(* CoDeSys 2.3.9.47 project: WTP_Pro_23_6_2016.pro *)
(* Libraries: STANDARD.LIB 5.6.98 12:03:02 *)

(* Task configuration *)
TASK Standard (PRIORITY := 0, INTERVAL := T#500ms);
	MAIN
END_TASK

(* Global variable list: Global_Variables *)
VAR_GLOBAL
	dummy: BOOL;
	LSH620 : inBlock;
	GlobalON: TIME := T#5s;
	GlobalOFF: TIME := T#5s;
END_VAR

(* Global variable list: TwinCAT_Configuration *)
(* Generated automatically by TwinCAT - (read only) *)
VAR_CONFIG
	GRIT_REMOVAL_OPERATION.B101A.dutyRemoteMode AT %IX2.1 : BOOL;
	GRIT_REMOVAL_OPERATION.B101A.dutyOverload AT %IX2.2 : BOOL;
	GRIT_REMOVAL_OPERATION.B101A.dutyIncomplete AT %IX2.3 : BOOL;
	GRIT_REMOVAL_OPERATION.B101A.dutyStart AT %IX2.4 : BOOL;
	GRIT_REMOVAL_OPERATION.B101A.standbyRemoteMode AT %IX2.5 : BOOL;
	GRIT_REMOVAL_OPERATION.B101A.standbyOverload AT %IX2.6 : BOOL;
	GRIT_REMOVAL_OPERATION.B101A.standbyIncomplete AT %IX2.7 : BOOL;
	GRIT_REMOVAL_OPERATION.B101A.standbyStart AT %IX3.0 : BOOL;
	GRIT_REMOVAL_OPERATION.B101A.thirdRemoteMode AT %IX3.1 : BOOL;
	GRIT_REMOVAL_OPERATION.B101A.thirdOverload AT %IX3.2 : BOOL;
	GRIT_REMOVAL_OPERATION.B101A.thirdStart AT %IX3.3 : BOOL;
	GRIT_REMOVAL_OPERATION.B101A.thirdIncomplete AT %IX3.4 : BOOL;
	GRIT_REMOVAL_OPERATION.B101A.standbyClose AT %IX3.5 : BOOL;
	GRIT_REMOVAL_OPERATION.B101A.dutyClose AT %IX3.6 : BOOL;
	GRIT_REMOVAL_OPERATION.B101A.thirdClose AT %IX3.7 : BOOL;
	GRIT_REMOVAL_OPERATION.B101A.dutyAdditionalStat AT %IX4.0 : BOOL;
	GRIT_REMOVAL_OPERATION.B101A.remoteAdditionalStat AT %IX4.1 : BOOL;
	GRIT_REMOVAL_OPERATION.B101A.thirdAdditionalStat AT %IX4.2 : BOOL;
	GRIT_REMOVAL_OPERATION.B101A.dutyCommand AT %QX0.0 : BOOL;
	GRIT_REMOVAL_OPERATION.B101A.standbyCommand AT %QX0.1 : BOOL;
	GRIT_REMOVAL_OPERATION.B101A.thirdCommand AT %QX0.2 : BOOL;
	GRIT_REMOVAL_OPERATION.XV100A.dutyRemoteMode AT %IX4.3 : BOOL;
	GRIT_REMOVAL_OPERATION.XV100A.dutyOverload AT %IX4.4 : BOOL;
	GRIT_REMOVAL_OPERATION.XV100A.dutyIncomplete AT %IX4.5 : BOOL;
	GRIT_REMOVAL_OPERATION.XV100A.dutyStart AT %IX4.6 : BOOL;
	GRIT_REMOVAL_OPERATION.XV100A.standbyRemoteMode AT %IX4.7 : BOOL;
	GRIT_REMOVAL_OPERATION.XV100A.standbyOverload AT %IX5.0 : BOOL;
	GRIT_REMOVAL_OPERATION.XV100A.standbyIncomplete AT %IX5.1 : BOOL;
	GRIT_REMOVAL_OPERATION.XV100A.standbyStart AT %IX5.2 : BOOL;
	GRIT_REMOVAL_OPERATION.XV100A.thirdRemoteMode AT %IX5.3 : BOOL;
	GRIT_REMOVAL_OPERATION.XV100A.thirdOverload AT %IX5.4 : BOOL;
	GRIT_REMOVAL_OPERATION.XV100A.thirdStart AT %IX5.5 : BOOL;
	GRIT_REMOVAL_OPERATION.XV100A.thirdIncomplete AT %IX5.6 : BOOL;
	GRIT_REMOVAL_OPERATION.XV100A.standbyClose AT %IX5.7 : BOOL;
	GRIT_REMOVAL_OPERATION.XV100A.dutyClose AT %IX6.0 : BOOL;
	GRIT_REMOVAL_OPERATION.XV100A.thirdClose AT %IX6.1 : BOOL;
	GRIT_REMOVAL_OPERATION.XV100A.dutyAdditionalStat AT %IX6.2 : BOOL;
	GRIT_REMOVAL_OPERATION.XV100A.remoteAdditionalStat AT %IX6.3 : BOOL;
	GRIT_REMOVAL_OPERATION.XV100A.thirdAdditionalStat AT %IX6.4 : BOOL;
	GRIT_REMOVAL_OPERATION.XV100A.dutyCommand AT %QX0.3 : BOOL;
	GRIT_REMOVAL_OPERATION.XV100A.standbyCommand AT %QX0.4 : BOOL;
	GRIT_REMOVAL_OPERATION.XV100A.thirdCommand AT %QX0.5 : BOOL;
	GRIT_REMOVAL_OPERATION.XV100B.dutyRemoteMode AT %IX6.5 : BOOL;
	GRIT_REMOVAL_OPERATION.XV100B.dutyOverload AT %IX6.6 : BOOL;
	GRIT_REMOVAL_OPERATION.XV100B.dutyIncomplete AT %IX6.7 : BOOL;
	GRIT_REMOVAL_OPERATION.XV100B.dutyStart AT %IX7.0 : BOOL;
	GRIT_REMOVAL_OPERATION.XV100B.standbyRemoteMode AT %IX7.1 : BOOL;
	GRIT_REMOVAL_OPERATION.XV100B.standbyOverload AT %IX7.2 : BOOL;
	GRIT_REMOVAL_OPERATION.XV100B.standbyIncomplete AT %IX7.3 : BOOL;
	GRIT_REMOVAL_OPERATION.XV100B.standbyStart AT %IX7.4 : BOOL;
	GRIT_REMOVAL_OPERATION.XV100B.thirdRemoteMode AT %IX7.5 : BOOL;
	GRIT_REMOVAL_OPERATION.XV100B.thirdOverload AT %IX7.6 : BOOL;
	GRIT_REMOVAL_OPERATION.XV100B.thirdStart AT %IX7.7 : BOOL;
	GRIT_REMOVAL_OPERATION.XV100B.thirdIncomplete AT %IX8.0 : BOOL;
	GRIT_REMOVAL_OPERATION.XV100B.standbyClose AT %IX8.1 : BOOL;
	GRIT_REMOVAL_OPERATION.XV100B.dutyClose AT %IX8.2 : BOOL;
	GRIT_REMOVAL_OPERATION.XV100B.thirdClose AT %IX8.3 : BOOL;
	GRIT_REMOVAL_OPERATION.XV100B.dutyAdditionalStat AT %IX8.4 : BOOL;
	GRIT_REMOVAL_OPERATION.XV100B.remoteAdditionalStat AT %IX8.5 : BOOL;
	GRIT_REMOVAL_OPERATION.XV100B.thirdAdditionalStat AT %IX8.6 : BOOL;
	GRIT_REMOVAL_OPERATION.XV100B.dutyCommand AT %QX0.6 : BOOL;
	GRIT_REMOVAL_OPERATION.XV100B.standbyCommand AT %QX0.7 : BOOL;
	GRIT_REMOVAL_OPERATION.XV100B.thirdCommand AT %QX1.0 : BOOL;
	GRIT_REMOVAL_OPERATION.C103AandB.dutyRemoteMode AT %IX8.7 : BOOL;
	GRIT_REMOVAL_OPERATION.C103AandB.dutyOverload AT %IX9.0 : BOOL;
	GRIT_REMOVAL_OPERATION.C103AandB.dutyIncomplete AT %IX9.1 : BOOL;
	GRIT_REMOVAL_OPERATION.C103AandB.dutyStart AT %IX9.2 : BOOL;
	GRIT_REMOVAL_OPERATION.C103AandB.standbyRemoteMode AT %IX9.3 : BOOL;
	GRIT_REMOVAL_OPERATION.C103AandB.standbyOverload AT %IX9.4 : BOOL;
	GRIT_REMOVAL_OPERATION.C103AandB.standbyIncomplete AT %IX9.5 : BOOL;
	GRIT_REMOVAL_OPERATION.C103AandB.standbyStart AT %IX9.6 : BOOL;
	GRIT_REMOVAL_OPERATION.C103AandB.thirdRemoteMode AT %IX9.7 : BOOL;
	GRIT_REMOVAL_OPERATION.C103AandB.thirdOverload AT %IX10.0 : BOOL;
	GRIT_REMOVAL_OPERATION.C103AandB.thirdStart AT %IX10.1 : BOOL;
	GRIT_REMOVAL_OPERATION.C103AandB.thirdIncomplete AT %IX10.2 : BOOL;
	GRIT_REMOVAL_OPERATION.C103AandB.standbyClose AT %IX10.3 : BOOL;
	GRIT_REMOVAL_OPERATION.C103AandB.dutyClose AT %IX10.4 : BOOL;
	GRIT_REMOVAL_OPERATION.C103AandB.thirdClose AT %IX10.5 : BOOL;
	GRIT_REMOVAL_OPERATION.C103AandB.dutyAdditionalStat AT %IX10.6 : BOOL;
	GRIT_REMOVAL_OPERATION.C103AandB.remoteAdditionalStat AT %IX10.7 : BOOL;
	GRIT_REMOVAL_OPERATION.C103AandB.thirdAdditionalStat AT %IX11.0 : BOOL;
	GRIT_REMOVAL_OPERATION.C103AandB.dutyCommand AT %QX1.1 : BOOL;
	GRIT_REMOVAL_OPERATION.C103AandB.standbyCommand AT %QX1.2 : BOOL;
	GRIT_REMOVAL_OPERATION.C103AandB.thirdCommand AT %QX1.3 : BOOL;
	INLET_SCREENING_OPERATION_1.LSH105A.IN AT %IX38.7 : BOOL;
	INLET_SCREENING_OPERATION_1.LSHH105A.IN AT %IX39.0 : BOOL;
	INLET_SCREENING_OPERATION_1.F101A.dutyRemoteMode AT %IX39.1 : BOOL;
	INLET_SCREENING_OPERATION_1.F101A.dutyOverload AT %IX39.2 : BOOL;
	INLET_SCREENING_OPERATION_1.F101A.dutyIncomplete AT %IX39.3 : BOOL;
	INLET_SCREENING_OPERATION_1.F101A.dutyStart AT %IX39.4 : BOOL;
	INLET_SCREENING_OPERATION_1.F101A.standbyRemoteMode AT %IX39.5 : BOOL;
	INLET_SCREENING_OPERATION_1.F101A.standbyOverload AT %IX39.6 : BOOL;
	INLET_SCREENING_OPERATION_1.F101A.standbyIncomplete AT %IX39.7 : BOOL;
	INLET_SCREENING_OPERATION_1.F101A.standbyStart AT %IX40.0 : BOOL;
	INLET_SCREENING_OPERATION_1.F101A.thirdRemoteMode AT %IX40.1 : BOOL;
	INLET_SCREENING_OPERATION_1.F101A.thirdOverload AT %IX40.2 : BOOL;
	INLET_SCREENING_OPERATION_1.F101A.thirdStart AT %IX40.3 : BOOL;
	INLET_SCREENING_OPERATION_1.F101A.thirdIncomplete AT %IX40.4 : BOOL;
	INLET_SCREENING_OPERATION_1.F101A.standbyClose AT %IX40.5 : BOOL;
	INLET_SCREENING_OPERATION_1.F101A.dutyClose AT %IX40.6 : BOOL;
	INLET_SCREENING_OPERATION_1.F101A.thirdClose AT %IX40.7 : BOOL;
	INLET_SCREENING_OPERATION_1.F101A.dutyAdditionalStat AT %IX41.0 : BOOL;
	INLET_SCREENING_OPERATION_1.F101A.remoteAdditionalStat AT %IX41.1 : BOOL;
	INLET_SCREENING_OPERATION_1.F101A.thirdAdditionalStat AT %IX41.2 : BOOL;
	INLET_SCREENING_OPERATION_1.F101A.dutyCommand AT %QX5.5 : BOOL;
	INLET_SCREENING_OPERATION_1.F101A.standbyCommand AT %QX5.6 : BOOL;
	INLET_SCREENING_OPERATION_1.F101A.thirdCommand AT %QX5.7 : BOOL;
	INLET_SCREENING_OPERATION_1.XV101A1.dutyRemoteMode AT %IX41.3 : BOOL;
	INLET_SCREENING_OPERATION_1.XV101A1.dutyOverload AT %IX41.4 : BOOL;
	INLET_SCREENING_OPERATION_1.XV101A1.dutyIncomplete AT %IX41.5 : BOOL;
	INLET_SCREENING_OPERATION_1.XV101A1.dutyStart AT %IX41.6 : BOOL;
	INLET_SCREENING_OPERATION_1.XV101A1.standbyRemoteMode AT %IX41.7 : BOOL;
	INLET_SCREENING_OPERATION_1.XV101A1.standbyOverload AT %IX42.0 : BOOL;
	INLET_SCREENING_OPERATION_1.XV101A1.standbyIncomplete AT %IX42.1 : BOOL;
	INLET_SCREENING_OPERATION_1.XV101A1.standbyStart AT %IX42.2 : BOOL;
	INLET_SCREENING_OPERATION_1.XV101A1.thirdRemoteMode AT %IX42.3 : BOOL;
	INLET_SCREENING_OPERATION_1.XV101A1.thirdOverload AT %IX42.4 : BOOL;
	INLET_SCREENING_OPERATION_1.XV101A1.thirdStart AT %IX42.5 : BOOL;
	INLET_SCREENING_OPERATION_1.XV101A1.thirdIncomplete AT %IX42.6 : BOOL;
	INLET_SCREENING_OPERATION_1.XV101A1.standbyClose AT %IX42.7 : BOOL;
	INLET_SCREENING_OPERATION_1.XV101A1.dutyClose AT %IX43.0 : BOOL;
	INLET_SCREENING_OPERATION_1.XV101A1.thirdClose AT %IX43.1 : BOOL;
	INLET_SCREENING_OPERATION_1.XV101A1.dutyAdditionalStat AT %IX43.2 : BOOL;
	INLET_SCREENING_OPERATION_1.XV101A1.remoteAdditionalStat AT %IX43.3 : BOOL;
	INLET_SCREENING_OPERATION_1.XV101A1.thirdAdditionalStat AT %IX43.4 : BOOL;
	INLET_SCREENING_OPERATION_1.XV101A1.dutyCommand AT %QX6.0 : BOOL;
	INLET_SCREENING_OPERATION_1.XV101A1.standbyCommand AT %QX6.1 : BOOL;
	INLET_SCREENING_OPERATION_1.XV101A1.thirdCommand AT %QX6.2 : BOOL;
	INLET_SCREENING_OPERATION_1.XV101A2.dutyRemoteMode AT %IX43.5 : BOOL;
	INLET_SCREENING_OPERATION_1.XV101A2.dutyOverload AT %IX43.6 : BOOL;
	INLET_SCREENING_OPERATION_1.XV101A2.dutyIncomplete AT %IX43.7 : BOOL;
	INLET_SCREENING_OPERATION_1.XV101A2.dutyStart AT %IX44.0 : BOOL;
	INLET_SCREENING_OPERATION_1.XV101A2.standbyRemoteMode AT %IX44.1 : BOOL;
	INLET_SCREENING_OPERATION_1.XV101A2.standbyOverload AT %IX44.2 : BOOL;
	INLET_SCREENING_OPERATION_1.XV101A2.standbyIncomplete AT %IX44.3 : BOOL;
	INLET_SCREENING_OPERATION_1.XV101A2.standbyStart AT %IX44.4 : BOOL;
	INLET_SCREENING_OPERATION_1.XV101A2.thirdRemoteMode AT %IX44.5 : BOOL;
	INLET_SCREENING_OPERATION_1.XV101A2.thirdOverload AT %IX44.6 : BOOL;
	INLET_SCREENING_OPERATION_1.XV101A2.thirdStart AT %IX44.7 : BOOL;
	INLET_SCREENING_OPERATION_1.XV101A2.thirdIncomplete AT %IX45.0 : BOOL;
	INLET_SCREENING_OPERATION_1.XV101A2.standbyClose AT %IX45.1 : BOOL;
	INLET_SCREENING_OPERATION_1.XV101A2.dutyClose AT %IX45.2 : BOOL;
	INLET_SCREENING_OPERATION_1.XV101A2.thirdClose AT %IX45.3 : BOOL;
	INLET_SCREENING_OPERATION_1.XV101A2.dutyAdditionalStat AT %IX45.4 : BOOL;
	INLET_SCREENING_OPERATION_1.XV101A2.remoteAdditionalStat AT %IX45.5 : BOOL;
	INLET_SCREENING_OPERATION_1.XV101A2.thirdAdditionalStat AT %IX45.6 : BOOL;
	INLET_SCREENING_OPERATION_1.XV101A2.dutyCommand AT %QX6.3 : BOOL;
	INLET_SCREENING_OPERATION_1.XV101A2.standbyCommand AT %QX6.4 : BOOL;
	INLET_SCREENING_OPERATION_1.XV101A2.thirdCommand AT %QX6.5 : BOOL;
	INLET_SCREENING_OPERATION_1.PS101A.dutyRemoteMode AT %IX45.7 : BOOL;
	INLET_SCREENING_OPERATION_1.PS101A.dutyOverload AT %IX46.0 : BOOL;
	INLET_SCREENING_OPERATION_1.PS101A.dutyIncomplete AT %IX46.1 : BOOL;
	INLET_SCREENING_OPERATION_1.PS101A.dutyStart AT %IX46.2 : BOOL;
	INLET_SCREENING_OPERATION_1.PS101A.standbyRemoteMode AT %IX46.3 : BOOL;
	INLET_SCREENING_OPERATION_1.PS101A.standbyOverload AT %IX46.4 : BOOL;
	INLET_SCREENING_OPERATION_1.PS101A.standbyIncomplete AT %IX46.5 : BOOL;
	INLET_SCREENING_OPERATION_1.PS101A.standbyStart AT %IX46.6 : BOOL;
	INLET_SCREENING_OPERATION_1.PS101A.thirdRemoteMode AT %IX46.7 : BOOL;
	INLET_SCREENING_OPERATION_1.PS101A.thirdOverload AT %IX47.0 : BOOL;
	INLET_SCREENING_OPERATION_1.PS101A.thirdStart AT %IX47.1 : BOOL;
	INLET_SCREENING_OPERATION_1.PS101A.thirdIncomplete AT %IX47.2 : BOOL;
	INLET_SCREENING_OPERATION_1.PS101A.standbyClose AT %IX47.3 : BOOL;
	INLET_SCREENING_OPERATION_1.PS101A.dutyClose AT %IX47.4 : BOOL;
	INLET_SCREENING_OPERATION_1.PS101A.thirdClose AT %IX47.5 : BOOL;
	INLET_SCREENING_OPERATION_1.PS101A.dutyAdditionalStat AT %IX47.6 : BOOL;
	INLET_SCREENING_OPERATION_1.PS101A.remoteAdditionalStat AT %IX47.7 : BOOL;
	INLET_SCREENING_OPERATION_1.PS101A.thirdAdditionalStat AT %IX48.0 : BOOL;
	INLET_SCREENING_OPERATION_1.PS101A.dutyCommand AT %QX6.6 : BOOL;
	INLET_SCREENING_OPERATION_1.PS101A.standbyCommand AT %QX6.7 : BOOL;
	INLET_SCREENING_OPERATION_1.PS101A.thirdCommand AT %QX7.0 : BOOL;
	INLET_SCREENING_OPERATION_1.C102A.dutyRemoteMode AT %IX48.1 : BOOL;
	INLET_SCREENING_OPERATION_1.C102A.dutyOverload AT %IX48.2 : BOOL;
	INLET_SCREENING_OPERATION_1.C102A.dutyIncomplete AT %IX48.3 : BOOL;
	INLET_SCREENING_OPERATION_1.C102A.dutyStart AT %IX48.4 : BOOL;
	INLET_SCREENING_OPERATION_1.C102A.standbyRemoteMode AT %IX48.5 : BOOL;
	INLET_SCREENING_OPERATION_1.C102A.standbyOverload AT %IX48.6 : BOOL;
	INLET_SCREENING_OPERATION_1.C102A.standbyIncomplete AT %IX48.7 : BOOL;
	INLET_SCREENING_OPERATION_1.C102A.standbyStart AT %IX49.0 : BOOL;
	INLET_SCREENING_OPERATION_1.C102A.thirdRemoteMode AT %IX49.1 : BOOL;
	INLET_SCREENING_OPERATION_1.C102A.thirdOverload AT %IX49.2 : BOOL;
	INLET_SCREENING_OPERATION_1.C102A.thirdStart AT %IX49.3 : BOOL;
	INLET_SCREENING_OPERATION_1.C102A.thirdIncomplete AT %IX49.4 : BOOL;
	INLET_SCREENING_OPERATION_1.C102A.standbyClose AT %IX49.5 : BOOL;
	INLET_SCREENING_OPERATION_1.C102A.dutyClose AT %IX49.6 : BOOL;
	INLET_SCREENING_OPERATION_1.C102A.thirdClose AT %IX49.7 : BOOL;
	INLET_SCREENING_OPERATION_1.C102A.dutyAdditionalStat AT %IX50.0 : BOOL;
	INLET_SCREENING_OPERATION_1.C102A.remoteAdditionalStat AT %IX50.1 : BOOL;
	INLET_SCREENING_OPERATION_1.C102A.thirdAdditionalStat AT %IX50.2 : BOOL;
	INLET_SCREENING_OPERATION_1.C102A.dutyCommand AT %QX7.1 : BOOL;
	INLET_SCREENING_OPERATION_1.C102A.standbyCommand AT %QX7.2 : BOOL;
	INLET_SCREENING_OPERATION_1.C102A.thirdCommand AT %QX7.3 : BOOL;
	INLET_SCREENING_OPERATION_1.C101A.dutyRemoteMode AT %IX50.3 : BOOL;
	INLET_SCREENING_OPERATION_1.C101A.dutyOverload AT %IX50.4 : BOOL;
	INLET_SCREENING_OPERATION_1.C101A.dutyIncomplete AT %IX50.5 : BOOL;
	INLET_SCREENING_OPERATION_1.C101A.dutyStart AT %IX50.6 : BOOL;
	INLET_SCREENING_OPERATION_1.C101A.standbyRemoteMode AT %IX50.7 : BOOL;
	INLET_SCREENING_OPERATION_1.C101A.standbyOverload AT %IX51.0 : BOOL;
	INLET_SCREENING_OPERATION_1.C101A.standbyIncomplete AT %IX51.1 : BOOL;
	INLET_SCREENING_OPERATION_1.C101A.standbyStart AT %IX51.2 : BOOL;
	INLET_SCREENING_OPERATION_1.C101A.thirdRemoteMode AT %IX51.3 : BOOL;
	INLET_SCREENING_OPERATION_1.C101A.thirdOverload AT %IX51.4 : BOOL;
	INLET_SCREENING_OPERATION_1.C101A.thirdStart AT %IX51.5 : BOOL;
	INLET_SCREENING_OPERATION_1.C101A.thirdIncomplete AT %IX51.6 : BOOL;
	INLET_SCREENING_OPERATION_1.C101A.standbyClose AT %IX51.7 : BOOL;
	INLET_SCREENING_OPERATION_1.C101A.dutyClose AT %IX52.0 : BOOL;
	INLET_SCREENING_OPERATION_1.C101A.thirdClose AT %IX52.1 : BOOL;
	INLET_SCREENING_OPERATION_1.C101A.dutyAdditionalStat AT %IX52.2 : BOOL;
	INLET_SCREENING_OPERATION_1.C101A.remoteAdditionalStat AT %IX52.3 : BOOL;
	INLET_SCREENING_OPERATION_1.C101A.thirdAdditionalStat AT %IX52.4 : BOOL;
	INLET_SCREENING_OPERATION_1.C101A.dutyCommand AT %QX7.4 : BOOL;
	INLET_SCREENING_OPERATION_1.C101A.standbyCommand AT %QX7.5 : BOOL;
	INLET_SCREENING_OPERATION_1.C101A.thirdCommand AT %QX7.6 : BOOL;
	INLET_SCREENING_OPERATION_1.XV102A.dutyRemoteMode AT %IX52.5 : BOOL;
	INLET_SCREENING_OPERATION_1.XV102A.dutyOverload AT %IX52.6 : BOOL;
	INLET_SCREENING_OPERATION_1.XV102A.dutyIncomplete AT %IX52.7 : BOOL;
	INLET_SCREENING_OPERATION_1.XV102A.dutyStart AT %IX53.0 : BOOL;
	INLET_SCREENING_OPERATION_1.XV102A.standbyRemoteMode AT %IX53.1 : BOOL;
	INLET_SCREENING_OPERATION_1.XV102A.standbyOverload AT %IX53.2 : BOOL;
	INLET_SCREENING_OPERATION_1.XV102A.standbyIncomplete AT %IX53.3 : BOOL;
	INLET_SCREENING_OPERATION_1.XV102A.standbyStart AT %IX53.4 : BOOL;
	INLET_SCREENING_OPERATION_1.XV102A.thirdRemoteMode AT %IX53.5 : BOOL;
	INLET_SCREENING_OPERATION_1.XV102A.thirdOverload AT %IX53.6 : BOOL;
	INLET_SCREENING_OPERATION_1.XV102A.thirdStart AT %IX53.7 : BOOL;
	INLET_SCREENING_OPERATION_1.XV102A.thirdIncomplete AT %IX54.0 : BOOL;
	INLET_SCREENING_OPERATION_1.XV102A.standbyClose AT %IX54.1 : BOOL;
	INLET_SCREENING_OPERATION_1.XV102A.dutyClose AT %IX54.2 : BOOL;
	INLET_SCREENING_OPERATION_1.XV102A.thirdClose AT %IX54.3 : BOOL;
	INLET_SCREENING_OPERATION_1.XV102A.dutyAdditionalStat AT %IX54.4 : BOOL;
	INLET_SCREENING_OPERATION_1.XV102A.remoteAdditionalStat AT %IX54.5 : BOOL;
	INLET_SCREENING_OPERATION_1.XV102A.thirdAdditionalStat AT %IX54.6 : BOOL;
	INLET_SCREENING_OPERATION_1.XV102A.dutyCommand AT %QX7.7 : BOOL;
	INLET_SCREENING_OPERATION_1.XV102A.standbyCommand AT %QX8.0 : BOOL;
	INLET_SCREENING_OPERATION_1.XV102A.thirdCommand AT %QX8.1 : BOOL;
	INLET_SCREENING_OPERATION_2.LSH105B.IN AT %IX54.7 : BOOL;
	INLET_SCREENING_OPERATION_2.LSHH105B.IN AT %IX55.0 : BOOL;
	INLET_SCREENING_OPERATION_2.F101B.dutyRemoteMode AT %IX55.1 : BOOL;
	INLET_SCREENING_OPERATION_2.F101B.dutyOverload AT %IX55.2 : BOOL;
	INLET_SCREENING_OPERATION_2.F101B.dutyIncomplete AT %IX55.3 : BOOL;
	INLET_SCREENING_OPERATION_2.F101B.dutyStart AT %IX55.4 : BOOL;
	INLET_SCREENING_OPERATION_2.F101B.standbyRemoteMode AT %IX55.5 : BOOL;
	INLET_SCREENING_OPERATION_2.F101B.standbyOverload AT %IX55.6 : BOOL;
	INLET_SCREENING_OPERATION_2.F101B.standbyIncomplete AT %IX55.7 : BOOL;
	INLET_SCREENING_OPERATION_2.F101B.standbyStart AT %IX56.0 : BOOL;
	INLET_SCREENING_OPERATION_2.F101B.thirdRemoteMode AT %IX56.1 : BOOL;
	INLET_SCREENING_OPERATION_2.F101B.thirdOverload AT %IX56.2 : BOOL;
	INLET_SCREENING_OPERATION_2.F101B.thirdStart AT %IX56.3 : BOOL;
	INLET_SCREENING_OPERATION_2.F101B.thirdIncomplete AT %IX56.4 : BOOL;
	INLET_SCREENING_OPERATION_2.F101B.standbyClose AT %IX56.5 : BOOL;
	INLET_SCREENING_OPERATION_2.F101B.dutyClose AT %IX56.6 : BOOL;
	INLET_SCREENING_OPERATION_2.F101B.thirdClose AT %IX56.7 : BOOL;
	INLET_SCREENING_OPERATION_2.F101B.dutyAdditionalStat AT %IX57.0 : BOOL;
	INLET_SCREENING_OPERATION_2.F101B.remoteAdditionalStat AT %IX57.1 : BOOL;
	INLET_SCREENING_OPERATION_2.F101B.thirdAdditionalStat AT %IX57.2 : BOOL;
	INLET_SCREENING_OPERATION_2.F101B.dutyCommand AT %QX8.2 : BOOL;
	INLET_SCREENING_OPERATION_2.F101B.standbyCommand AT %QX8.3 : BOOL;
	INLET_SCREENING_OPERATION_2.F101B.thirdCommand AT %QX8.4 : BOOL;
	INLET_SCREENING_OPERATION_2.XV101B1.dutyRemoteMode AT %IX57.3 : BOOL;
	INLET_SCREENING_OPERATION_2.XV101B1.dutyOverload AT %IX57.4 : BOOL;
	INLET_SCREENING_OPERATION_2.XV101B1.dutyIncomplete AT %IX57.5 : BOOL;
	INLET_SCREENING_OPERATION_2.XV101B1.dutyStart AT %IX57.6 : BOOL;
	INLET_SCREENING_OPERATION_2.XV101B1.standbyRemoteMode AT %IX57.7 : BOOL;
	INLET_SCREENING_OPERATION_2.XV101B1.standbyOverload AT %IX58.0 : BOOL;
	INLET_SCREENING_OPERATION_2.XV101B1.standbyIncomplete AT %IX58.1 : BOOL;
	INLET_SCREENING_OPERATION_2.XV101B1.standbyStart AT %IX58.2 : BOOL;
	INLET_SCREENING_OPERATION_2.XV101B1.thirdRemoteMode AT %IX58.3 : BOOL;
	INLET_SCREENING_OPERATION_2.XV101B1.thirdOverload AT %IX58.4 : BOOL;
	INLET_SCREENING_OPERATION_2.XV101B1.thirdStart AT %IX58.5 : BOOL;
	INLET_SCREENING_OPERATION_2.XV101B1.thirdIncomplete AT %IX58.6 : BOOL;
	INLET_SCREENING_OPERATION_2.XV101B1.standbyClose AT %IX58.7 : BOOL;
	INLET_SCREENING_OPERATION_2.XV101B1.dutyClose AT %IX59.0 : BOOL;
	INLET_SCREENING_OPERATION_2.XV101B1.thirdClose AT %IX59.1 : BOOL;
	INLET_SCREENING_OPERATION_2.XV101B1.dutyAdditionalStat AT %IX59.2 : BOOL;
	INLET_SCREENING_OPERATION_2.XV101B1.remoteAdditionalStat AT %IX59.3 : BOOL;
	INLET_SCREENING_OPERATION_2.XV101B1.thirdAdditionalStat AT %IX59.4 : BOOL;
	INLET_SCREENING_OPERATION_2.XV101B1.dutyCommand AT %QX8.5 : BOOL;
	INLET_SCREENING_OPERATION_2.XV101B1.standbyCommand AT %QX8.6 : BOOL;
	INLET_SCREENING_OPERATION_2.XV101B1.thirdCommand AT %QX8.7 : BOOL;
	INLET_SCREENING_OPERATION_2.XV101B2.dutyRemoteMode AT %IX59.5 : BOOL;
	INLET_SCREENING_OPERATION_2.XV101B2.dutyOverload AT %IX59.6 : BOOL;
	INLET_SCREENING_OPERATION_2.XV101B2.dutyIncomplete AT %IX59.7 : BOOL;
	INLET_SCREENING_OPERATION_2.XV101B2.dutyStart AT %IX60.0 : BOOL;
	INLET_SCREENING_OPERATION_2.XV101B2.standbyRemoteMode AT %IX60.1 : BOOL;
	INLET_SCREENING_OPERATION_2.XV101B2.standbyOverload AT %IX60.2 : BOOL;
	INLET_SCREENING_OPERATION_2.XV101B2.standbyIncomplete AT %IX60.3 : BOOL;
	INLET_SCREENING_OPERATION_2.XV101B2.standbyStart AT %IX60.4 : BOOL;
	INLET_SCREENING_OPERATION_2.XV101B2.thirdRemoteMode AT %IX60.5 : BOOL;
	INLET_SCREENING_OPERATION_2.XV101B2.thirdOverload AT %IX60.6 : BOOL;
	INLET_SCREENING_OPERATION_2.XV101B2.thirdStart AT %IX60.7 : BOOL;
	INLET_SCREENING_OPERATION_2.XV101B2.thirdIncomplete AT %IX61.0 : BOOL;
	INLET_SCREENING_OPERATION_2.XV101B2.standbyClose AT %IX61.1 : BOOL;
	INLET_SCREENING_OPERATION_2.XV101B2.dutyClose AT %IX61.2 : BOOL;
	INLET_SCREENING_OPERATION_2.XV101B2.thirdClose AT %IX61.3 : BOOL;
	INLET_SCREENING_OPERATION_2.XV101B2.dutyAdditionalStat AT %IX61.4 : BOOL;
	INLET_SCREENING_OPERATION_2.XV101B2.remoteAdditionalStat AT %IX61.5 : BOOL;
	INLET_SCREENING_OPERATION_2.XV101B2.thirdAdditionalStat AT %IX61.6 : BOOL;
	INLET_SCREENING_OPERATION_2.XV101B2.dutyCommand AT %QX9.0 : BOOL;
	INLET_SCREENING_OPERATION_2.XV101B2.standbyCommand AT %QX9.1 : BOOL;
	INLET_SCREENING_OPERATION_2.XV101B2.thirdCommand AT %QX9.2 : BOOL;
	INLET_SCREENING_OPERATION_2.PS101B.dutyRemoteMode AT %IX61.7 : BOOL;
	INLET_SCREENING_OPERATION_2.PS101B.dutyOverload AT %IX62.0 : BOOL;
	INLET_SCREENING_OPERATION_2.PS101B.dutyIncomplete AT %IX62.1 : BOOL;
	INLET_SCREENING_OPERATION_2.PS101B.dutyStart AT %IX62.2 : BOOL;
	INLET_SCREENING_OPERATION_2.PS101B.standbyRemoteMode AT %IX62.3 : BOOL;
	INLET_SCREENING_OPERATION_2.PS101B.standbyOverload AT %IX62.4 : BOOL;
	INLET_SCREENING_OPERATION_2.PS101B.standbyIncomplete AT %IX62.5 : BOOL;
	INLET_SCREENING_OPERATION_2.PS101B.standbyStart AT %IX62.6 : BOOL;
	INLET_SCREENING_OPERATION_2.PS101B.thirdRemoteMode AT %IX62.7 : BOOL;
	INLET_SCREENING_OPERATION_2.PS101B.thirdOverload AT %IX63.0 : BOOL;
	INLET_SCREENING_OPERATION_2.PS101B.thirdStart AT %IX63.1 : BOOL;
	INLET_SCREENING_OPERATION_2.PS101B.thirdIncomplete AT %IX63.2 : BOOL;
	INLET_SCREENING_OPERATION_2.PS101B.standbyClose AT %IX63.3 : BOOL;
	INLET_SCREENING_OPERATION_2.PS101B.dutyClose AT %IX63.4 : BOOL;
	INLET_SCREENING_OPERATION_2.PS101B.thirdClose AT %IX63.5 : BOOL;
	INLET_SCREENING_OPERATION_2.PS101B.dutyAdditionalStat AT %IX63.6 : BOOL;
	INLET_SCREENING_OPERATION_2.PS101B.remoteAdditionalStat AT %IX63.7 : BOOL;
	INLET_SCREENING_OPERATION_2.PS101B.thirdAdditionalStat AT %IX64.0 : BOOL;
	INLET_SCREENING_OPERATION_2.PS101B.dutyCommand AT %QX9.3 : BOOL;
	INLET_SCREENING_OPERATION_2.PS101B.standbyCommand AT %QX9.4 : BOOL;
	INLET_SCREENING_OPERATION_2.PS101B.thirdCommand AT %QX9.5 : BOOL;
	INLET_SCREENING_OPERATION_2.C102B.dutyRemoteMode AT %IX64.1 : BOOL;
	INLET_SCREENING_OPERATION_2.C102B.dutyOverload AT %IX64.2 : BOOL;
	INLET_SCREENING_OPERATION_2.C102B.dutyIncomplete AT %IX64.3 : BOOL;
	INLET_SCREENING_OPERATION_2.C102B.dutyStart AT %IX64.4 : BOOL;
	INLET_SCREENING_OPERATION_2.C102B.standbyRemoteMode AT %IX64.5 : BOOL;
	INLET_SCREENING_OPERATION_2.C102B.standbyOverload AT %IX64.6 : BOOL;
	INLET_SCREENING_OPERATION_2.C102B.standbyIncomplete AT %IX64.7 : BOOL;
	INLET_SCREENING_OPERATION_2.C102B.standbyStart AT %IX65.0 : BOOL;
	INLET_SCREENING_OPERATION_2.C102B.thirdRemoteMode AT %IX65.1 : BOOL;
	INLET_SCREENING_OPERATION_2.C102B.thirdOverload AT %IX65.2 : BOOL;
	INLET_SCREENING_OPERATION_2.C102B.thirdStart AT %IX65.3 : BOOL;
	INLET_SCREENING_OPERATION_2.C102B.thirdIncomplete AT %IX65.4 : BOOL;
	INLET_SCREENING_OPERATION_2.C102B.standbyClose AT %IX65.5 : BOOL;
	INLET_SCREENING_OPERATION_2.C102B.dutyClose AT %IX65.6 : BOOL;
	INLET_SCREENING_OPERATION_2.C102B.thirdClose AT %IX65.7 : BOOL;
	INLET_SCREENING_OPERATION_2.C102B.dutyAdditionalStat AT %IX66.0 : BOOL;
	INLET_SCREENING_OPERATION_2.C102B.remoteAdditionalStat AT %IX66.1 : BOOL;
	INLET_SCREENING_OPERATION_2.C102B.thirdAdditionalStat AT %IX66.2 : BOOL;
	INLET_SCREENING_OPERATION_2.C102B.dutyCommand AT %QX9.6 : BOOL;
	INLET_SCREENING_OPERATION_2.C102B.standbyCommand AT %QX9.7 : BOOL;
	INLET_SCREENING_OPERATION_2.C102B.thirdCommand AT %QX10.0 : BOOL;
	INLET_SCREENING_OPERATION_2.C101B.dutyRemoteMode AT %IX66.3 : BOOL;
	INLET_SCREENING_OPERATION_2.C101B.dutyOverload AT %IX66.4 : BOOL;
	INLET_SCREENING_OPERATION_2.C101B.dutyIncomplete AT %IX66.5 : BOOL;
	INLET_SCREENING_OPERATION_2.C101B.dutyStart AT %IX66.6 : BOOL;
	INLET_SCREENING_OPERATION_2.C101B.standbyRemoteMode AT %IX66.7 : BOOL;
	INLET_SCREENING_OPERATION_2.C101B.standbyOverload AT %IX67.0 : BOOL;
	INLET_SCREENING_OPERATION_2.C101B.standbyIncomplete AT %IX67.1 : BOOL;
	INLET_SCREENING_OPERATION_2.C101B.standbyStart AT %IX67.2 : BOOL;
	INLET_SCREENING_OPERATION_2.C101B.thirdRemoteMode AT %IX67.3 : BOOL;
	INLET_SCREENING_OPERATION_2.C101B.thirdOverload AT %IX67.4 : BOOL;
	INLET_SCREENING_OPERATION_2.C101B.thirdStart AT %IX67.5 : BOOL;
	INLET_SCREENING_OPERATION_2.C101B.thirdIncomplete AT %IX67.6 : BOOL;
	INLET_SCREENING_OPERATION_2.C101B.standbyClose AT %IX67.7 : BOOL;
	INLET_SCREENING_OPERATION_2.C101B.dutyClose AT %IX68.0 : BOOL;
	INLET_SCREENING_OPERATION_2.C101B.thirdClose AT %IX68.1 : BOOL;
	INLET_SCREENING_OPERATION_2.C101B.dutyAdditionalStat AT %IX68.2 : BOOL;
	INLET_SCREENING_OPERATION_2.C101B.remoteAdditionalStat AT %IX68.3 : BOOL;
	INLET_SCREENING_OPERATION_2.C101B.thirdAdditionalStat AT %IX68.4 : BOOL;
	INLET_SCREENING_OPERATION_2.C101B.dutyCommand AT %QX10.1 : BOOL;
	INLET_SCREENING_OPERATION_2.C101B.standbyCommand AT %QX10.2 : BOOL;
	INLET_SCREENING_OPERATION_2.C101B.thirdCommand AT %QX10.3 : BOOL;
	INLET_SCREENING_OPERATION_2.XV102B.dutyRemoteMode AT %IX68.5 : BOOL;
	INLET_SCREENING_OPERATION_2.XV102B.dutyOverload AT %IX68.6 : BOOL;
	INLET_SCREENING_OPERATION_2.XV102B.dutyIncomplete AT %IX68.7 : BOOL;
	INLET_SCREENING_OPERATION_2.XV102B.dutyStart AT %IX69.0 : BOOL;
	INLET_SCREENING_OPERATION_2.XV102B.standbyRemoteMode AT %IX69.1 : BOOL;
	INLET_SCREENING_OPERATION_2.XV102B.standbyOverload AT %IX69.2 : BOOL;
	INLET_SCREENING_OPERATION_2.XV102B.standbyIncomplete AT %IX69.3 : BOOL;
	INLET_SCREENING_OPERATION_2.XV102B.standbyStart AT %IX69.4 : BOOL;
	INLET_SCREENING_OPERATION_2.XV102B.thirdRemoteMode AT %IX69.5 : BOOL;
	INLET_SCREENING_OPERATION_2.XV102B.thirdOverload AT %IX69.6 : BOOL;
	INLET_SCREENING_OPERATION_2.XV102B.thirdStart AT %IX69.7 : BOOL;
	INLET_SCREENING_OPERATION_2.XV102B.thirdIncomplete AT %IX70.0 : BOOL;
	INLET_SCREENING_OPERATION_2.XV102B.standbyClose AT %IX70.1 : BOOL;
	INLET_SCREENING_OPERATION_2.XV102B.dutyClose AT %IX70.2 : BOOL;
	INLET_SCREENING_OPERATION_2.XV102B.thirdClose AT %IX70.3 : BOOL;
	INLET_SCREENING_OPERATION_2.XV102B.dutyAdditionalStat AT %IX70.4 : BOOL;
	INLET_SCREENING_OPERATION_2.XV102B.remoteAdditionalStat AT %IX70.5 : BOOL;
	INLET_SCREENING_OPERATION_2.XV102B.thirdAdditionalStat AT %IX70.6 : BOOL;
	INLET_SCREENING_OPERATION_2.XV102B.dutyCommand AT %QX10.4 : BOOL;
	INLET_SCREENING_OPERATION_2.XV102B.standbyCommand AT %QX10.5 : BOOL;
	INLET_SCREENING_OPERATION_2.XV102B.thirdCommand AT %QX10.6 : BOOL;
	REUSE_WATER_SYSTEM.LSH405.IN AT %IX11.1 : BOOL;
	REUSE_WATER_SYSTEM.LSL308A.IN AT %IX11.2 : BOOL;
	REUSE_WATER_SYSTEM.LSH308A.IN AT %IX11.3 : BOOL;
	REUSE_WATER_SYSTEM.FSL101.IN AT %IX11.4 : BOOL;
	REUSE_WATER_SYSTEM.PSL411 AT %IB0 : INT;
	REUSE_WATER_SYSTEM.PSL412 AT %IX2.0 : BOOL;
	REUSE_WATER_SYSTEM.P403.dutyRemoteMode AT %IX11.5 : BOOL;
	REUSE_WATER_SYSTEM.P403.dutyOverload AT %IX11.6 : BOOL;
	REUSE_WATER_SYSTEM.P403.dutyIncomplete AT %IX11.7 : BOOL;
	REUSE_WATER_SYSTEM.P403.dutyStart AT %IX12.0 : BOOL;
	REUSE_WATER_SYSTEM.P403.standbyRemoteMode AT %IX12.1 : BOOL;
	REUSE_WATER_SYSTEM.P403.standbyOverload AT %IX12.2 : BOOL;
	REUSE_WATER_SYSTEM.P403.standbyIncomplete AT %IX12.3 : BOOL;
	REUSE_WATER_SYSTEM.P403.standbyStart AT %IX12.4 : BOOL;
	REUSE_WATER_SYSTEM.P403.thirdRemoteMode AT %IX12.5 : BOOL;
	REUSE_WATER_SYSTEM.P403.thirdOverload AT %IX12.6 : BOOL;
	REUSE_WATER_SYSTEM.P403.thirdStart AT %IX12.7 : BOOL;
	REUSE_WATER_SYSTEM.P403.thirdIncomplete AT %IX13.0 : BOOL;
	REUSE_WATER_SYSTEM.P403.standbyClose AT %IX13.1 : BOOL;
	REUSE_WATER_SYSTEM.P403.dutyClose AT %IX13.2 : BOOL;
	REUSE_WATER_SYSTEM.P403.thirdClose AT %IX13.3 : BOOL;
	REUSE_WATER_SYSTEM.P403.dutyAdditionalStat AT %IX13.4 : BOOL;
	REUSE_WATER_SYSTEM.P403.remoteAdditionalStat AT %IX13.5 : BOOL;
	REUSE_WATER_SYSTEM.P403.thirdAdditionalStat AT %IX13.6 : BOOL;
	REUSE_WATER_SYSTEM.P403.dutyCommand AT %QX1.4 : BOOL;
	REUSE_WATER_SYSTEM.P403.standbyCommand AT %QX1.5 : BOOL;
	REUSE_WATER_SYSTEM.P403.thirdCommand AT %QX1.6 : BOOL;
	REUSE_WATER_SYSTEM.P402.dutyRemoteMode AT %IX13.7 : BOOL;
	REUSE_WATER_SYSTEM.P402.dutyOverload AT %IX14.0 : BOOL;
	REUSE_WATER_SYSTEM.P402.dutyIncomplete AT %IX14.1 : BOOL;
	REUSE_WATER_SYSTEM.P402.dutyStart AT %IX14.2 : BOOL;
	REUSE_WATER_SYSTEM.P402.standbyRemoteMode AT %IX14.3 : BOOL;
	REUSE_WATER_SYSTEM.P402.standbyOverload AT %IX14.4 : BOOL;
	REUSE_WATER_SYSTEM.P402.standbyIncomplete AT %IX14.5 : BOOL;
	REUSE_WATER_SYSTEM.P402.standbyStart AT %IX14.6 : BOOL;
	REUSE_WATER_SYSTEM.P402.thirdRemoteMode AT %IX14.7 : BOOL;
	REUSE_WATER_SYSTEM.P402.thirdOverload AT %IX15.0 : BOOL;
	REUSE_WATER_SYSTEM.P402.thirdStart AT %IX15.1 : BOOL;
	REUSE_WATER_SYSTEM.P402.thirdIncomplete AT %IX15.2 : BOOL;
	REUSE_WATER_SYSTEM.P402.standbyClose AT %IX15.3 : BOOL;
	REUSE_WATER_SYSTEM.P402.dutyClose AT %IX15.4 : BOOL;
	REUSE_WATER_SYSTEM.P402.thirdClose AT %IX15.5 : BOOL;
	REUSE_WATER_SYSTEM.P402.dutyAdditionalStat AT %IX15.6 : BOOL;
	REUSE_WATER_SYSTEM.P402.remoteAdditionalStat AT %IX15.7 : BOOL;
	REUSE_WATER_SYSTEM.P402.thirdAdditionalStat AT %IX16.0 : BOOL;
	REUSE_WATER_SYSTEM.P402.dutyCommand AT %QX1.7 : BOOL;
	REUSE_WATER_SYSTEM.P402.standbyCommand AT %QX2.0 : BOOL;
	REUSE_WATER_SYSTEM.P402.thirdCommand AT %QX2.1 : BOOL;
	REUSE_WATER_SYSTEM.P401AB.dutyRemoteMode AT %IX16.1 : BOOL;
	REUSE_WATER_SYSTEM.P401AB.dutyOverload AT %IX16.2 : BOOL;
	REUSE_WATER_SYSTEM.P401AB.dutyIncomplete AT %IX16.3 : BOOL;
	REUSE_WATER_SYSTEM.P401AB.dutyStart AT %IX16.4 : BOOL;
	REUSE_WATER_SYSTEM.P401AB.standbyRemoteMode AT %IX16.5 : BOOL;
	REUSE_WATER_SYSTEM.P401AB.standbyOverload AT %IX16.6 : BOOL;
	REUSE_WATER_SYSTEM.P401AB.standbyIncomplete AT %IX16.7 : BOOL;
	REUSE_WATER_SYSTEM.P401AB.standbyStart AT %IX17.0 : BOOL;
	REUSE_WATER_SYSTEM.P401AB.thirdRemoteMode AT %IX17.1 : BOOL;
	REUSE_WATER_SYSTEM.P401AB.thirdOverload AT %IX17.2 : BOOL;
	REUSE_WATER_SYSTEM.P401AB.thirdStart AT %IX17.3 : BOOL;
	REUSE_WATER_SYSTEM.P401AB.thirdIncomplete AT %IX17.4 : BOOL;
	REUSE_WATER_SYSTEM.P401AB.standbyClose AT %IX17.5 : BOOL;
	REUSE_WATER_SYSTEM.P401AB.dutyClose AT %IX17.6 : BOOL;
	REUSE_WATER_SYSTEM.P401AB.thirdClose AT %IX17.7 : BOOL;
	REUSE_WATER_SYSTEM.P401AB.dutyAdditionalStat AT %IX18.0 : BOOL;
	REUSE_WATER_SYSTEM.P401AB.remoteAdditionalStat AT %IX18.1 : BOOL;
	REUSE_WATER_SYSTEM.P401AB.thirdAdditionalStat AT %IX18.2 : BOOL;
	REUSE_WATER_SYSTEM.P401AB.dutyCommand AT %QX2.2 : BOOL;
	REUSE_WATER_SYSTEM.P401AB.standbyCommand AT %QX2.3 : BOOL;
	REUSE_WATER_SYSTEM.P401AB.thirdCommand AT %QX2.4 : BOOL;
	REUSE_WATER_SYSTEM.P401CD.dutyRemoteMode AT %IX18.3 : BOOL;
	REUSE_WATER_SYSTEM.P401CD.dutyOverload AT %IX18.4 : BOOL;
	REUSE_WATER_SYSTEM.P401CD.dutyIncomplete AT %IX18.5 : BOOL;
	REUSE_WATER_SYSTEM.P401CD.dutyStart AT %IX18.6 : BOOL;
	REUSE_WATER_SYSTEM.P401CD.standbyRemoteMode AT %IX18.7 : BOOL;
	REUSE_WATER_SYSTEM.P401CD.standbyOverload AT %IX19.0 : BOOL;
	REUSE_WATER_SYSTEM.P401CD.standbyIncomplete AT %IX19.1 : BOOL;
	REUSE_WATER_SYSTEM.P401CD.standbyStart AT %IX19.2 : BOOL;
	REUSE_WATER_SYSTEM.P401CD.thirdRemoteMode AT %IX19.3 : BOOL;
	REUSE_WATER_SYSTEM.P401CD.thirdOverload AT %IX19.4 : BOOL;
	REUSE_WATER_SYSTEM.P401CD.thirdStart AT %IX19.5 : BOOL;
	REUSE_WATER_SYSTEM.P401CD.thirdIncomplete AT %IX19.6 : BOOL;
	REUSE_WATER_SYSTEM.P401CD.standbyClose AT %IX19.7 : BOOL;
	REUSE_WATER_SYSTEM.P401CD.dutyClose AT %IX20.0 : BOOL;
	REUSE_WATER_SYSTEM.P401CD.thirdClose AT %IX20.1 : BOOL;
	REUSE_WATER_SYSTEM.P401CD.dutyAdditionalStat AT %IX20.2 : BOOL;
	REUSE_WATER_SYSTEM.P401CD.remoteAdditionalStat AT %IX20.3 : BOOL;
	REUSE_WATER_SYSTEM.P401CD.thirdAdditionalStat AT %IX20.4 : BOOL;
	REUSE_WATER_SYSTEM.P401CD.dutyCommand AT %QX2.5 : BOOL;
	REUSE_WATER_SYSTEM.P401CD.standbyCommand AT %QX2.6 : BOOL;
	REUSE_WATER_SYSTEM.P401CD.thirdCommand AT %QX2.7 : BOOL;
	REUSE_WATER_SYSTEM.XV102.dutyRemoteMode AT %IX20.5 : BOOL;
	REUSE_WATER_SYSTEM.XV102.dutyOverload AT %IX20.6 : BOOL;
	REUSE_WATER_SYSTEM.XV102.dutyIncomplete AT %IX20.7 : BOOL;
	REUSE_WATER_SYSTEM.XV102.dutyStart AT %IX21.0 : BOOL;
	REUSE_WATER_SYSTEM.XV102.standbyRemoteMode AT %IX21.1 : BOOL;
	REUSE_WATER_SYSTEM.XV102.standbyOverload AT %IX21.2 : BOOL;
	REUSE_WATER_SYSTEM.XV102.standbyIncomplete AT %IX21.3 : BOOL;
	REUSE_WATER_SYSTEM.XV102.standbyStart AT %IX21.4 : BOOL;
	REUSE_WATER_SYSTEM.XV102.thirdRemoteMode AT %IX21.5 : BOOL;
	REUSE_WATER_SYSTEM.XV102.thirdOverload AT %IX21.6 : BOOL;
	REUSE_WATER_SYSTEM.XV102.thirdStart AT %IX21.7 : BOOL;
	REUSE_WATER_SYSTEM.XV102.thirdIncomplete AT %IX22.0 : BOOL;
	REUSE_WATER_SYSTEM.XV102.standbyClose AT %IX22.1 : BOOL;
	REUSE_WATER_SYSTEM.XV102.dutyClose AT %IX22.2 : BOOL;
	REUSE_WATER_SYSTEM.XV102.thirdClose AT %IX22.3 : BOOL;
	REUSE_WATER_SYSTEM.XV102.dutyAdditionalStat AT %IX22.4 : BOOL;
	REUSE_WATER_SYSTEM.XV102.remoteAdditionalStat AT %IX22.5 : BOOL;
	REUSE_WATER_SYSTEM.XV102.thirdAdditionalStat AT %IX22.6 : BOOL;
	REUSE_WATER_SYSTEM.XV102.dutyCommand AT %QX3.0 : BOOL;
	REUSE_WATER_SYSTEM.XV102.standbyCommand AT %QX3.1 : BOOL;
	REUSE_WATER_SYSTEM.XV102.thirdCommand AT %QX3.2 : BOOL;
	STREAM_INLET_MIXER_1.LSL101A.IN AT %IX22.7 : BOOL;
	STREAM_INLET_MIXER_1.LSS101A.IN AT %IX23.0 : BOOL;
	STREAM_INLET_MIXER_1.LSH101A.IN AT %IX23.1 : BOOL;
	STREAM_INLET_MIXER_1.LSD101A.IN AT %IX23.2 : BOOL;
	STREAM_INLET_MIXER_1.LSL100A.IN AT %IX23.3 : BOOL;
	STREAM_INLET_MIXER_1.LSHL100A.IN AT %IX23.4 : BOOL;
	STREAM_INLET_MIXER_1.P101A.dutyRemoteMode AT %IX23.5 : BOOL;
	STREAM_INLET_MIXER_1.P101A.dutyOverload AT %IX23.6 : BOOL;
	STREAM_INLET_MIXER_1.P101A.dutyIncomplete AT %IX23.7 : BOOL;
	STREAM_INLET_MIXER_1.P101A.dutyStart AT %IX24.0 : BOOL;
	STREAM_INLET_MIXER_1.P101A.standbyRemoteMode AT %IX24.1 : BOOL;
	STREAM_INLET_MIXER_1.P101A.standbyOverload AT %IX24.2 : BOOL;
	STREAM_INLET_MIXER_1.P101A.standbyIncomplete AT %IX24.3 : BOOL;
	STREAM_INLET_MIXER_1.P101A.standbyStart AT %IX24.4 : BOOL;
	STREAM_INLET_MIXER_1.P101A.thirdRemoteMode AT %IX24.5 : BOOL;
	STREAM_INLET_MIXER_1.P101A.thirdOverload AT %IX24.6 : BOOL;
	STREAM_INLET_MIXER_1.P101A.thirdStart AT %IX24.7 : BOOL;
	STREAM_INLET_MIXER_1.P101A.thirdIncomplete AT %IX25.0 : BOOL;
	STREAM_INLET_MIXER_1.P101A.standbyClose AT %IX25.1 : BOOL;
	STREAM_INLET_MIXER_1.P101A.dutyClose AT %IX25.2 : BOOL;
	STREAM_INLET_MIXER_1.P101A.thirdClose AT %IX25.3 : BOOL;
	STREAM_INLET_MIXER_1.P101A.dutyAdditionalStat AT %IX25.4 : BOOL;
	STREAM_INLET_MIXER_1.P101A.remoteAdditionalStat AT %IX25.5 : BOOL;
	STREAM_INLET_MIXER_1.P101A.thirdAdditionalStat AT %IX25.6 : BOOL;
	STREAM_INLET_MIXER_1.P101A.dutyCommand AT %QX3.3 : BOOL;
	STREAM_INLET_MIXER_1.P101A.standbyCommand AT %QX3.4 : BOOL;
	STREAM_INLET_MIXER_1.P101A.thirdCommand AT %QX3.5 : BOOL;
	STREAM_INLET_MIXER_1.M101A.dutyRemoteMode AT %IX25.7 : BOOL;
	STREAM_INLET_MIXER_1.M101A.dutyOverload AT %IX26.0 : BOOL;
	STREAM_INLET_MIXER_1.M101A.dutyIncomplete AT %IX26.1 : BOOL;
	STREAM_INLET_MIXER_1.M101A.dutyStart AT %IX26.2 : BOOL;
	STREAM_INLET_MIXER_1.M101A.standbyRemoteMode AT %IX26.3 : BOOL;
	STREAM_INLET_MIXER_1.M101A.standbyOverload AT %IX26.4 : BOOL;
	STREAM_INLET_MIXER_1.M101A.standbyIncomplete AT %IX26.5 : BOOL;
	STREAM_INLET_MIXER_1.M101A.standbyStart AT %IX26.6 : BOOL;
	STREAM_INLET_MIXER_1.M101A.thirdRemoteMode AT %IX26.7 : BOOL;
	STREAM_INLET_MIXER_1.M101A.thirdOverload AT %IX27.0 : BOOL;
	STREAM_INLET_MIXER_1.M101A.thirdStart AT %IX27.1 : BOOL;
	STREAM_INLET_MIXER_1.M101A.thirdIncomplete AT %IX27.2 : BOOL;
	STREAM_INLET_MIXER_1.M101A.standbyClose AT %IX27.3 : BOOL;
	STREAM_INLET_MIXER_1.M101A.dutyClose AT %IX27.4 : BOOL;
	STREAM_INLET_MIXER_1.M101A.thirdClose AT %IX27.5 : BOOL;
	STREAM_INLET_MIXER_1.M101A.dutyAdditionalStat AT %IX27.6 : BOOL;
	STREAM_INLET_MIXER_1.M101A.remoteAdditionalStat AT %IX27.7 : BOOL;
	STREAM_INLET_MIXER_1.M101A.thirdAdditionalStat AT %IX28.0 : BOOL;
	STREAM_INLET_MIXER_1.M101A.dutyCommand AT %QX3.6 : BOOL;
	STREAM_INLET_MIXER_1.M101A.standbyCommand AT %QX3.7 : BOOL;
	STREAM_INLET_MIXER_1.M101A.thirdCommand AT %QX4.0 : BOOL;
	STREAM_INLET_MIXER_2.LSL101B.IN AT %IX28.1 : BOOL;
	STREAM_INLET_MIXER_2.LSS101B.IN AT %IX28.2 : BOOL;
	STREAM_INLET_MIXER_2.LSH101B.IN AT %IX28.3 : BOOL;
	STREAM_INLET_MIXER_2.LSD101B.IN AT %IX28.4 : BOOL;
	STREAM_INLET_MIXER_2.LSL100B.IN AT %IX28.5 : BOOL;
	STREAM_INLET_MIXER_2.LSHL100B.IN AT %IX28.6 : BOOL;
	STREAM_INLET_MIXER_2.P101B.dutyRemoteMode AT %IX28.7 : BOOL;
	STREAM_INLET_MIXER_2.P101B.dutyOverload AT %IX29.0 : BOOL;
	STREAM_INLET_MIXER_2.P101B.dutyIncomplete AT %IX29.1 : BOOL;
	STREAM_INLET_MIXER_2.P101B.dutyStart AT %IX29.2 : BOOL;
	STREAM_INLET_MIXER_2.P101B.standbyRemoteMode AT %IX29.3 : BOOL;
	STREAM_INLET_MIXER_2.P101B.standbyOverload AT %IX29.4 : BOOL;
	STREAM_INLET_MIXER_2.P101B.standbyIncomplete AT %IX29.5 : BOOL;
	STREAM_INLET_MIXER_2.P101B.standbyStart AT %IX29.6 : BOOL;
	STREAM_INLET_MIXER_2.P101B.thirdRemoteMode AT %IX29.7 : BOOL;
	STREAM_INLET_MIXER_2.P101B.thirdOverload AT %IX30.0 : BOOL;
	STREAM_INLET_MIXER_2.P101B.thirdStart AT %IX30.1 : BOOL;
	STREAM_INLET_MIXER_2.P101B.thirdIncomplete AT %IX30.2 : BOOL;
	STREAM_INLET_MIXER_2.P101B.standbyClose AT %IX30.3 : BOOL;
	STREAM_INLET_MIXER_2.P101B.dutyClose AT %IX30.4 : BOOL;
	STREAM_INLET_MIXER_2.P101B.thirdClose AT %IX30.5 : BOOL;
	STREAM_INLET_MIXER_2.P101B.dutyAdditionalStat AT %IX30.6 : BOOL;
	STREAM_INLET_MIXER_2.P101B.remoteAdditionalStat AT %IX30.7 : BOOL;
	STREAM_INLET_MIXER_2.P101B.thirdAdditionalStat AT %IX31.0 : BOOL;
	STREAM_INLET_MIXER_2.P101B.dutyCommand AT %QX4.1 : BOOL;
	STREAM_INLET_MIXER_2.P101B.standbyCommand AT %QX4.2 : BOOL;
	STREAM_INLET_MIXER_2.P101B.thirdCommand AT %QX4.3 : BOOL;
	STREAM_INLET_MIXER_2.M101B.dutyRemoteMode AT %IX31.1 : BOOL;
	STREAM_INLET_MIXER_2.M101B.dutyOverload AT %IX31.2 : BOOL;
	STREAM_INLET_MIXER_2.M101B.dutyIncomplete AT %IX31.3 : BOOL;
	STREAM_INLET_MIXER_2.M101B.dutyStart AT %IX31.4 : BOOL;
	STREAM_INLET_MIXER_2.M101B.standbyRemoteMode AT %IX31.5 : BOOL;
	STREAM_INLET_MIXER_2.M101B.standbyOverload AT %IX31.6 : BOOL;
	STREAM_INLET_MIXER_2.M101B.standbyIncomplete AT %IX31.7 : BOOL;
	STREAM_INLET_MIXER_2.M101B.standbyStart AT %IX32.0 : BOOL;
	STREAM_INLET_MIXER_2.M101B.thirdRemoteMode AT %IX32.1 : BOOL;
	STREAM_INLET_MIXER_2.M101B.thirdOverload AT %IX32.2 : BOOL;
	STREAM_INLET_MIXER_2.M101B.thirdStart AT %IX32.3 : BOOL;
	STREAM_INLET_MIXER_2.M101B.thirdIncomplete AT %IX32.4 : BOOL;
	STREAM_INLET_MIXER_2.M101B.standbyClose AT %IX32.5 : BOOL;
	STREAM_INLET_MIXER_2.M101B.dutyClose AT %IX32.6 : BOOL;
	STREAM_INLET_MIXER_2.M101B.thirdClose AT %IX32.7 : BOOL;
	STREAM_INLET_MIXER_2.M101B.dutyAdditionalStat AT %IX33.0 : BOOL;
	STREAM_INLET_MIXER_2.M101B.remoteAdditionalStat AT %IX33.1 : BOOL;
	STREAM_INLET_MIXER_2.M101B.thirdAdditionalStat AT %IX33.2 : BOOL;
	STREAM_INLET_MIXER_2.M101B.dutyCommand AT %QX4.4 : BOOL;
	STREAM_INLET_MIXER_2.M101B.standbyCommand AT %QX4.5 : BOOL;
	STREAM_INLET_MIXER_2.M101B.thirdCommand AT %QX4.6 : BOOL;
	.LSH620.IN AT %IX70.7 : BOOL;
END_VAR

(* Data type *)
TYPE TEST :
STRUCT
	x : POINTER TO BOOL;
END_STRUCT
END_TYPE

(* Data type *)
TYPE TEST2 :
STRUCT
	X : BOOL;
END_STRUCT
END_TYPE

(* POU MAIN, ST *)
PROGRAM MAIN
VAR
END_VAR
STREAM_INLET_MIXER_1;
STREAM_INLET_MIXER_2;
INLET_SCREENING_OPERATION_2;
GRIT_REMOVAL_OPERATION;
SBR_TRANSFER_1;
SBR_TRANSFER_2;
REUSE_WATER_SYSTEM;
SBR_REACTOR_1;
SLUDGE_TANK;
END_PROGRAM

(* POU STREAM_INLET_MIXER_1, CFC *)
PROGRAM STREAM_INLET_MIXER_1
VAR
	LSL101A : inBlock;
	LSS101A : inBlock;
	LSH101A : inBlock;
	LSD101A : inBlock;

	LSL100A : inBlock;
	LSHL100A:inBlock;

	bEQPump: BOOL;
	bCriticalEQFloatHi: BOOL;
	bWarningFloatSensorLow: BOOL;
	bCriticalFloatSensorDry: BOOL;
	bEQMixer: BOOL;
	P101A: fb_equipment_with_linking;
	M101A: fb_equipment_with_linking;
END_VAR
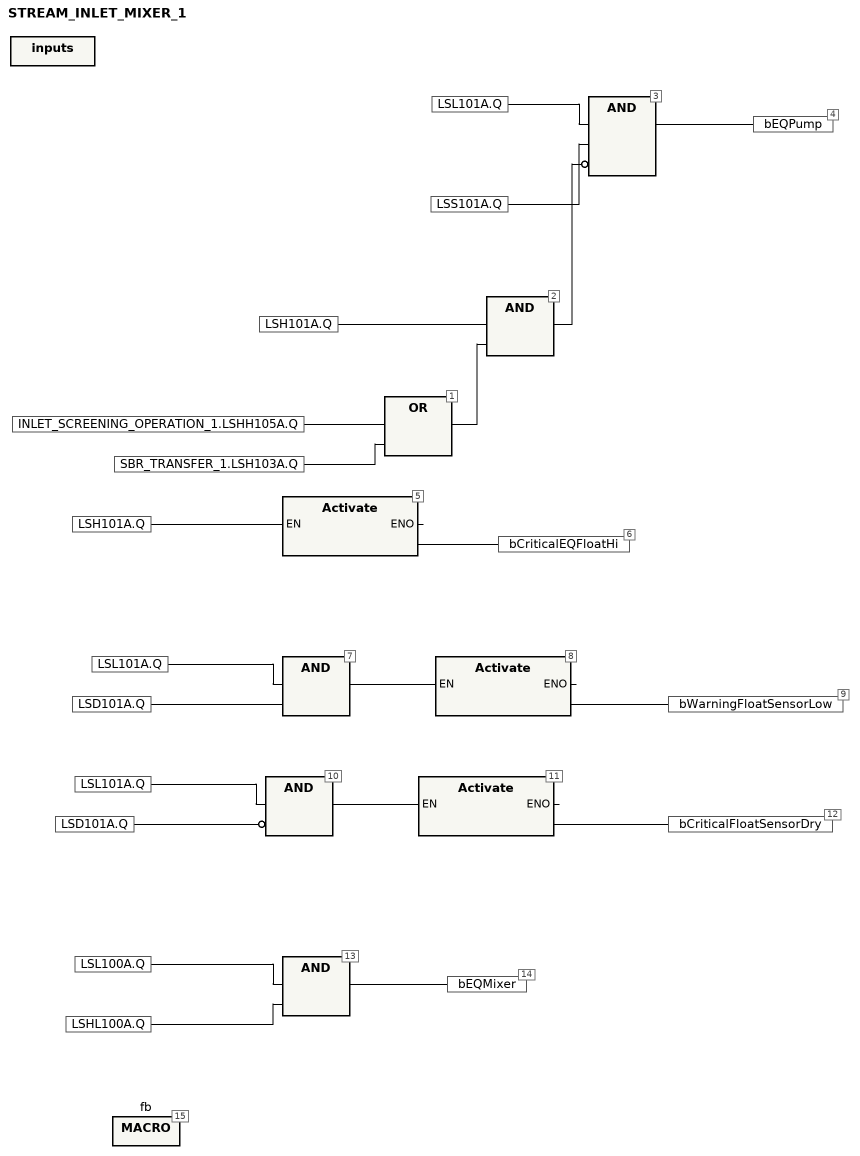
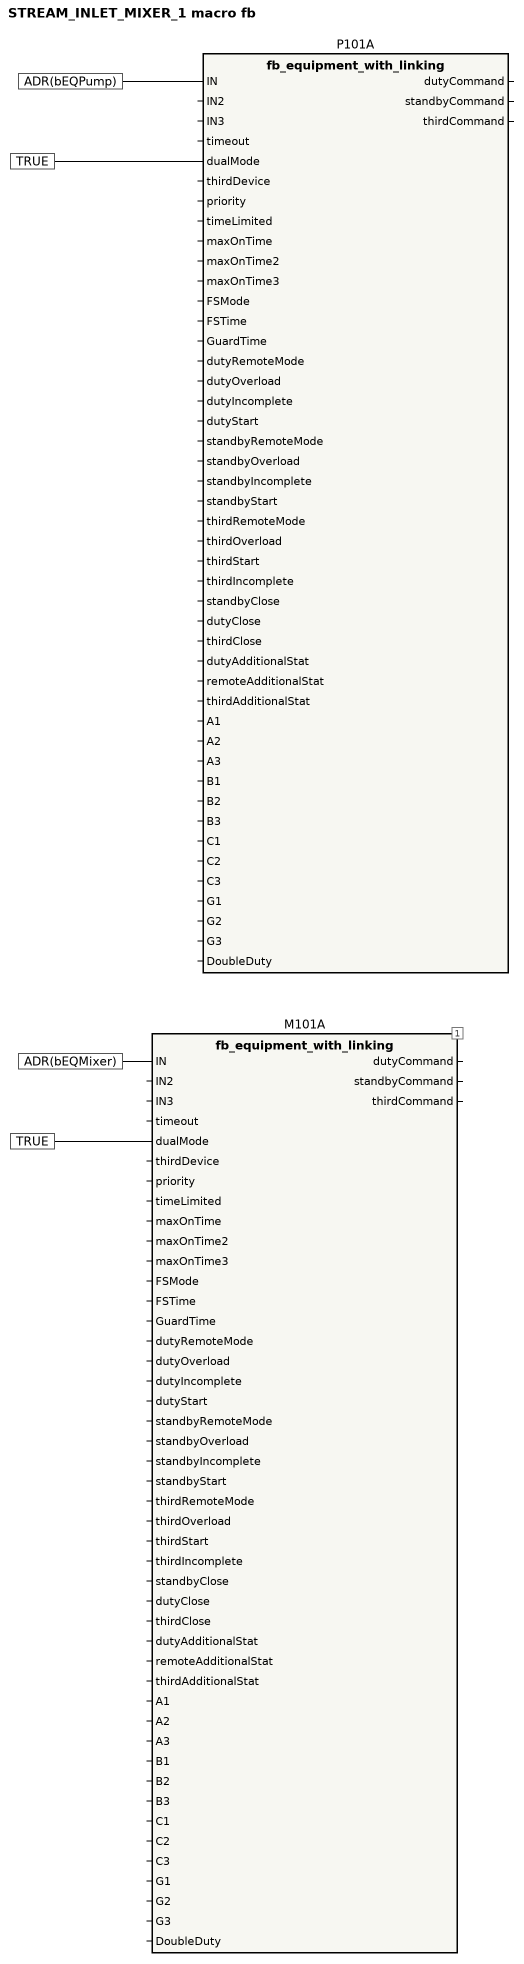
_CFC_ (* Continuous Function Chart, elements in execution order *)
#0 inputs()
#1 OR(INLET_SCREENING_OPERATION_1.LSHH105A.Q, SBR_TRANSFER_1.LSH103A.Q)
#2 AND(LSH101A.Q, #1)
#3 AND(LSL101A.Q, LSS101A.Q, NOT #2)
#4 bEQPump <= #3
#5 Activate(EN: LSH101A.Q)
#6 bCriticalEQFloatHi <= #5
#7 AND(LSL101A.Q, LSD101A.Q)
#8 Activate(EN: #7)
#9 bWarningFloatSensorLow <= #8
#10 AND(LSL101A.Q, NOT LSD101A.Q)
#11 Activate(EN: #10)
#12 bCriticalFloatSensorDry <= #11
#13 AND(LSL100A.Q, LSHL100A.Q)
#14 bEQMixer <= #13
#15 MACRO fb()
	#16 P101A:fb_equipment_with_linking(IN: ADR(bEQPump), IN2: -, IN3: -, timeout: -, dualMode: TRUE, thirdDevice: -, priority: -, timeLimited: -, maxOnTime: -, maxOnTime2: -, maxOnTime3: -, FSMode: -, FSTime: -, GuardTime: -, dutyRemoteMode: -, dutyOverload: -, dutyIncomplete: -, dutyStart: -, standbyRemoteMode: -, standbyOverload: -, standbyIncomplete: -, standbyStart: -, thirdRemoteMode: -, thirdOverload: -, thirdStart: -, thirdIncomplete: -, standbyClose: -, dutyClose: -, thirdClose: -, dutyAdditionalStat: -, remoteAdditionalStat: -, thirdAdditionalStat: -, A1: -, A2: -, A3: -, B1: -, B2: -, B3: -, C1: -, C2: -, C3: -, G1: -, G2: -, G3: -, DoubleDuty: -)
	#17 M101A:fb_equipment_with_linking(IN: ADR(bEQMixer), IN2: -, IN3: -, timeout: -, dualMode: TRUE, thirdDevice: -, priority: -, timeLimited: -, maxOnTime: -, maxOnTime2: -, maxOnTime3: -, FSMode: -, FSTime: -, GuardTime: -, dutyRemoteMode: -, dutyOverload: -, dutyIncomplete: -, dutyStart: -, standbyRemoteMode: -, standbyOverload: -, standbyIncomplete: -, standbyStart: -, thirdRemoteMode: -, thirdOverload: -, thirdStart: -, thirdIncomplete: -, standbyClose: -, dutyClose: -, thirdClose: -, dutyAdditionalStat: -, remoteAdditionalStat: -, thirdAdditionalStat: -, A1: -, A2: -, A3: -, B1: -, B2: -, B3: -, C1: -, C2: -, C3: -, G1: -, G2: -, G3: -, DoubleDuty: -)
END_MACRO
_END_CFC_
(* the same logic as Structured Text *)
inputs();
bEQPump := LSL101A.Q AND LSS101A.Q AND NOT (LSH101A.Q AND (INLET_SCREENING_OPERATION_1.LSHH105A.Q OR SBR_TRANSFER_1.LSH103A.Q));
IF LSH101A.Q THEN bCriticalEQFloatHi := Activate(); END_IF;
IF LSL101A.Q AND LSD101A.Q THEN bWarningFloatSensorLow := Activate(); END_IF;
IF LSL101A.Q AND NOT LSD101A.Q THEN bCriticalFloatSensorDry := Activate(); END_IF;
bEQMixer := LSL100A.Q AND LSHL100A.Q;
(* macro fb *)
P101A(IN := ADR(bEQPump), dualMode := TRUE);
M101A(IN := ADR(bEQMixer), dualMode := TRUE);
END_PROGRAM
ACTION inputs:
	LSL101A();
	LSS101A();
	LSH101A();
	LSD101A();

	LSL100A();
	LSHL100A();
END_ACTION

(* POU module/inBlock, ST *)
FUNCTION_BLOCK inBlock
VAR_INPUT
END_VAR
VAR_OUTPUT
	Q : BOOL;
END_VAR
VAR
	IN AT%I* : BOOL;
	ON:TON;
	OFF: TON;
END_VAR
IF NOT Q THEN
	OFF(IN:= FALSE, PT:=GlobalOFF );
	ON(IN:= IN, PT:=GlobalON );
	IF ON.Q THEN
		ON(IN:= FALSE, PT:=GlobalON );
		Q:=TRUE;
	END_IF
ELSE
	ON(IN:= FALSE, PT:=GlobalON );
	OFF(IN:= NOT IN, PT:=GlobalOFF );
	IF OFF.Q THEN
		OFF(IN:= FALSE, PT:=GlobalON );
		Q:=FALSE;
	END_IF
END_IF
END_FUNCTION_BLOCK

(* POU module/fb_equipment_with_linking, ST *)
FUNCTION_BLOCK fb_equipment_with_linking
VAR_INPUT
	IN							: POINTER TO BOOL;
	IN2							: POINTER TO BOOL;
	IN3							: POINTER TO BOOL;

	timeout						: TIME:= T#2s;
	dualMode					: BOOL:=TRUE;
	thirdDevice					: BOOL:= FALSE;
	priority						: BOOL := FALSE;
	timeLimited					: BOOL :=FALSE;
	maxOnTime					: TIME := T#10s;
	maxOnTime2					: TIME := T#10s;
	maxOnTime3					: TIME := T#10s;

	FSMode						: BOOL := FALSE;
	FSTime						: TIME := T#2m;
(*
	FSBothTime					: TIME := T#5m;
*)
	GuardTime					: TIME := T#5m;

	dutyRemoteMode				AT%I* : BOOL;
	dutyOverload					AT%I* : BOOL;
	dutyIncomplete				AT%I* : BOOL;
	dutyStart						AT%I* : BOOL;

	standbyRemoteMode			AT%I* : BOOL;
	standbyOverload				AT%I* : BOOL;
	standbyIncomplete			AT%I* : BOOL;
	standbyStart					AT%I* : BOOL;

	thirdRemoteMode				AT%I* : BOOL;
	thirdOverload					AT%I* : BOOL;
	thirdStart						AT%I* : BOOL;
	thirdIncomplete				AT%I* : BOOL;

	standbyClose					AT%I* : BOOL;
	dutyClose					AT%I* : BOOL;
	thirdClose					AT%I* : BOOL;

	dutyAdditionalStat				AT%I* : BOOL := TRUE;
	remoteAdditionalStat			AT%I* : BOOL := TRUE;
	thirdAdditionalStat				AT%I* : BOOL := TRUE;

	A1							: POINTER TO BOOL;
	A2							: POINTER TO BOOL;
	A3							: POINTER TO BOOL;
	B1							: POINTER TO BOOL;
	B2							: POINTER TO BOOL;
	B3							: POINTER TO BOOL;
	C1							: POINTER TO BOOL;
	C2							: POINTER TO BOOL;
	C3							: POINTER TO BOOL;
(*
	Q1							: POINTER TO BOOL;
	Q2							: POINTER TO BOOL;
	Q3							: POINTER TO BOOL;
*)
	G1							: POINTER TO BOOL;
	G2							: POINTER TO BOOL;
	G3							: POINTER TO BOOL;

	DoubleDuty: BOOL;
END_VAR
VAR_OUTPUT

	dutyCommand				AT%Q*: BOOL;
	standbyCommand				AT%Q*: BOOL;
	thirdCommand				AT%Q*: BOOL;
END_VAR
VAR




	warningDutyOverload			: BOOL;
	warningDutyFailed				: BOOL;
	warningDutyNotClose			: BOOL;
	warningDutyClose				: BOOL;
	warningStandbyOverload		: BOOL;
	warningStandbyFailed			: BOOL;
	warningStandbyNotClose		: BOOL;
	warningStandbyClose			: BOOL;
	warningThirdOverload			: BOOL;
	warningThirdFailed			: BOOL;
	warningThirdNotClose			: BOOL;
	warningThirdClose			: BOOL;

	criticalErrorStartingFailed		: BOOL;
	criticalDutyStopFailed			: BOOL;
	criticalStandbyStopFailed		: BOOL;
	criticalThirdStopFailed			: BOOL;

	duty							: INT;
	iStopDuty					: INT;
	state						: INT;
	third							: INT;
	iStopThird					: INT;
	iStopStandby					: INT;
	standby						: INT;
	startDuty						: BOOL;
	startStandby					: BOOL;
	stopStandby					: BOOL;
	stopDuty						: BOOL;
	dutyHalt						: BOOL;
	standbyHalt					: BOOL;
	stopThird					: BOOL;
	startThird					: BOOL;
	thirdHalt						: BOOL;

	dutyTimer					: TON;
	standbyTimer					: TON;
	stopStandbyTimer				: TON;
	stopDutyTimer				: TON;
	FSStopDuty					:TON;
	FSStopStandby				: TON;
	FSBothStop					: TON;
	OnTimer						: TON;
	StandbyOnTimer				: TON;
	thirdTimer					: TON;
	stopThirdTimer				: TON;
	GuardTONDuty				: TON;
	GuardTONStandby			: TON;
	GuardTONThird				: TON;

	ROnce5						: R_TRIG;
	ROnce10					: R_TRIG;
	ROnce20					: R_TRIG;
	SOnceDuty					: R_TRIG;
	SOnceStandby				: R_TRIG;
	SOnceFS					: R_TRIG;
	SOnceThird					: R_TRIG;
	DutyStopR					: R_TRIG;
	StandbyStopR				: R_TRIG;
	ThirdStopR					: R_TRIG;

	internalDummy: BOOL;
	dummyIN: BOOL;
	dummyIN2: BOOL;
	dummyIN3: BOOL;
END_VAR
VAR_IN_OUT
END_VAR
IF IN = 0 THEN
	IN := ADR(dummyIN);
END_IF

IF IN2 = 0 THEN
	IN2 := ADR(dummyIN2);
END_IF

IF IN3 = 0 THEN
	IN3 := ADR(dummyIN3);
END_IF

IF A1 = 0 THEN
	A1 := ADR(internalDummy);
END_IF
IF A2 = 0 THEN
	A2 := ADR(internalDummy);
END_IF
IF A3 = 0 THEN
	A3 := ADR(internalDummy);
END_IF

IF B1 = 0 THEN
	B1 := ADR(internalDummy);
END_IF
IF B2 = 0 THEN
	B2 := ADR(internalDummy);
END_IF
IF B3 = 0 THEN
	B3 := ADR(internalDummy);
END_IF

IF C1 = 0 THEN
	C1 := ADR(internalDummy);
END_IF
IF C2 = 0 THEN
	C2 := ADR(internalDummy);
END_IF
IF C3 = 0 THEN
	C3 := ADR(internalDummy);
END_IF

IF G1 = 0 THEN
	G1 := ADR(internalDummy);
END_IF
IF G2 = 0 THEN
	G2 := ADR(internalDummy);
END_IF
IF G3 = 0 THEN
	G3 := ADR(internalDummy);
END_IF


(*
IF warningDutyOverload = 0 THEN
	warningDutyOverload := ADR(internalDummy);
END_IF
IF warningDutyFailed = 0 THEN
	warningDutyFailed := ADR(internalDummy);
END_IF
IF warningDutyNotClose = 0 THEN
	warningDutyNotClose := ADR(internalDummy);
END_IF
IF warningDutyClose = 0 THEN
	warningDutyClose := ADR(internalDummy);
END_IF



IF warningStandbyOverload = 0 THEN
	warningStandbyOverload := ADR(internalDummy);
END_IF
IF warningStandbyFailed = 0 THEN
	warningStandbyFailed := ADR(internalDummy);
END_IF
IF warningStandbyNotClose = 0 THEN
	warningStandbyNotClose := ADR(internalDummy);
END_IF
IF warningStandbyClose = 0 THEN
	warningStandbyClose := ADR(internalDummy);
END_IF


IF warningThirdOverload = 0 THEN
	warningThirdOverload := ADR(internalDummy);
END_IF
IF warningThirdFailed = 0 THEN
	warningThirdFailed := ADR(internalDummy);
END_IF
IF warningThirdNotClose = 0 THEN
	warningThirdNotClose := ADR(internalDummy);
END_IF
IF warningThirdClose = 0 THEN
	warningThirdClose := ADR(internalDummy);
END_IF


IF criticalErrorStartingFailed = 0 THEN
	criticalErrorStartingFailed := ADR(internalDummy);
END_IF
IF criticalDutyStopFailed = 0 THEN
	criticalDutyStopFailed := ADR(internalDummy);
END_IF
IF criticalStandbyStopFailed = 0 THEN
	criticalStandbyStopFailed := ADR(internalDummy);
END_IF
IF criticalThirdStopFailed = 0 THEN
	criticalThirdStopFailed := ADR(internalDummy);
END_IF
*)
(*---------------------------------------------------------------------------------------------------------------------------*)

IF dualMode THEN

IF NOT IN^ THEN
	state := 0;
	stopDuty := TRUE;
	stopStandby := TRUE;

	startDuty:=FALSE;
	startStandby := FALSE;
	IF thirdDevice THEN
		stopThird :=TRUE;
		startThird := FALSE;
	END_IF
END_IF

ELSE

state := 0;
startDuty := IN^;
stopDuty := NOT IN^;

startStandby := IN2^;
stopStandby := NOT IN2^;

startThird := IN3^;
stopThird := NOT IN3^;

A1^:=  IN^;
A2^:= IN^;
A3^ := IN^;
B1^:=  IN2^;
B2^:= IN2^;
B3^ := IN2^;
C1^:=  IN3^;
C2^:= IN3^;
C3^ := IN3^;

END_IF

(*
IF NOT IN^ THEN
	state := 0;
	stopDuty := TRUE;
	stopStandby := TRUE;

	startDuty:=FALSE;
	startStandby := FALSE;
	IF thirdDevice THEN
		stopThird :=TRUE;
		startThird := FALSE;
	END_IF
ELSIF IN^ AND NOT dualMode THEN
	state := 0;
	stopDuty := FALSE;
	stopStandby := FALSE;

	startDuty:=TRUE;
	startStandby := TRUE;
	IF thirdDevice THEN
		stopThird :=FALSE;
		startThird := TRUE;
	END_IF

	A1^:= TRUE;
	A2^:=TRUE;
	A3^ :=TRUE;
	B1^:= TRUE;
	B2^:=TRUE;
	B3^ :=TRUE;
	C1^:= TRUE;
	C2^:=TRUE;
	C3^ :=TRUE;
END_IF
*)

(*-------------------------------------------------------------------------------------------------------------------------------------------*)

IF NOT DoubleDuty THEN

CASE state OF
0:
	state := 5;
5:
	IF NOT DutyHalt AND dutyStart THEN
		stopStandby := TRUE;
		stopThird:=TRUE;
	END_IF

	stopDuty := FALSE;
	startDuty := TRUE;
	IF timeLimited THEN
		OnTimer(IN:=TRUE,PT:=maxOnTime);
	ELSE
		OnTimer(IN:=FALSE,PT:=maxOnTime);
	END_IF
	IF dutyHalt  OR onTimer.Q THEN
		OnTimer(IN:=FALSE,PT:=maxOnTime);
		startDuty := FALSE;
		stopDuty := TRUE;
		state := 10;
	END_IF
10:
	IF NOT StandbyHalt AND standbyStart THEN
		stopDuty := TRUE;
		stopThird:=TRUE;
	END_IF

	stopStandby := FALSE;
	startStandby := TRUE;

	IF timeLimited THEN
		OnTimer(IN:=TRUE,PT:=maxOnTime2);
	ELSE
		OnTimer(IN:=FALSE,PT:=maxOnTime2);
	END_IF
	IF standbyHalt OR onTimer.Q THEN
		OnTimer(IN:=FALSE,PT:=maxOnTime2);
		startStandby := FALSE;
		stopStandby := TRUE;
		IF thirdDevice THEN
			IF priority THEN
				IF dutyIncomplete OR dutyOverload THEN
					state:= 20;
				ELSE
					dutyHalt := FALSE;
					standbyHalt := FALSE;
					state:=0;
				END_IF
			ELSE
				state:= 20;
			END_IF
		ELSE
			IF dutyIncomplete OR dutyOverload THEN
				CriticalErrorStartingFailed := TRUE;
			END_IF
			state:=0;
			dutyHalt := FALSE;
			standbyHalt := FALSE;
		END_IF
	END_IF
20:
	IF NOT thirdHalt AND thirdStart THEN
		stopStandby := TRUE;
		stopDuty:=TRUE;
	END_IF

	stopThird := FALSE;
	startThird := TRUE;
	IF timeLimited THEN
		OnTimer(IN:=TRUE,PT:=maxOnTime3);
	ELSE
		OnTimer(IN:=FALSE,PT:=maxOnTime3);
	END_IF
	IF thirdHalt OR OnTimer.Q THEN
		OnTimer(IN:=FALSE,PT:=maxOnTime3);
		startThird := FALSE;
		stopThird := TRUE;
		state := 0;
		IF  (dutyIncomplete OR dutyOverload)  AND (standbyIncomplete OR standbyOverload) THEN
				CriticalErrorStartingFailed := TRUE;
		END_IF
		dutyHalt := FALSE;
		standbyHalt := FALSE;
		thirdHalt := FALSE;
	END_IF
END_CASE

ELSE

thirdDevice := TRUE; (*third device must be enable when double duty*)
dualMode := TRUE; (*dual mode also must be true*)

CASE state OF
0:
	state := 5;
5:
	thirdHalt := FALSE;
	stopStandby := TRUE;
	startStandby := FALSE;

	stopDuty := FALSE;
	startDuty := TRUE;

	stopThird := FALSE;
	startThird := TRUE;

	IF dutyHalt  THEN
		state := 10;
	END_IF


	IF thirdHalt  THEN
		state := 20;
	END_IF
10:
	dutyHalt := FALSE;

	stopStandby := FALSE;
	startStandby := TRUE;

	stopDuty := TRUE;
	startDuty := FALSE;

	stopThird := FALSE;
	startThird := TRUE;

	IF standbyHalt THEN
		state:= 0;
	END_IF
20:
	thirdHalt := FALSE;

	stopStandby := FALSE;
	startStandby := TRUE;

	stopDuty := FALSE;
	startDuty := TRUE;

	stopThird := TRUE;
	startThird := FALSE;

	IF standbyHalt THEN
		state:= 0;
	END_IF
END_CASE


IF NOT(state = 0) AND  (dutyIncomplete OR dutyOverload)  AND (standbyIncomplete OR standbyOverload) AND (thirdIncomplete OR thirdOverload)  THEN
	CriticalErrorStartingFailed := TRUE;
END_IF
END_IF

(*-------------------------------------------------------------------------------------------------------------------------------------------*)

CASE duty OF
0:
	IF startDuty THEN
		duty := 5;
	END_IF
5:
	IF dutyRemoteMode AND dutyAdditionalStat THEN
		duty := 10;
	ELSE
		duty := 900;
	END_IF
10:
	IF dutyOverload THEN
		warningDutyOverload := TRUE;
		dutyHalt := TRUE;
		duty := 40;
	ELSE
		duty := 15;
	END_IF

15:
	duty := 20;
	dutyCommand := TRUE;
20:
	dutyTimer(IN:= TRUE, PT := timeout);
	IF dutyTimer.Q THEN
		dutyTimer(IN:=FALSE);
		duty := 30;
	END_IF
30:

		IF dutyIncomplete OR NOT dutyStart THEN
			warningDutyFailed := TRUE;
			dutyHalt := TRUE;
			IF  dutyClose THEN
				warningDutyClose := TRUE;
			END_IF
		END_IF
		duty := 40;
40:

	duty := 900;
900:
	duty := 0;
END_CASE

(*----------------------------------------------------------------------------------------------------------------------*)

CASE standby OF
0:
	IF startStandby THEN
		standby := 5;
	END_IF
5:
	IF standbyRemoteMode AND remoteAdditionalStat THEN
		standby := 10;
	ELSE
		standby := 900;
	END_IF
10:
	IF standbyOverload THEN
		warningStandbyOverload := TRUE;
		standbyHalt := TRUE;
		standby := 40;
	ELSE
		standby := 15;
	END_IF
15:
		standbyCommand := TRUE;
		standby := 20;
20:
	standbyTimer(IN:= TRUE, PT := timeout);
	IF standbyTimer.Q THEN
		standbyTimer(IN:=FALSE);
		standby := 30;
	END_IF
30:

		IF standbyIncomplete OR NOT standbyStart THEN
			warningStandbyFailed := TRUE;
			standbyHalt := TRUE;
			IF  standbyClose THEN
				warningStandbyClose := TRUE;
			END_IF
		END_IF
		standby := 40;
40:

	standby := 900;

900:
	standby := 0;
END_CASE

(*-------------------------------------------------------------------------------------------------------------------------------------------*)

CASE third OF
0:
	IF startThird THEN
		third := 5;
	END_IF
5:
	IF thirdRemoteMode AND thirdAdditionalStat THEN
		third := 10;
	ELSE
		third := 900;
	END_IF
10:
	IF thirdOverload THEN
		warningThirdOverload := TRUE;
		thirdHalt := TRUE;
		third := 40;
	ELSE
		third := 15;
	END_IF
15:
		thirdCommand := TRUE;
		third := 20;
20:
	thirdTimer(IN:= TRUE, PT := timeout);
	IF thirdTimer.Q THEN
		thirdTimer(IN:=FALSE);
		third := 30;
	END_IF
30:

		IF thirdIncomplete OR NOT thirdStart THEN
			warningThirdFailed := TRUE;
			thirdHalt := TRUE;
			IF thirdClose THEN
				warningThirdClose := TRUE;
			END_IF
		END_IF
		third := 40;
40:

	third := 900;

900:
	third := 0;
END_CASE

(*-------------------------------------------------------------------------------------------------------------------------------------------*)

ROnce5(CLK:=(state=5));
IF ROnce5.Q THEN
		A1^:= TRUE;
		A2^:=TRUE;
		A3^ :=TRUE;
END_IF

ROnce10(CLK:=(state=10));
IF ROnce10.Q THEN
		B1^:= TRUE;
		B2^:= TRUE;
		B3^:= TRUE;
END_IF

IF thirdDevice THEN
ROnce20(CLK:=(state=20));
IF ROnce20.Q THEN
		C1^:= TRUE;
		C2^:= TRUE;
		C3^:= TRUE;
END_IF
END_IF

(*-------------------------------------------------------------------------------------------------------------------------------------------*)
GuardTONDuty(IN:=dutyIncomplete OR dutyOverload OR NOT dutyStart, PT:= GuardTime);
IF GuardTONDuty.Q THEN
	G1^ := TRUE;
END_IF
GuardTONStandby(IN:=standbyIncomplete OR standbyOverload OR NOT standbyStart, PT:= GuardTime);
IF GuardTONStandby.Q THEN
	G2^ := TRUE;
END_IF

IF thirdDevice THEN
GuardTONThird(IN:=thirdIncomplete OR thirdOverload OR NOT thirdStart, PT:= GuardTime);
IF GuardTONThird.q THEN
	G3^ := TRUE;
END_IF
END_IF
(*-------------------------------------------------------------------------------------------------------------------------------------------*)
stopAction;
test();
END_FUNCTION_BLOCK
ACTION stopAction:
CASE iStopDuty OF
0:
	DutyStopR(CLK:=stopDuty);
	IF DutyStopR.Q THEN
		iStopDuty := 5;
	END_IF
5:
	IF FSMode THEN
		FSStopDuty(IN:=TRUE,PT:=FSTime);
		IF FSStopDuty.Q THEN
			iStopDuty := 10;
			FSStopDuty(IN:=FALSE,PT:=FSTime);
		END_IF
	ELSE
		iStopDuty:=10;
	END_IF
10:
	dutyCommand := FALSE;
	stopDutyTimer(IN:=TRUE, PT:=timeout);
		IF stopDutyTimer.Q THEN
			stopDutyTimer(IN:=FALSE);
			IF NOT dutyClose THEN
				IF dutyStart THEN
					criticalDutyStopFailed := TRUE;
				END_IF
				warningDutyNotClose := TRUE;
			END_IF
			iStopDuty := 0;
		END_IF
END_CASE

(*-------------------------------------------------------------------------------------------------------------------------------------------*)

CASE iStopStandby OF
0:
	StandbyStopR(CLK:=stopStandby);
	IF StandbyStopR.Q THEN
		iStopStandby := 5;
	END_IF
5:
	IF FSMode THEN
		FSStopStandby(IN:=TRUE,PT:=FSTime);
		IF FSStopStandby.Q THEN
			iStopStandby := 10;
			FSStopStandby(IN:=FALSE,PT:=FSTime);
		END_IF
	ELSE
		iStopStandby:=10;
	END_IF
10:
	standbyCommand := FALSE;
	stopStandbyTimer(IN:=TRUE, PT:=timeout);
		IF stopStandbyTimer.Q THEN
			stopStandbyTimer(IN:=FALSE);
			IF NOT standbyClose THEN
				IF standbyStart THEN
					criticalStandbyStopFailed := TRUE;
				END_IF
					warningStandbyNotClose := TRUE;
			END_IF
			iStopStandby := 0;
		END_IF
END_CASE


(*-------------------------------------------------------------------------------------------------------------------------------------------*)

CASE iStopThird OF
0:
	ThirdStopR(CLK:=stopThird);
	IF ThirdStopR.Q THEN
		iStopThird := 10;
	END_IF
10:
	thirdCommand := FALSE;
	stopThirdTimer(IN:=TRUE, PT:=timeout);
		IF stopThirdTimer.Q THEN
			stopThirdTimer(IN:=FALSE);
			IF NOT thirdClose THEN
				IF thirdStart THEN
					criticalThirdStopFailed := TRUE;
				END_IF
				warningThirdNotClose := TRUE;
			END_IF
			iStopThird := 0;
		END_IF
END_CASE


(*-------------------------------------------------------------------------------------------------------------------------------------------*)

SOnceDuty(CLK:=(iStopDuty = 10));
IF SOnceDuty.Q THEN
		A1^:=FALSE;
		A2^:=FALSE;
		A3^:=FALSE;
END_IF


SOnceStandby(CLK:=(iStopStandby = 10));
IF SOnceStandby.Q THEN
		B1^:=FALSE;
		B2^:=FALSE;
		B3^:=FALSE;
END_IF

IF thirdDevice THEN
SOnceThird(CLK:=(iStopThird = 10));
IF SOnceThird.Q THEN
		C1^:=FALSE;
		C2^:=FALSE;
		C3^:=FALSE;
END_IF
END_IF


(*-------------------------------------------------------------------------------------------------------------------------------------------*)

(*
IF FSMode THEN

FSBothStop(IN:=NOT dutyCommand AND NOT standbyCommand,PT:=FSBothTime);
SOnceFS(CLK:=FSBothStop.Q);
IF SOnceFS.Q THEN
	FSBothStop(IN:=FALSE,PT:=FSBothTime);
	Q1^ := TRUE;
	Q2^ := TRUE;
	Q3^:=TRUE;
END_IF

END_IF
*)
END_ACTION
ACTION test:
dutyStart := dutyCommand;
standbyStart := standbyCommand;
thirdStart:=thirdCommand;
END_ACTION

(* POU INLET_SCREENING_OPERATION_1, CFC *)
PROGRAM INLET_SCREENING_OPERATION_1
VAR
	bTest: BOOL;
	bTestReault: BOOL;

	LSH105A : inBlock;
	LSHH105A: inBlock;
	bPenstockDual: BOOL;
	Timer1: TON;
	bWarningStreamLineOverflow: BOOL;
	bFineScreen: BOOL;
	F101A: fb_equipment_with_linking;
	XV101A1 : fb_equipment_with_linking;
	StopTimer: TON;
	bScrewConveyor: BOOL;
	bScreenCompactor: BOOL;
	bWaterSprayScreenDuty: BOOL;
	bWaterSprayScreenStandby: BOOL;
	bPenstockDuty: BOOL;
	bPenstockStandby: BOOL;
	XV101A2: fb_equipment_with_linking;
	timerCompactor: TON;
	bFineScreenDual: BOOL;
	PS101A: fb_equipment_with_linking;
	bContinuousWaterSpray: BOOL;
	C102A: fb_equipment_with_linking;
	C101A: fb_equipment_with_linking;
	XV102A: fb_equipment_with_linking;
END_VAR
VAR (* helpers for the ST form of the networks *)
	_en57 : BOOL;
	_t57 : BOOL;
	_en85 : BOOL;
	_t85 : BOOL;
END_VAR
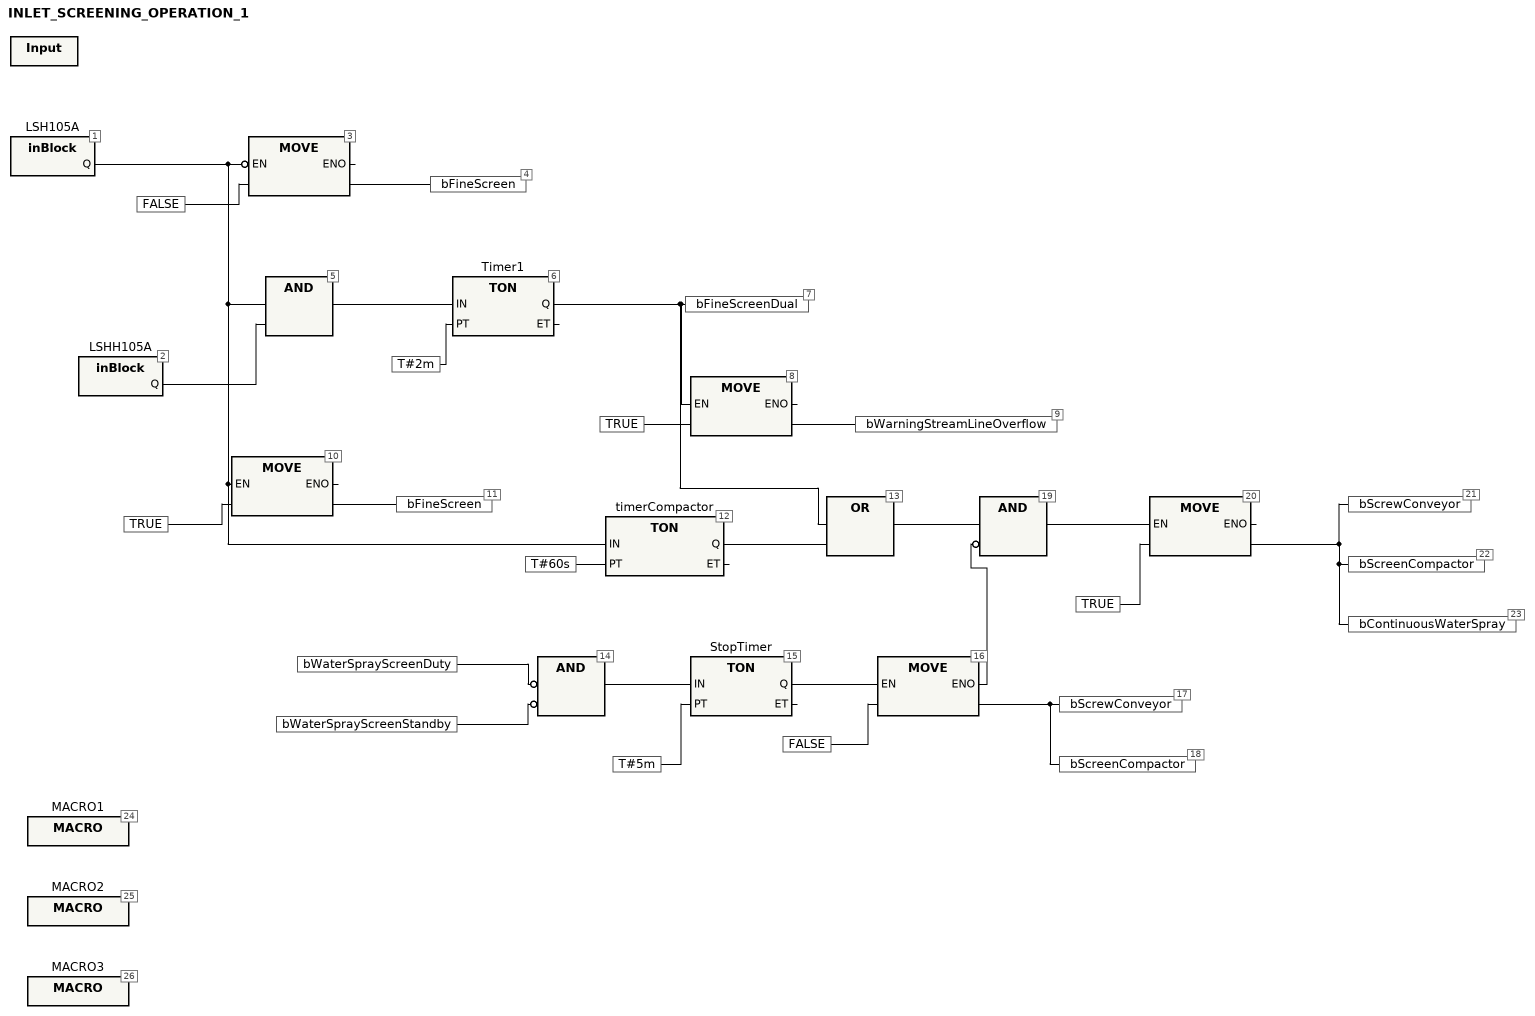
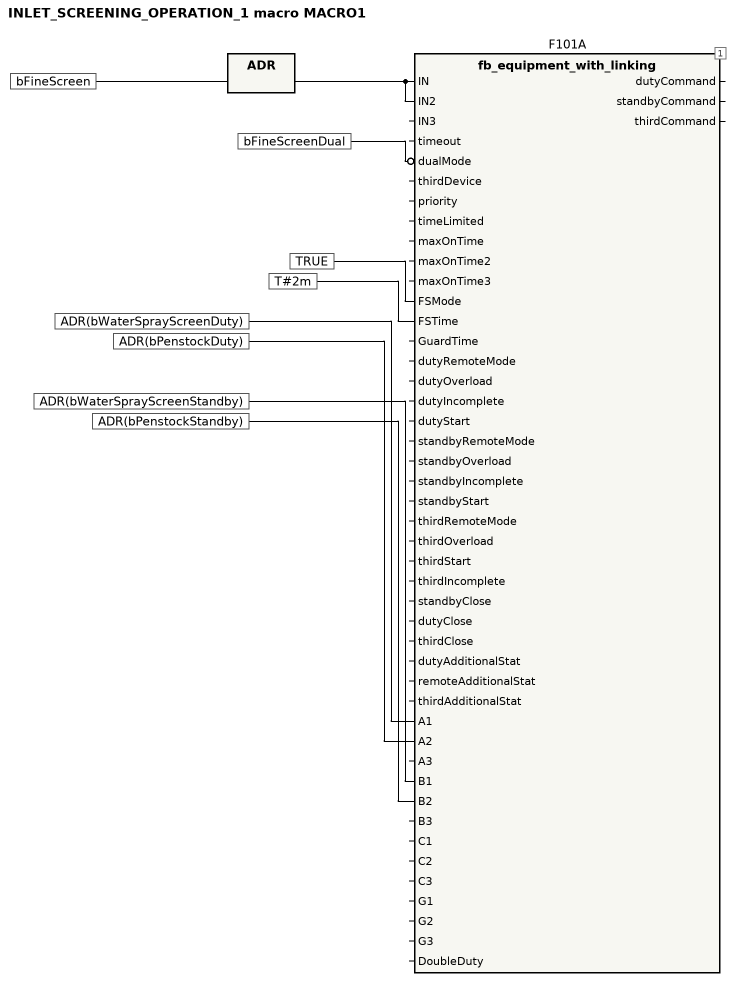
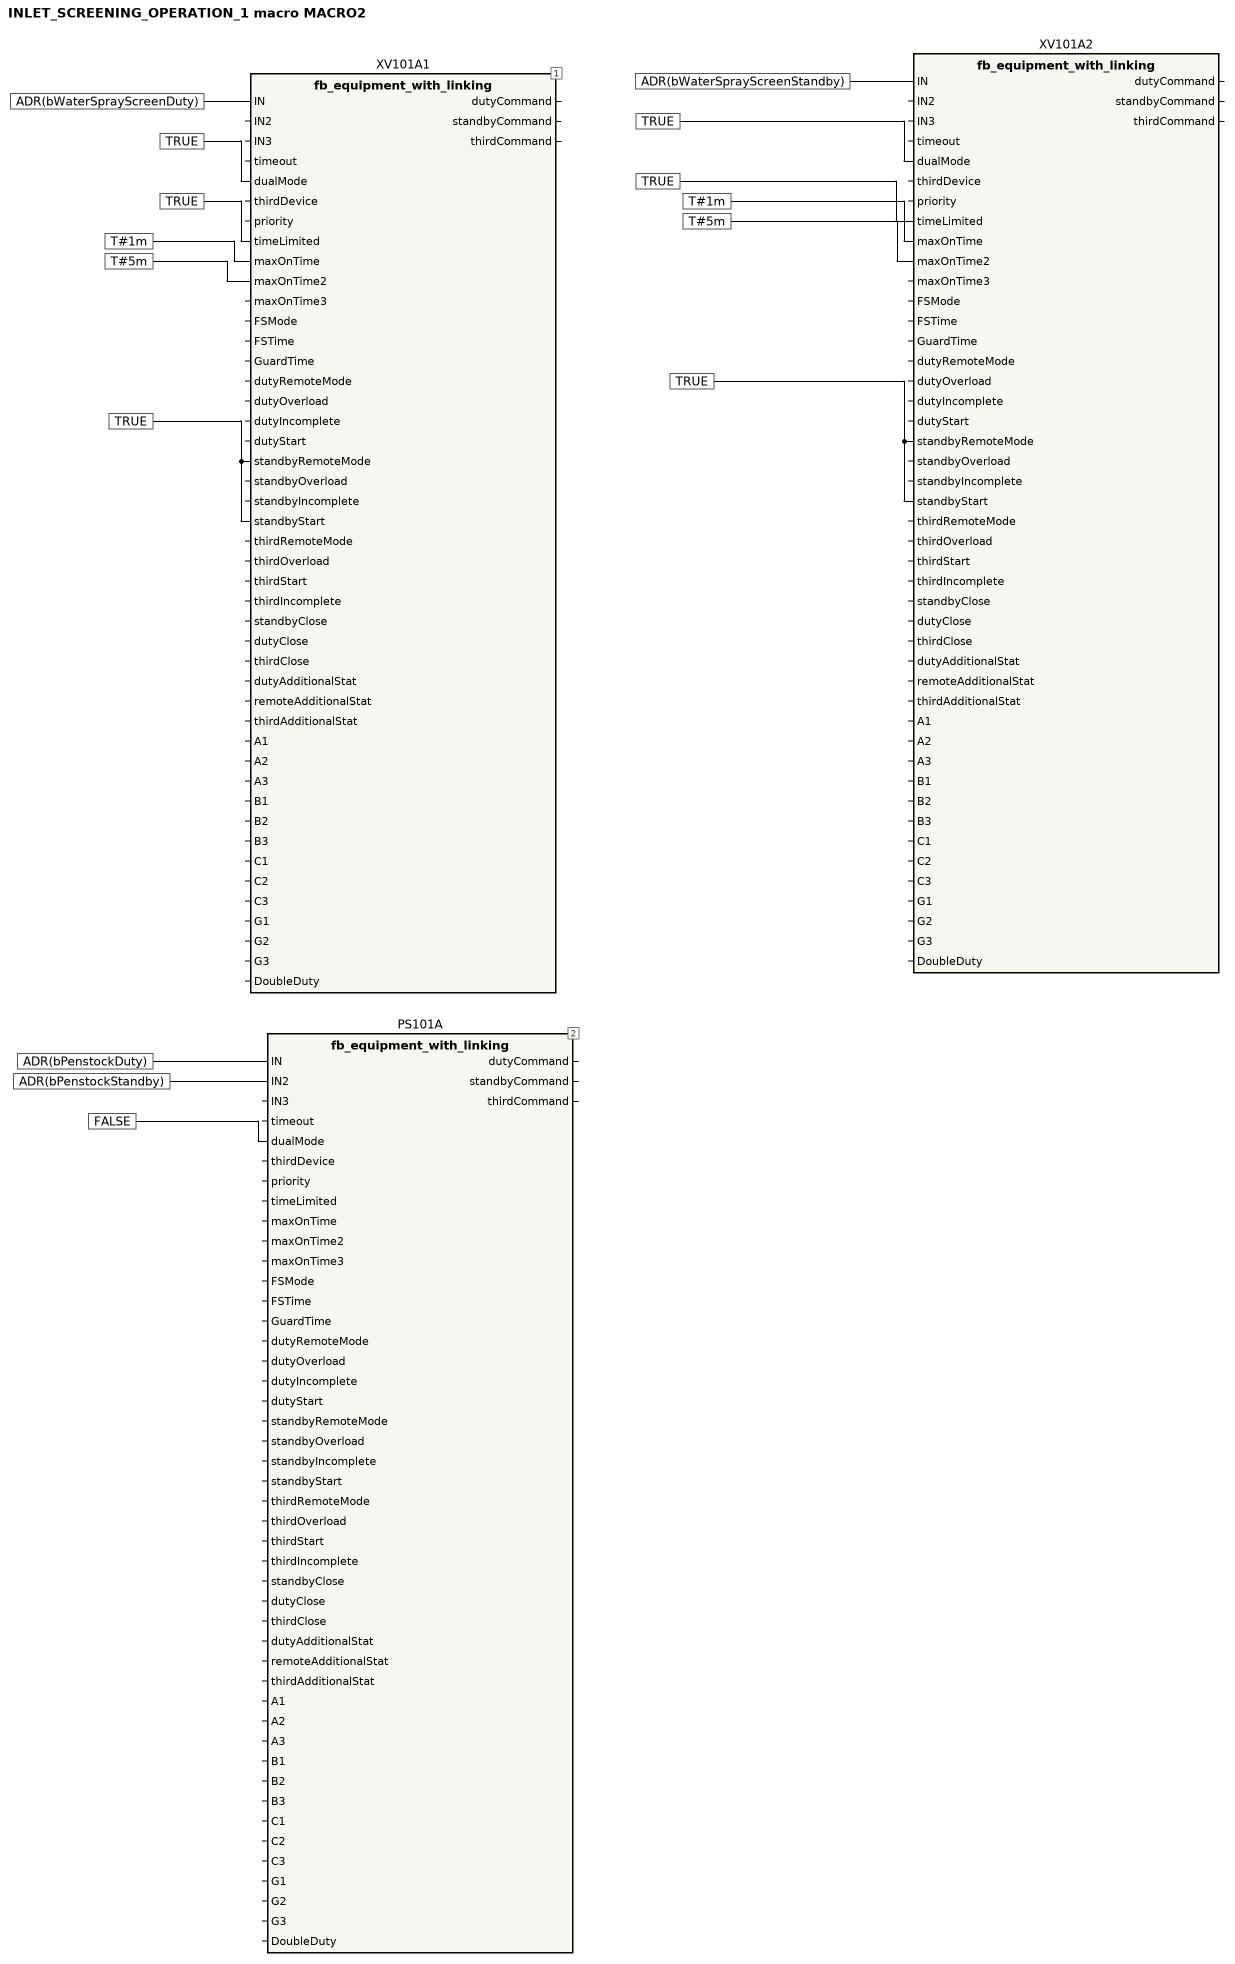
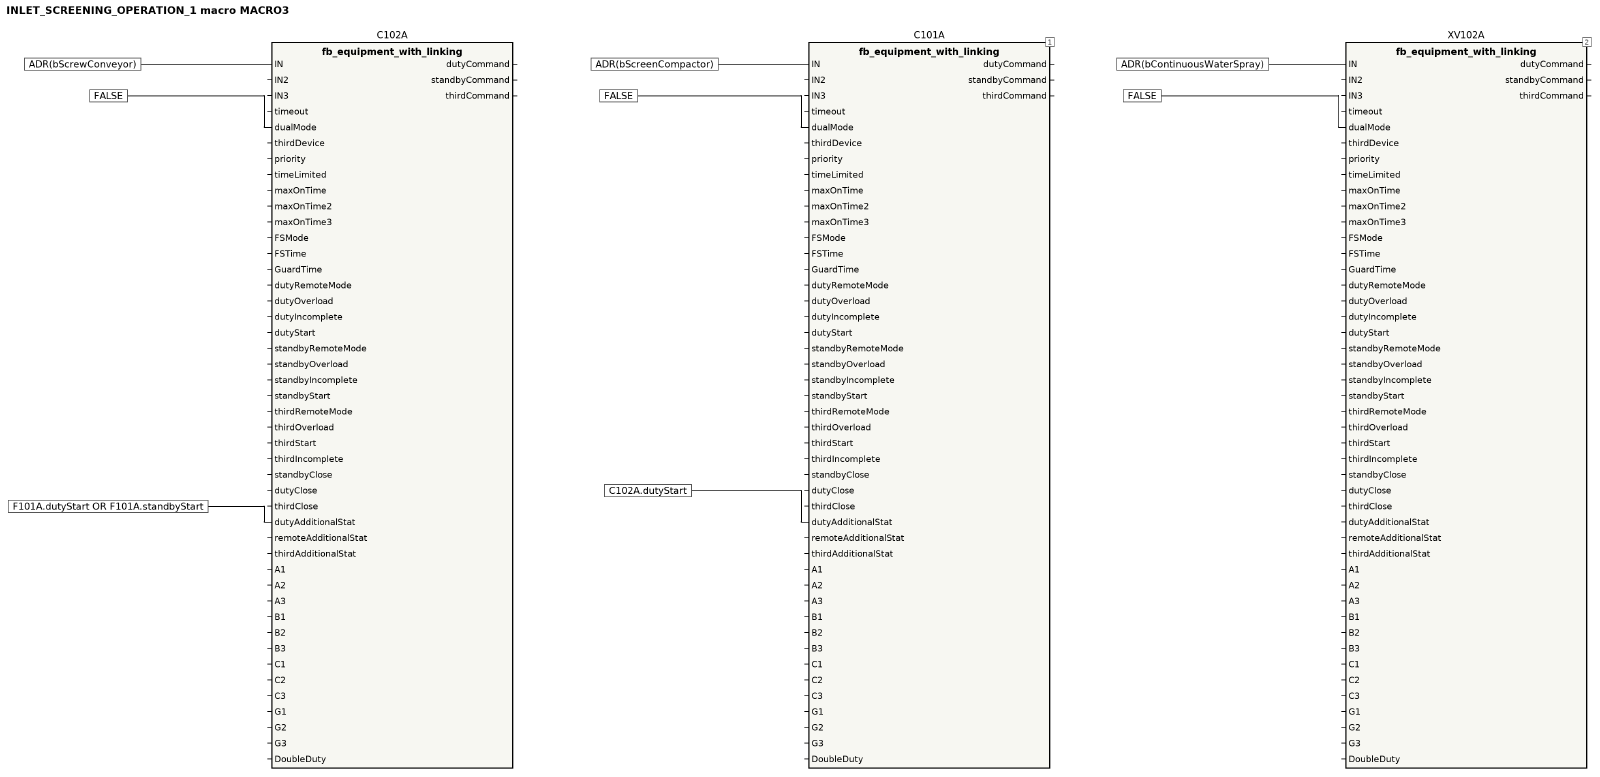
_CFC_ (* Continuous Function Chart, elements in execution order *)
#0 Input()
#1 LSH105A:inBlock()
#2 LSHH105A:inBlock()
#3 MOVE(EN: NOT #1.Q, FALSE)
#4 bFineScreen <= #3
#5 AND(#1.Q, #2.Q)
#6 Timer1:TON(IN: #5, PT: T#2m)
#7 bFineScreenDual <= #6.Q
#8 MOVE(EN: #6.Q, TRUE)
#9 bWarningStreamLineOverflow <= #8
#10 MOVE(EN: #1.Q, TRUE)
#11 bFineScreen <= #10
#12 timerCompactor:TON(IN: #1.Q, PT: T#60s)
#13 OR(#6.Q, #12.Q)
#14 AND(NOT bWaterSprayScreenDuty, NOT bWaterSprayScreenStandby)
#15 StopTimer:TON(IN: #14, PT: T#5m)
#16 MOVE(EN: #15.Q, FALSE)
#17 bScrewConveyor <= #16
#18 bScreenCompactor <= #16
#19 AND(#13, NOT #16.ENO)
#20 MOVE(EN: #19, TRUE)
#21 bScrewConveyor <= #20
#22 bScreenCompactor <= #20
#23 bContinuousWaterSpray <= #20
#24 MACRO MACRO1()
	#25 ADR(bFineScreen)
	#26 F101A:fb_equipment_with_linking(IN: #25, IN2: #25, IN3: -, timeout: -, dualMode: NOT bFineScreenDual, thirdDevice: -, priority: -, timeLimited: -, maxOnTime: -, maxOnTime2: -, maxOnTime3: -, FSMode: TRUE, FSTime: T#2m, GuardTime: -, dutyRemoteMode: -, dutyOverload: -, dutyIncomplete: -, dutyStart: -, standbyRemoteMode: -, standbyOverload: -, standbyIncomplete: -, standbyStart: -, thirdRemoteMode: -, thirdOverload: -, thirdStart: -, thirdIncomplete: -, standbyClose: -, dutyClose: -, thirdClose: -, dutyAdditionalStat: -, remoteAdditionalStat: -, thirdAdditionalStat: -, A1: ADR(bWaterSprayScreenDuty), A2: ADR(bPenstockDuty), A3: -, B1: ADR(bWaterSprayScreenStandby), B2: ADR(bPenstockStandby), B3: -, C1: -, C2: -, C3: -, G1: -, G2: -, G3: -, DoubleDuty: -)
END_MACRO
#27 MACRO MACRO2()
	#28 XV101A2:fb_equipment_with_linking(IN: ADR(bWaterSprayScreenStandby), IN2: -, IN3: -, timeout: -, dualMode: TRUE, thirdDevice: -, priority: -, timeLimited: TRUE, maxOnTime: T#1m, maxOnTime2: T#5m, maxOnTime3: -, FSMode: -, FSTime: -, GuardTime: -, dutyRemoteMode: -, dutyOverload: -, dutyIncomplete: -, dutyStart: -, standbyRemoteMode: TRUE, standbyOverload: -, standbyIncomplete: -, standbyStart: TRUE, thirdRemoteMode: -, thirdOverload: -, thirdStart: -, thirdIncomplete: -, standbyClose: -, dutyClose: -, thirdClose: -, dutyAdditionalStat: -, remoteAdditionalStat: -, thirdAdditionalStat: -, A1: -, A2: -, A3: -, B1: -, B2: -, B3: -, C1: -, C2: -, C3: -, G1: -, G2: -, G3: -, DoubleDuty: -)
	#29 XV101A1:fb_equipment_with_linking(IN: ADR(bWaterSprayScreenDuty), IN2: -, IN3: -, timeout: -, dualMode: TRUE, thirdDevice: -, priority: -, timeLimited: TRUE, maxOnTime: T#1m, maxOnTime2: T#5m, maxOnTime3: -, FSMode: -, FSTime: -, GuardTime: -, dutyRemoteMode: -, dutyOverload: -, dutyIncomplete: -, dutyStart: -, standbyRemoteMode: TRUE, standbyOverload: -, standbyIncomplete: -, standbyStart: TRUE, thirdRemoteMode: -, thirdOverload: -, thirdStart: -, thirdIncomplete: -, standbyClose: -, dutyClose: -, thirdClose: -, dutyAdditionalStat: -, remoteAdditionalStat: -, thirdAdditionalStat: -, A1: -, A2: -, A3: -, B1: -, B2: -, B3: -, C1: -, C2: -, C3: -, G1: -, G2: -, G3: -, DoubleDuty: -)
	#30 PS101A:fb_equipment_with_linking(IN: ADR(bPenstockDuty), IN2: ADR(bPenstockStandby), IN3: -, timeout: -, dualMode: FALSE, thirdDevice: -, priority: -, timeLimited: -, maxOnTime: -, maxOnTime2: -, maxOnTime3: -, FSMode: -, FSTime: -, GuardTime: -, dutyRemoteMode: -, dutyOverload: -, dutyIncomplete: -, dutyStart: -, standbyRemoteMode: -, standbyOverload: -, standbyIncomplete: -, standbyStart: -, thirdRemoteMode: -, thirdOverload: -, thirdStart: -, thirdIncomplete: -, standbyClose: -, dutyClose: -, thirdClose: -, dutyAdditionalStat: -, remoteAdditionalStat: -, thirdAdditionalStat: -, A1: -, A2: -, A3: -, B1: -, B2: -, B3: -, C1: -, C2: -, C3: -, G1: -, G2: -, G3: -, DoubleDuty: -)
END_MACRO
#31 MACRO MACRO3()
	#32 C102A:fb_equipment_with_linking(IN: ADR(bScrewConveyor), IN2: -, IN3: -, timeout: -, dualMode: FALSE, thirdDevice: -, priority: -, timeLimited: -, maxOnTime: -, maxOnTime2: -, maxOnTime3: -, FSMode: -, FSTime: -, GuardTime: -, dutyRemoteMode: -, dutyOverload: -, dutyIncomplete: -, dutyStart: -, standbyRemoteMode: -, standbyOverload: -, standbyIncomplete: -, standbyStart: -, thirdRemoteMode: -, thirdOverload: -, thirdStart: -, thirdIncomplete: -, standbyClose: -, dutyClose: -, thirdClose: -, dutyAdditionalStat: F101A.dutyStart OR F101A.standbyStart, remoteAdditionalStat: -, thirdAdditionalStat: -, A1: -, A2: -, A3: -, B1: -, B2: -, B3: -, C1: -, C2: -, C3: -, G1: -, G2: -, G3: -, DoubleDuty: -)
	#33 C101A:fb_equipment_with_linking(IN: ADR(bScreenCompactor), IN2: -, IN3: -, timeout: -, dualMode: FALSE, thirdDevice: -, priority: -, timeLimited: -, maxOnTime: -, maxOnTime2: -, maxOnTime3: -, FSMode: -, FSTime: -, GuardTime: -, dutyRemoteMode: -, dutyOverload: -, dutyIncomplete: -, dutyStart: -, standbyRemoteMode: -, standbyOverload: -, standbyIncomplete: -, standbyStart: -, thirdRemoteMode: -, thirdOverload: -, thirdStart: -, thirdIncomplete: -, standbyClose: -, dutyClose: -, thirdClose: -, dutyAdditionalStat: C102A.dutyStart, remoteAdditionalStat: -, thirdAdditionalStat: -, A1: -, A2: -, A3: -, B1: -, B2: -, B3: -, C1: -, C2: -, C3: -, G1: -, G2: -, G3: -, DoubleDuty: -)
	#34 XV102A:fb_equipment_with_linking(IN: ADR(bContinuousWaterSpray), IN2: -, IN3: -, timeout: -, dualMode: FALSE, thirdDevice: -, priority: -, timeLimited: -, maxOnTime: -, maxOnTime2: -, maxOnTime3: -, FSMode: -, FSTime: -, GuardTime: -, dutyRemoteMode: -, dutyOverload: -, dutyIncomplete: -, dutyStart: -, standbyRemoteMode: -, standbyOverload: -, standbyIncomplete: -, standbyStart: -, thirdRemoteMode: -, thirdOverload: -, thirdStart: -, thirdIncomplete: -, standbyClose: -, dutyClose: -, thirdClose: -, dutyAdditionalStat: -, remoteAdditionalStat: -, thirdAdditionalStat: -, A1: -, A2: -, A3: -, B1: -, B2: -, B3: -, C1: -, C2: -, C3: -, G1: -, G2: -, G3: -, DoubleDuty: -)
END_MACRO
_END_CFC_
(* the same logic as Structured Text *)
Input();
LSH105A();
LSHH105A();
IF NOT LSH105A.Q THEN bFineScreen := FALSE; END_IF;
Timer1(IN := LSH105A.Q AND LSHH105A.Q, PT := T#2m);
bFineScreenDual := Timer1.Q;
IF Timer1.Q THEN bWarningStreamLineOverflow := TRUE; END_IF;
IF LSH105A.Q THEN bFineScreen := TRUE; END_IF;
timerCompactor(IN := LSH105A.Q, PT := T#60s);
StopTimer(IN := NOT bWaterSprayScreenDuty AND NOT bWaterSprayScreenStandby, PT := T#5m);
_en57 := StopTimer.Q;
IF _en57 THEN _t57 := FALSE; END_IF;
IF _en57 THEN bScrewConveyor := _t57; END_IF;
IF _en57 THEN bScreenCompactor := _t57; END_IF;
_en85 := (Timer1.Q OR timerCompactor.Q) AND NOT _en57;
IF _en85 THEN _t85 := TRUE; END_IF;
IF _en85 THEN bScrewConveyor := _t85; END_IF;
IF _en85 THEN bScreenCompactor := _t85; END_IF;
IF _en85 THEN bContinuousWaterSpray := _t85; END_IF;
(* macro MACRO1 *)
F101A(IN := ADR(bFineScreen), IN2 := ADR(bFineScreen), dualMode := NOT bFineScreenDual, FSMode := TRUE, FSTime := T#2m, A1 := ADR(bWaterSprayScreenDuty), A2 := ADR(bPenstockDuty), B1 := ADR(bWaterSprayScreenStandby), B2 := ADR(bPenstockStandby));
(* macro MACRO2 *)
XV101A2(IN := ADR(bWaterSprayScreenStandby), dualMode := TRUE, timeLimited := TRUE, maxOnTime := T#1m, maxOnTime2 := T#5m, standbyRemoteMode := TRUE, standbyStart := TRUE);
XV101A1(IN := ADR(bWaterSprayScreenDuty), dualMode := TRUE, timeLimited := TRUE, maxOnTime := T#1m, maxOnTime2 := T#5m, standbyRemoteMode := TRUE, standbyStart := TRUE);
PS101A(IN := ADR(bPenstockDuty), IN2 := ADR(bPenstockStandby), dualMode := FALSE);
(* macro MACRO3 *)
C102A(IN := ADR(bScrewConveyor), dualMode := FALSE, dutyAdditionalStat := F101A.dutyStart OR F101A.standbyStart);
C101A(IN := ADR(bScreenCompactor), dualMode := FALSE, dutyAdditionalStat := C102A.dutyStart);
XV102A(IN := ADR(bContinuousWaterSpray), dualMode := FALSE);
END_PROGRAM
ACTION Input:
LSH105A( );
LSHH105A( );
END_ACTION

(* POU SBR_TRANSFER_1, CFC *)
PROGRAM SBR_TRANSFER_1
VAR
	LSL103A : inBlock;
	LSS103A : inBlock;
	LSH103A : inBlock;
	LSD103A : inBlock;

	bSBRTransfer:BOOL;


	bWarningSBRDry: BOOL;
	bCriticalSBRDry: BOOL;
	bCriticalSBRHi: BOOL;
	P102A: fb_equipment_with_linking;
END_VAR
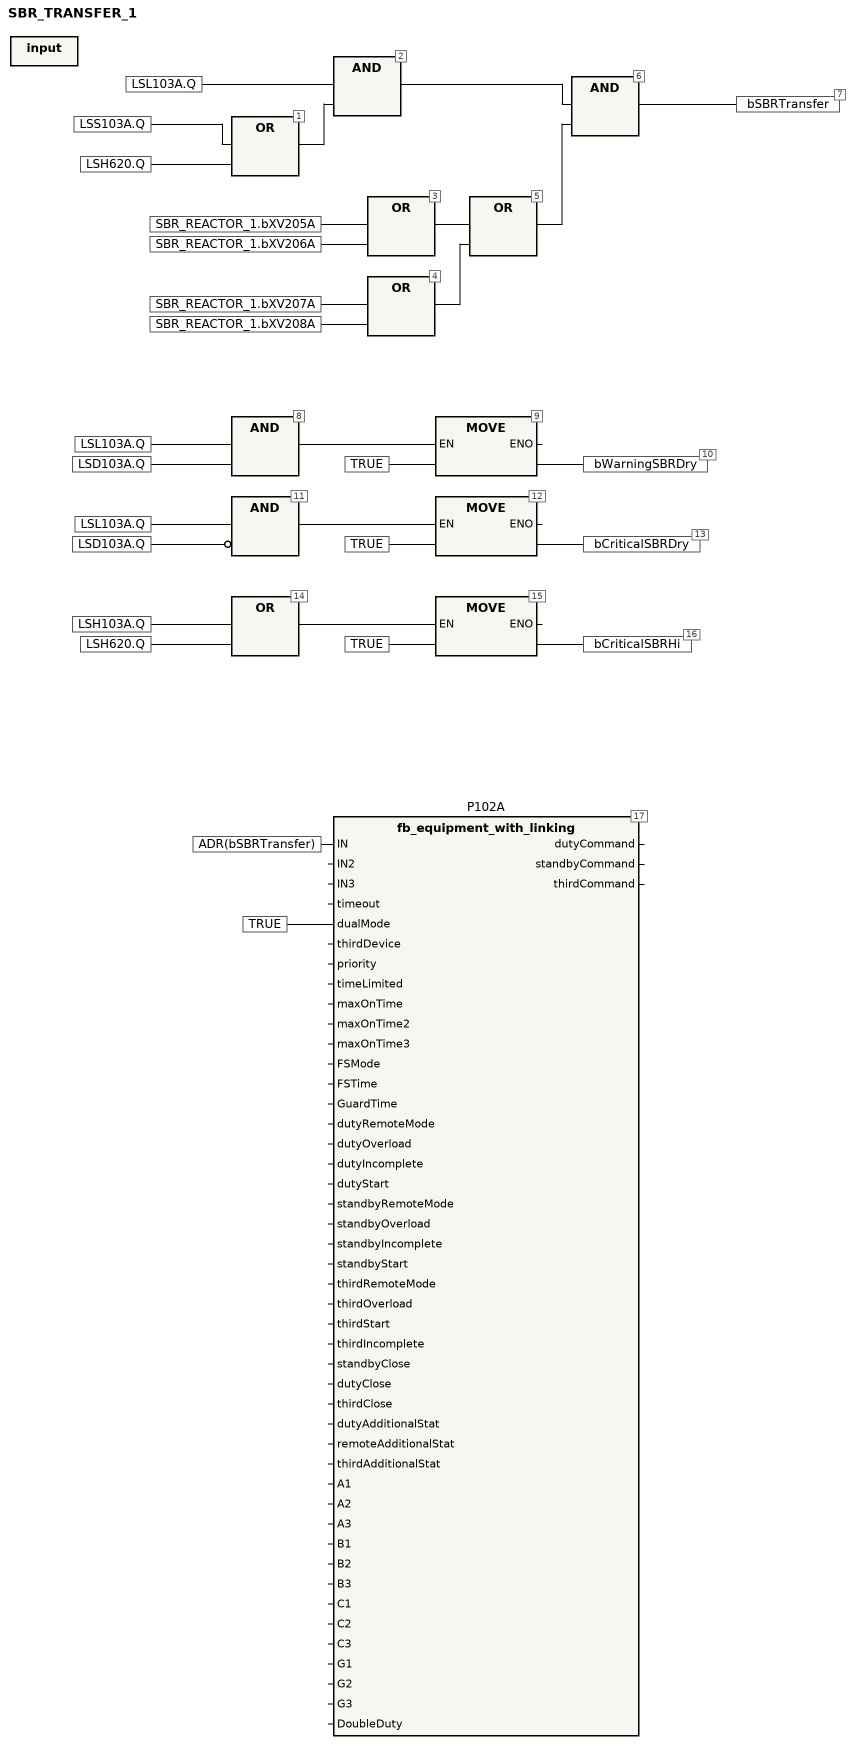
_CFC_ (* Continuous Function Chart, elements in execution order *)
#0 input()
#1 OR(LSS103A.Q, LSH620.Q)
#2 AND(LSL103A.Q, #1)
#3 OR(SBR_REACTOR_1.bXV205A, SBR_REACTOR_1.bXV206A)
#4 OR(SBR_REACTOR_1.bXV207A, SBR_REACTOR_1.bXV208A)
#5 OR(#3, #4)
#6 AND(#2, #5)
#7 bSBRTransfer <= #6
#8 AND(LSL103A.Q, LSD103A.Q)
#9 MOVE(EN: #8, TRUE)
#10 bWarningSBRDry <= #9
#11 AND(LSL103A.Q, NOT LSD103A.Q)
#12 MOVE(EN: #11, TRUE)
#13 bCriticalSBRDry <= #12
#14 OR(LSH103A.Q, LSH620.Q)
#15 MOVE(EN: #14, TRUE)
#16 bCriticalSBRHi <= #15
#17 P102A:fb_equipment_with_linking(IN: ADR(bSBRTransfer), IN2: -, IN3: -, timeout: -, dualMode: TRUE, thirdDevice: -, priority: -, timeLimited: -, maxOnTime: -, maxOnTime2: -, maxOnTime3: -, FSMode: -, FSTime: -, GuardTime: -, dutyRemoteMode: -, dutyOverload: -, dutyIncomplete: -, dutyStart: -, standbyRemoteMode: -, standbyOverload: -, standbyIncomplete: -, standbyStart: -, thirdRemoteMode: -, thirdOverload: -, thirdStart: -, thirdIncomplete: -, standbyClose: -, dutyClose: -, thirdClose: -, dutyAdditionalStat: -, remoteAdditionalStat: -, thirdAdditionalStat: -, A1: -, A2: -, A3: -, B1: -, B2: -, B3: -, C1: -, C2: -, C3: -, G1: -, G2: -, G3: -, DoubleDuty: -)
_END_CFC_
(* the same logic as Structured Text *)
input();
bSBRTransfer := (LSL103A.Q AND (LSS103A.Q OR LSH620.Q)) AND ((SBR_REACTOR_1.bXV205A OR SBR_REACTOR_1.bXV206A) OR (SBR_REACTOR_1.bXV207A OR SBR_REACTOR_1.bXV208A));
IF LSL103A.Q AND LSD103A.Q THEN bWarningSBRDry := TRUE; END_IF;
IF LSL103A.Q AND NOT LSD103A.Q THEN bCriticalSBRDry := TRUE; END_IF;
IF LSH103A.Q OR LSH620.Q THEN bCriticalSBRHi := TRUE; END_IF;
P102A(IN := ADR(bSBRTransfer), dualMode := TRUE);
END_PROGRAM
ACTION Input:
LSD103A( );
LSH103A();
LSH620( );
LSL103A( );
LSS103A( );
END_ACTION

(* POU SBR_REACTOR_1, CFC *)
PROGRAM SBR_REACTOR_1
VAR
	REACTOR1 :SBRReactor;
	REACTOR2 :SBRReactor;
	REACTOR3 :SBRReactor;
	REACTOR4 :SBRReactor;
	OP_SW_R1 AT %I*: BOOL;
	LSL510A: inBlock;
	bDeSlug: BOOL;
	P201A: fb_equipment_with_linking;
	bBlower: BOOL;
	TimerStartBlower1: TON;
	TimerStartBlower2: TON;
	TimerStartBlower3: TON;
	tBlower1: fb_timer_on_off;
	tBlower2: fb_timer_on_off;
	tBlower3: fb_timer_on_off;
	B201A: fb_equipment_with_linking;
	bXV205A: BOOL;
	bXV206A: BOOL;
	bXV207A: BOOL;
	bXV208A: BOOL;
END_VAR

VAR PERSISTENT
	FILLING_TOKEN : INT;
	AERATION_TOKEN: INT;
	DECANTING_TOKEN: INT;
END_VAR
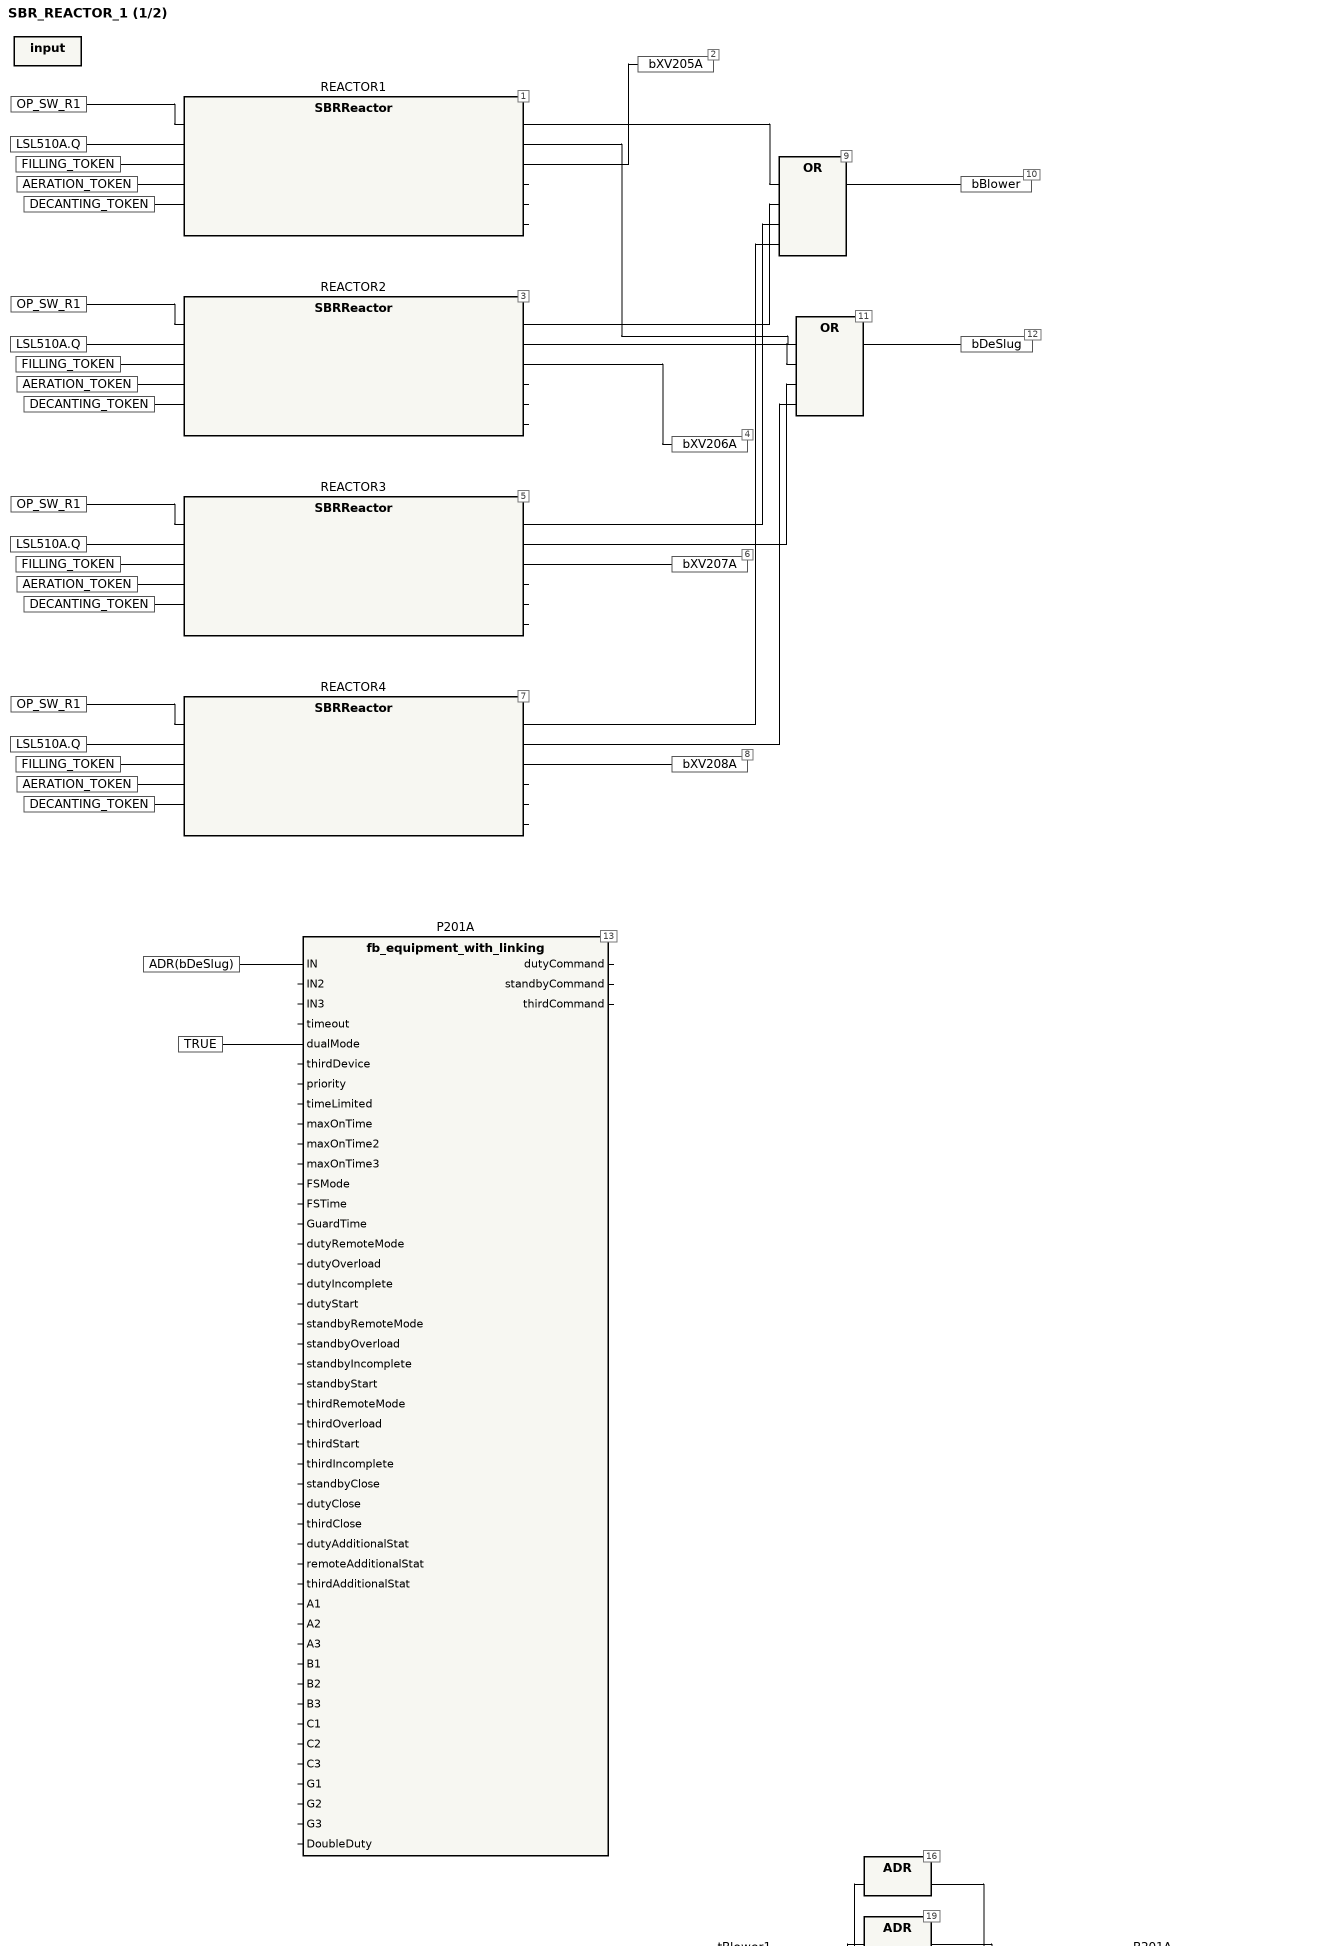
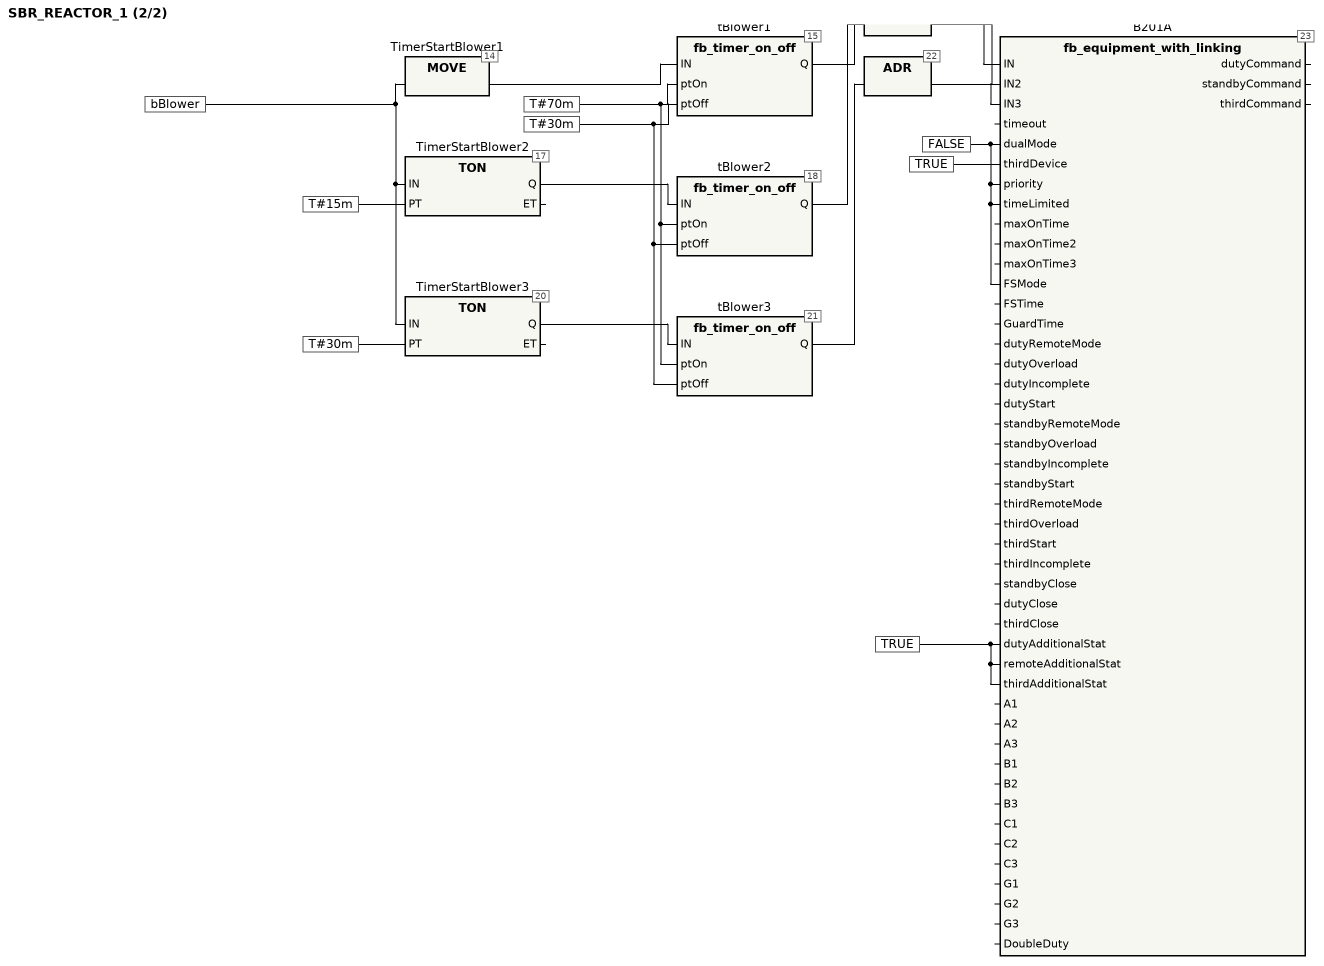
_CFC_ (* Continuous Function Chart, elements in execution order *)
#0 input()
#1 REACTOR1:SBRReactor(OP_SW_R1, LSL510A.Q, FILLING_TOKEN, AERATION_TOKEN, DECANTING_TOKEN)
#2 bXV205A <= #1.out 3
#3 REACTOR2:SBRReactor(OP_SW_R1, LSL510A.Q, FILLING_TOKEN, AERATION_TOKEN, DECANTING_TOKEN)
#4 bXV206A <= #3.out 3
#5 REACTOR3:SBRReactor(OP_SW_R1, LSL510A.Q, FILLING_TOKEN, AERATION_TOKEN, DECANTING_TOKEN)
#6 bXV207A <= #5.out 3
#7 REACTOR4:SBRReactor(OP_SW_R1, LSL510A.Q, FILLING_TOKEN, AERATION_TOKEN, DECANTING_TOKEN)
#8 bXV208A <= #7.out 3
#9 OR(#1.out 1, #3.out 1, #5.out 1, #7.out 1)
#10 bBlower <= #9
#11 OR(#1.out 2, #3.out 2, #5.out 2, #7.out 2)
#12 bDeSlug <= #11
#13 P201A:fb_equipment_with_linking(IN: ADR(bDeSlug), IN2: -, IN3: -, timeout: -, dualMode: TRUE, thirdDevice: -, priority: -, timeLimited: -, maxOnTime: -, maxOnTime2: -, maxOnTime3: -, FSMode: -, FSTime: -, GuardTime: -, dutyRemoteMode: -, dutyOverload: -, dutyIncomplete: -, dutyStart: -, standbyRemoteMode: -, standbyOverload: -, standbyIncomplete: -, standbyStart: -, thirdRemoteMode: -, thirdOverload: -, thirdStart: -, thirdIncomplete: -, standbyClose: -, dutyClose: -, thirdClose: -, dutyAdditionalStat: -, remoteAdditionalStat: -, thirdAdditionalStat: -, A1: -, A2: -, A3: -, B1: -, B2: -, B3: -, C1: -, C2: -, C3: -, G1: -, G2: -, G3: -, DoubleDuty: -)
#14 TimerStartBlower1:MOVE(bBlower)
#15 tBlower1:fb_timer_on_off(IN: #14, ptOn: T#70m, ptOff: T#30m)
#16 ADR(#15.Q)
#17 TimerStartBlower2:TON(IN: bBlower, PT: T#15m)
#18 tBlower2:fb_timer_on_off(IN: #17.Q, ptOn: T#70m, ptOff: T#30m)
#19 ADR(#18.Q)
#20 TimerStartBlower3:TON(IN: bBlower, PT: T#30m)
#21 tBlower3:fb_timer_on_off(IN: #20.Q, ptOn: T#70m, ptOff: T#30m)
#22 ADR(#21.Q)
#23 B201A:fb_equipment_with_linking(IN: #16, IN2: #19, IN3: #22, timeout: -, dualMode: FALSE, thirdDevice: TRUE, priority: FALSE, timeLimited: FALSE, maxOnTime: -, maxOnTime2: -, maxOnTime3: -, FSMode: FALSE, FSTime: -, GuardTime: -, dutyRemoteMode: -, dutyOverload: -, dutyIncomplete: -, dutyStart: -, standbyRemoteMode: -, standbyOverload: -, standbyIncomplete: -, standbyStart: -, thirdRemoteMode: -, thirdOverload: -, thirdStart: -, thirdIncomplete: -, standbyClose: -, dutyClose: -, thirdClose: -, dutyAdditionalStat: TRUE, remoteAdditionalStat: TRUE, thirdAdditionalStat: TRUE, A1: -, A2: -, A3: -, B1: -, B2: -, B3: -, C1: -, C2: -, C3: -, G1: -, G2: -, G3: -, DoubleDuty: -)
_END_CFC_
END_PROGRAM
ACTION input:
LSL510A();
END_ACTION

(* POU module/SBRReactor, ST *)
FUNCTION_BLOCK SBRReactor
VAR_INPUT
	bEnable : BOOL;
	SludgeTankLevelHi: BOOL;

END_VAR
VAR_OUTPUT

	bBlowerOn: BOOL;
	bDeSludgePump: BOOL;
	bSBRValve : BOOL;

END_VAR
VAR PERSISTENT
	step: INT;
END_VAR
VAR

	bFilling: BOOL;
	bAeration: BOOL;
	bSettling: BOOL;
	bDecanting: BOOL;


	bFillingDone: BOOL;
	bAerationDone: BOOL;
	bSettingDone: BOOL;
	bDecantingDone: BOOL;



	MixerOff: TON;
	bSBRMixer: BOOL;
	timerBlower: TON;
	DOtimer: TON;
	rDO201: REAL;
	bWarning_DoNotInRange: BOOL;
	TimerSettling: TON;

	decant: INT;
	bReverseDecant: BOOL;
	timerDecant: TON;


	SBRLevelSensor_LSH200A1: inBlock;

	DecanterLevelSensorHi AT%I*: BOOL;
	DecanterLevelSensorLow AT%I*: BOOL;

	bFowardDacant AT%Q*: BOOL;
	bForwardDecant AT%Q*: BOOL;
	bBlowerValve_XV201A AT%Q* : BOOL;
	bDeslugValve_XV241A AT %Q*: BOOL;
	bSBRValve_XV205A AT %Q*: BOOL;

	DecantTimeLapse: TON;
	bDesluging: BOOL;


	M200_MixerABC: fb_equipment_with_linking;
END_VAR

VAR_IN_OUT
	FILLING_TOKEN : INT;
	AERATION_TOKEN: INT;
	DECANTING_TOKEN: INT;
END_VAR
bFilling:= FALSE;
bAeration:= FALSE;
bSettling:= FALSE;
bDecanting:= FALSE;

IF NOT bEnable THEN
	step := 0;
END_IF

CASE step OF
0:
	(*Idle*)
	step := 10;
10:

	IF FILLING_TOKEN > 0 THEN
		FILLING_TOKEN :=0;
		step := 15;
	END_IF
15:
	bFilling :=TRUE;
	IF bFillingDone THEN
		step := 20;
		FILLING_TOKEN := 1;
	END_IF
20:

	IF AERATION_TOKEN > 0 THEN
		step := 25;
		AERATION_TOKEN := 0;
	END_IF
25:
	IF bAerationDone THEN
		step:= 30;
		AERATION_TOKEN := 1;
	END_IF
30:
	bSettling := TRUE;
	IF bSettingDone THEN
		step := 40;
	END_IF
40:
	IF DECANTING_TOKEN > 0 THEN
		DECANTING_TOKEN := 0;
		step := 45;
	END_IF
45:
		bDecanting := TRUE;
		IF bDecantingDone THEN
			step := 0;
			DECANTING_TOKEN := 1;
		END_IF
END_CASE



filling;
Aeration;
Settle;
Decanting;
FBs;
END_FUNCTION_BLOCK
ACTION Aeration:
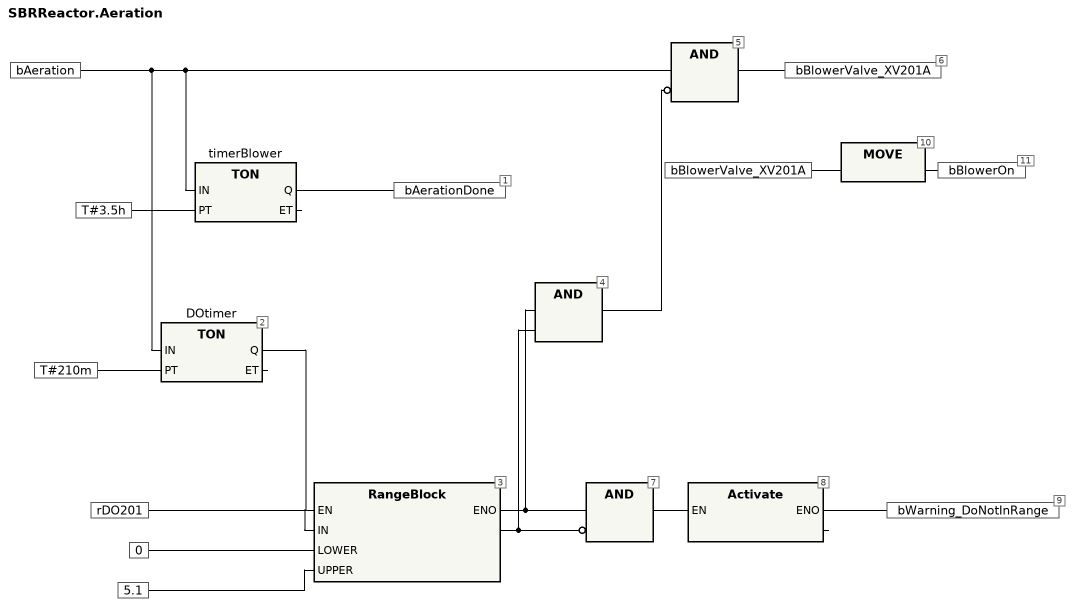
_CFC_ (* Continuous Function Chart, elements in execution order *)
#0 timerBlower:TON(IN: bAeration, PT: T#3.5h)
#1 bAerationDone <= #0.Q
#2 DOtimer:TON(IN: bAeration, PT: T#210m)
#3 RangeBlock(EN: #2.Q, IN: rDO201, LOWER: 0, UPPER: 5.1)
#4 AND(#3.ENO, #3)
#5 AND(bAeration, NOT #4)
#6 bBlowerValve_XV201A <= #5
#7 AND(#3.ENO, NOT #3)
#8 Activate(EN: #7)
#9 bWarning_DoNotInRange <= #8.ENO
#10 MOVE(bBlowerValve_XV201A)
#11 bBlowerOn <= #10
_END_CFC_
END_ACTION
ACTION Decanting:
IF NOT bDecanting THEN
decant := 0;
END_IF

bDecantingDone := (decant >= 60);


CASE decant OF
0:
	decant := 10;
10:

	IF DecanterLevelSensorHi THEN
		(*start Reverse Sequence*)
		bForwardDecant :=FALSE;
		decant := 20;
	ELSE
		bForwardDecant :=TRUE;
	END_IF


20:
	bReverseDecant := TRUE;
	timerDecant(IN:= TRUE, PT:= T#2s);
		IF timerDecant.Q THEN
			timerDecant(IN:= FALSE);
			bReverseDecant := FALSE;
			decant := 30;
		END_IF
30:
	timerDecant(IN:= TRUE, PT:= T#10s);
		IF timerDecant.Q THEN
			timerDecant(IN:= FALSE);
			IF DecanterLevelSensorLow THEN
				decant := 40;
			ELSE
				decant := 20;
			END_IF
		END_IF
40:
	timerDecant(IN:=TRUE,PT:=T#300s);
	IF timerDecant.Q THEN
		timerDecant(IN:=FALSE);
		decant := 50;
	END_IF
50:

	IF DecanterLevelSensorHi THEN
		(*start Reverse Sequence*)
		bForwardDecant :=FALSE;
		decant := 60;
	ELSE
		bForwardDecant :=TRUE;
	END_IF
60:
;
END_CASE

DecantTimeLapse(IN:=bDecanting, PT:= T#4000s);
bDesluging := (DecantTimeLapse.ET <= T#15m) OR (DecantTimeLapse.ET >= T#15m);

bDeslugValve_XV241A := bDesluging AND NOT SludgeTankLevelHi;
bDeSludgePump := bDeslugValve_XV241A;
END_ACTION
ACTION FBs:
M200_MixerABC(
	IN:=ADR(bSBRMixer) ,
	IN2:=ADR(bSBRMixer) ,
	IN3:= ADR(bSBRMixer),
	timeout:= T#2s,
	dualMode:=FALSE ,
	thirdDevice:= TRUE,
	priority:= FALSE,
	timeLimited:= FALSE,
	FSMode:=FALSE ,
	dutyRemoteMode:= ,
	dutyOverload:= , 
	dutyIncomplete:= ,
	dutyStart:= , 
	standbyRemoteMode:= ,
	standbyOverload:= , 
	standbyIncomplete:= , 
	standbyStart:= , 
	thirdRemoteMode:= , 
	thirdOverload:= , 
	thirdStart:= , 
	thirdIncomplete:= , 
	dutyCommand=> ,
	standbyCommand=> , 
	thirdCommand=> );
END_ACTION
ACTION filling:
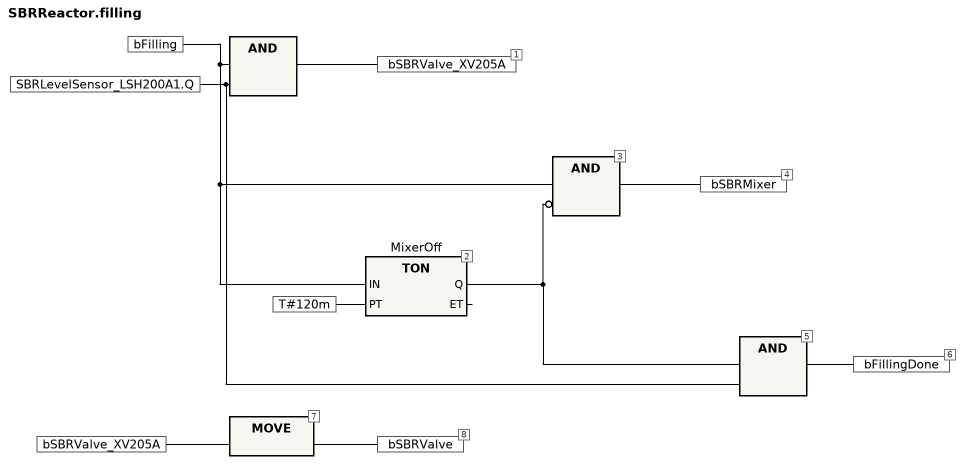
_CFC_ (* Continuous Function Chart, elements in execution order *)
#0 AND(bFilling, SBRLevelSensor_LSH200A1.Q)
#1 bSBRValve_XV205A <= #0
#2 MixerOff:TON(IN: bFilling, PT: T#120m)
#3 AND(bFilling, NOT #2.Q)
#4 bSBRMixer <= #3
#5 AND(#2.Q, SBRLevelSensor_LSH200A1.Q)
#6 bFillingDone <= #5
#7 MOVE(bSBRValve_XV205A)
#8 bSBRValve <= #7
_END_CFC_
(* the same logic as Structured Text *)
bSBRValve_XV205A := bFilling AND SBRLevelSensor_LSH200A1.Q;
MixerOff(IN := bFilling, PT := T#120m);
bSBRMixer := bFilling AND NOT MixerOff.Q;
bFillingDone := MixerOff.Q AND SBRLevelSensor_LSH200A1.Q;
bSBRValve := bSBRValve_XV205A;
END_ACTION
ACTION Settle:
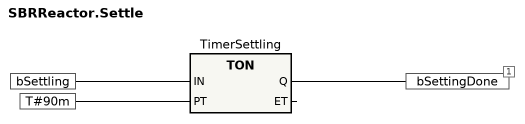
_CFC_ (* Continuous Function Chart, elements in execution order *)
#0 TimerSettling:TON(IN: bSettling, PT: T#90m)
#1 bSettingDone <= #0.Q
_END_CFC_
(* the same logic as Structured Text *)
TimerSettling(IN := bSettling, PT := T#90m);
bSettingDone := TimerSettling.Q;
END_ACTION

(* POU module/RangeBlock, ST *)
FUNCTION RangeBlock : BOOL
VAR_INPUT
	IN:REAL;
	LOWER : REAL;
	UPPER : REAL;
END_VAR
VAR
END_VAR
IF IN >= LOWER AND IN < UPPER THEN
	RangeBlock :=TRUE;
ELSE
	RangeBlock := FALSE;
END_IF
END_FUNCTION

(* POU module/Activate, ST *)
FUNCTION Activate : BOOL
VAR_INPUT
END_VAR
VAR
END_VAR
Activate := TRUE;
END_FUNCTION

(* POU module/fb_timer_on_off, CFC *)
FUNCTION_BLOCK fb_timer_on_off
VAR_INPUT
	IN: BOOL;
	ptOn: TIME;
	ptOff: TIME;
END_VAR
VAR_OUTPUT
	Q: BOOL;
END_VAR
VAR
	ON: TON;
	OFF: TON;
END_VAR
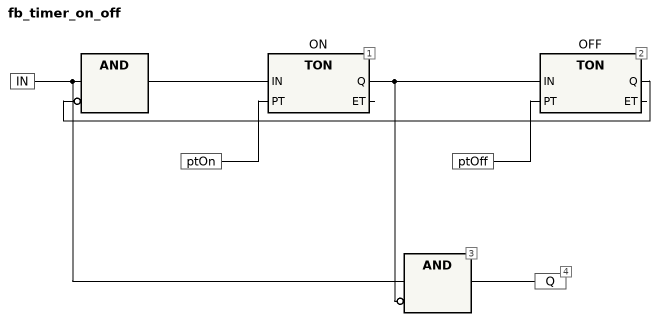
_CFC_ (* Continuous Function Chart, elements in execution order *)
#0 AND(IN, NOT #2.Q)
#1 ON:TON(IN: #0, PT: ptOn)
#2 OFF:TON(IN: #1.Q, PT: ptOff)
#3 AND(IN, NOT #1.Q)
#4 Q <= #3
_END_CFC_
(* the same logic as Structured Text *)
ON(IN := IN AND NOT OFF.Q, PT := ptOn);
OFF(IN := ON.Q, PT := ptOff);
Q := IN AND NOT ON.Q;
END_FUNCTION_BLOCK

(* POU STREAM_INLET_MIXER_2, CFC *)
PROGRAM STREAM_INLET_MIXER_2
VAR
	LSL101B : inBlock;
	LSS101B : inBlock;
	LSH101B : inBlock;
	LSD101B : inBlock;

	LSL100B : inBlock;
	LSHL100B:inBlock;

	bEQPump: BOOL;
	bCriticalEQFloatHi: BOOL;
	bWarningFloatSensorLow: BOOL;
	bCriticalFloatSensorDry: BOOL;
	bEQMixer: BOOL;
	P101B: fb_equipment_with_linking;
	M101B: fb_equipment_with_linking;
END_VAR
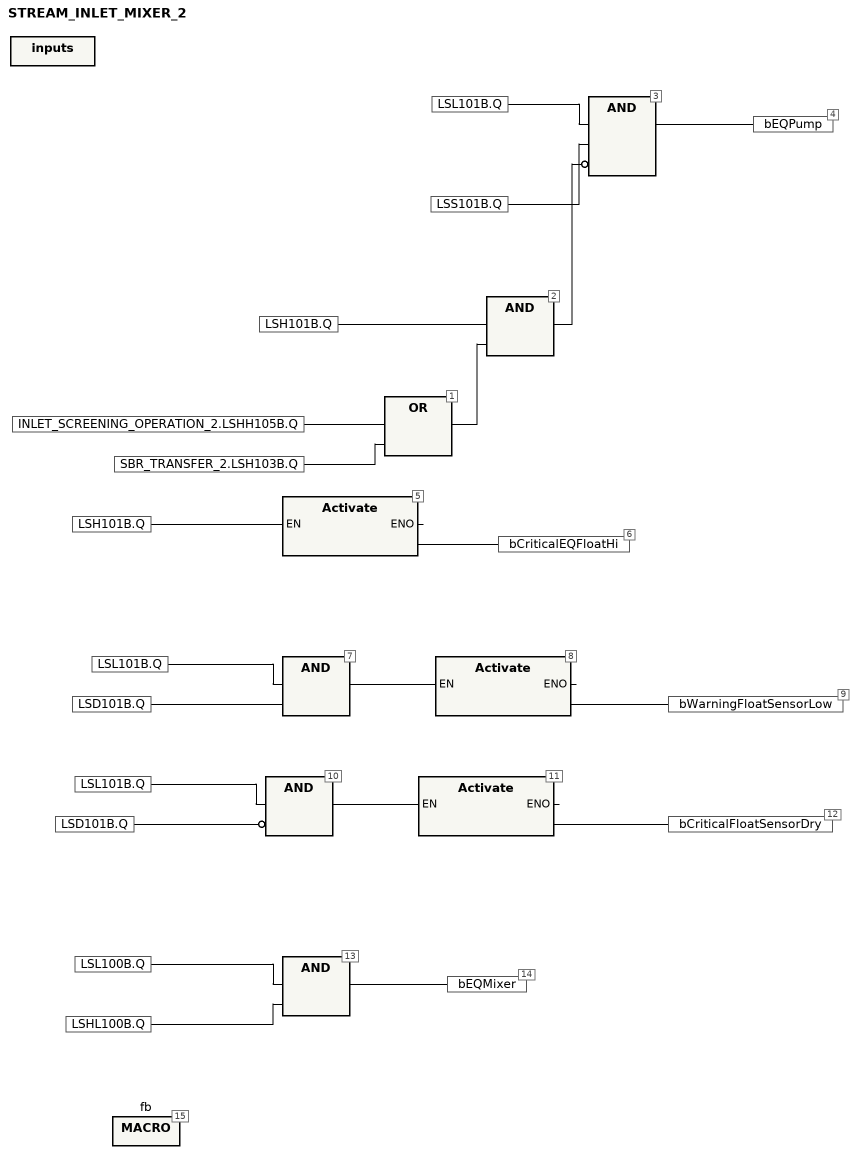
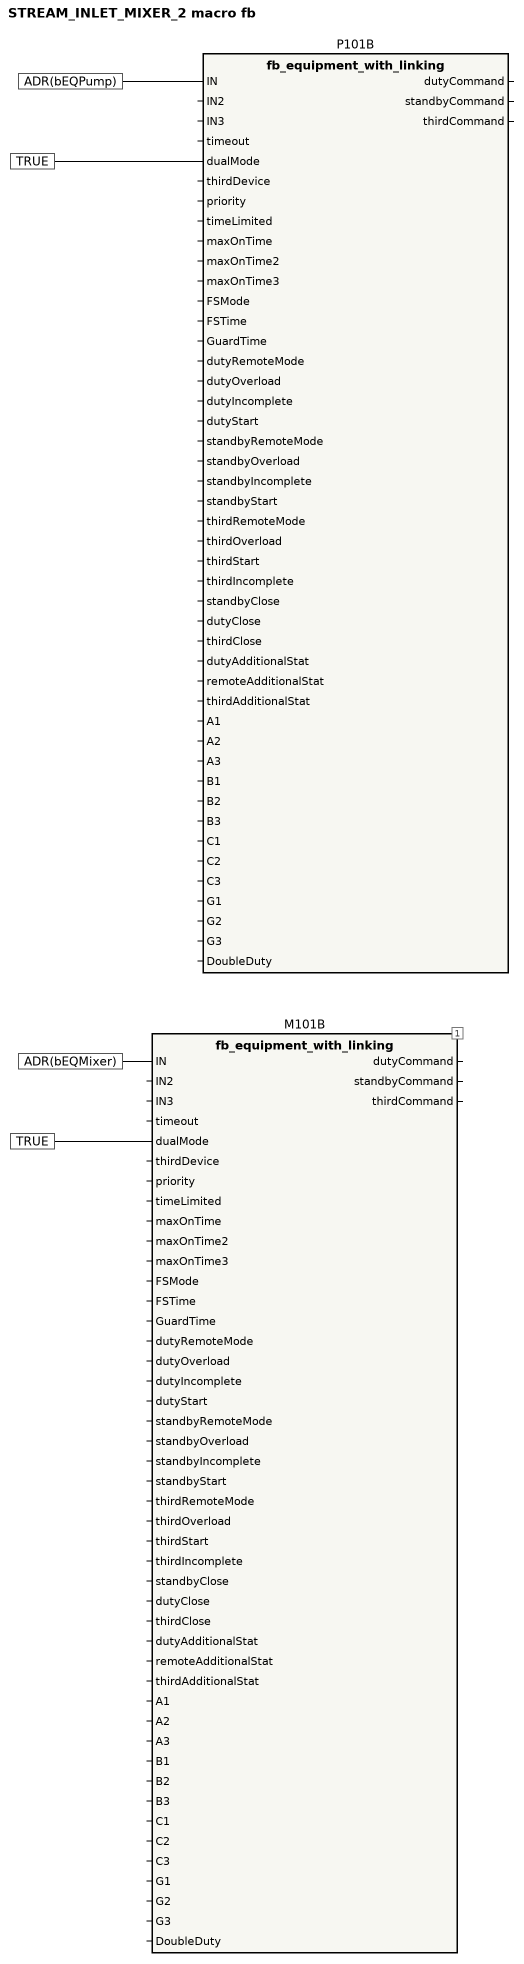
_CFC_ (* Continuous Function Chart, elements in execution order *)
#0 inputs()
#1 OR(INLET_SCREENING_OPERATION_2.LSHH105B.Q, SBR_TRANSFER_2.LSH103B.Q)
#2 AND(LSH101B.Q, #1)
#3 AND(LSL101B.Q, LSS101B.Q, NOT #2)
#4 bEQPump <= #3
#5 Activate(EN: LSH101B.Q)
#6 bCriticalEQFloatHi <= #5
#7 AND(LSL101B.Q, LSD101B.Q)
#8 Activate(EN: #7)
#9 bWarningFloatSensorLow <= #8
#10 AND(LSL101B.Q, NOT LSD101B.Q)
#11 Activate(EN: #10)
#12 bCriticalFloatSensorDry <= #11
#13 AND(LSL100B.Q, LSHL100B.Q)
#14 bEQMixer <= #13
#15 MACRO fb()
	#16 P101B:fb_equipment_with_linking(IN: ADR(bEQPump), IN2: -, IN3: -, timeout: -, dualMode: TRUE, thirdDevice: -, priority: -, timeLimited: -, maxOnTime: -, maxOnTime2: -, maxOnTime3: -, FSMode: -, FSTime: -, GuardTime: -, dutyRemoteMode: -, dutyOverload: -, dutyIncomplete: -, dutyStart: -, standbyRemoteMode: -, standbyOverload: -, standbyIncomplete: -, standbyStart: -, thirdRemoteMode: -, thirdOverload: -, thirdStart: -, thirdIncomplete: -, standbyClose: -, dutyClose: -, thirdClose: -, dutyAdditionalStat: -, remoteAdditionalStat: -, thirdAdditionalStat: -, A1: -, A2: -, A3: -, B1: -, B2: -, B3: -, C1: -, C2: -, C3: -, G1: -, G2: -, G3: -, DoubleDuty: -)
	#17 M101B:fb_equipment_with_linking(IN: ADR(bEQMixer), IN2: -, IN3: -, timeout: -, dualMode: TRUE, thirdDevice: -, priority: -, timeLimited: -, maxOnTime: -, maxOnTime2: -, maxOnTime3: -, FSMode: -, FSTime: -, GuardTime: -, dutyRemoteMode: -, dutyOverload: -, dutyIncomplete: -, dutyStart: -, standbyRemoteMode: -, standbyOverload: -, standbyIncomplete: -, standbyStart: -, thirdRemoteMode: -, thirdOverload: -, thirdStart: -, thirdIncomplete: -, standbyClose: -, dutyClose: -, thirdClose: -, dutyAdditionalStat: -, remoteAdditionalStat: -, thirdAdditionalStat: -, A1: -, A2: -, A3: -, B1: -, B2: -, B3: -, C1: -, C2: -, C3: -, G1: -, G2: -, G3: -, DoubleDuty: -)
END_MACRO
_END_CFC_
(* the same logic as Structured Text *)
inputs();
bEQPump := LSL101B.Q AND LSS101B.Q AND NOT (LSH101B.Q AND (INLET_SCREENING_OPERATION_2.LSHH105B.Q OR SBR_TRANSFER_2.LSH103B.Q));
IF LSH101B.Q THEN bCriticalEQFloatHi := Activate(); END_IF;
IF LSL101B.Q AND LSD101B.Q THEN bWarningFloatSensorLow := Activate(); END_IF;
IF LSL101B.Q AND NOT LSD101B.Q THEN bCriticalFloatSensorDry := Activate(); END_IF;
bEQMixer := LSL100B.Q AND LSHL100B.Q;
(* macro fb *)
P101B(IN := ADR(bEQPump), dualMode := TRUE);
M101B(IN := ADR(bEQMixer), dualMode := TRUE);
END_PROGRAM
ACTION inputs:
	LSL101B();
	LSS101B();
	LSH101B();
	LSD101B();

	LSL100B();
	LSHL100B();
END_ACTION

(* POU INLET_SCREENING_OPERATION_2, CFC *)
PROGRAM INLET_SCREENING_OPERATION_2
VAR
	bTest: BOOL;
	bTestReault: BOOL;

	LSH105B : inBlock;
	LSHH105B: inBlock;
	bPenstockDual: BOOL;
	Timer1: TON;
	bWarningStreamLineOverflow: BOOL;
	bFineScreen: BOOL;
	F101B: fb_equipment_with_linking;
	XV101B1 : fb_equipment_with_linking;
	StopTimer: TON;
	bScrewConveyor: BOOL;
	bScreenCompactor: BOOL;
	bWaterSprayScreenDuty: BOOL;
	bWaterSprayScreenStandby: BOOL;
	bPenstockDuty: BOOL;
	bPenstockStandby: BOOL;
	XV101B2: fb_equipment_with_linking;
	timerCompactor: TON;
	bFineScreenDual: BOOL;
	PS101B: fb_equipment_with_linking;
	bContinuousWaterSpray: BOOL;
	C102B: fb_equipment_with_linking;
	C101B: fb_equipment_with_linking;
	XV102B: fb_equipment_with_linking;
END_VAR
VAR (* helpers for the ST form of the networks *)
	_en57 : BOOL;
	_t57 : BOOL;
	_en85 : BOOL;
	_t85 : BOOL;
END_VAR
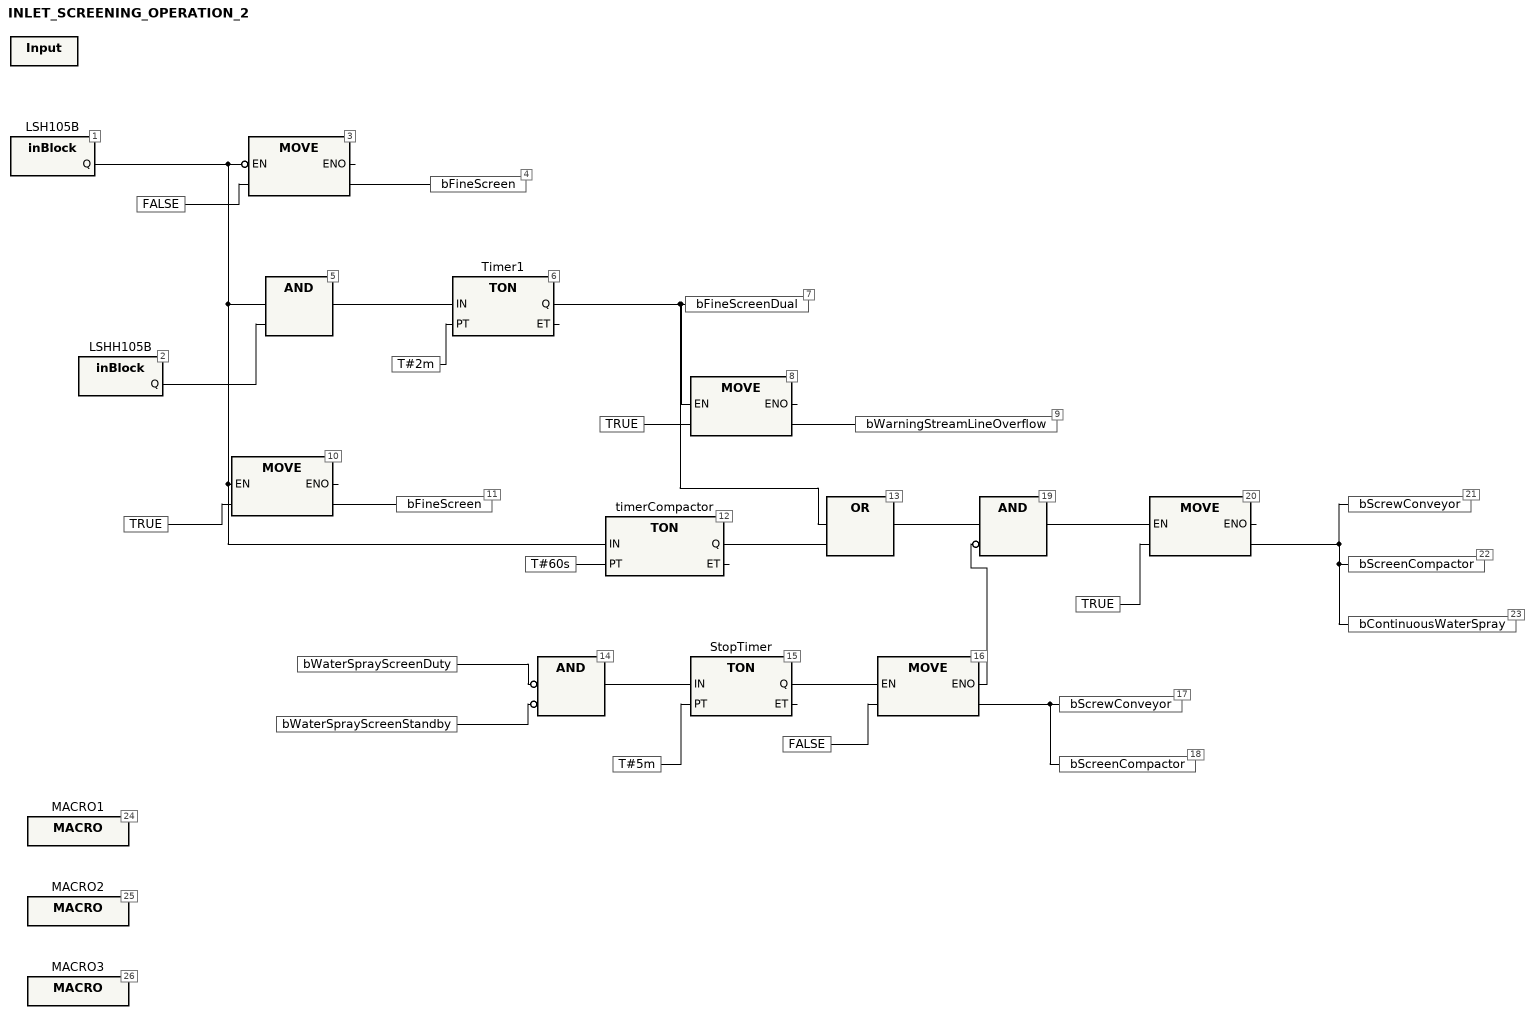
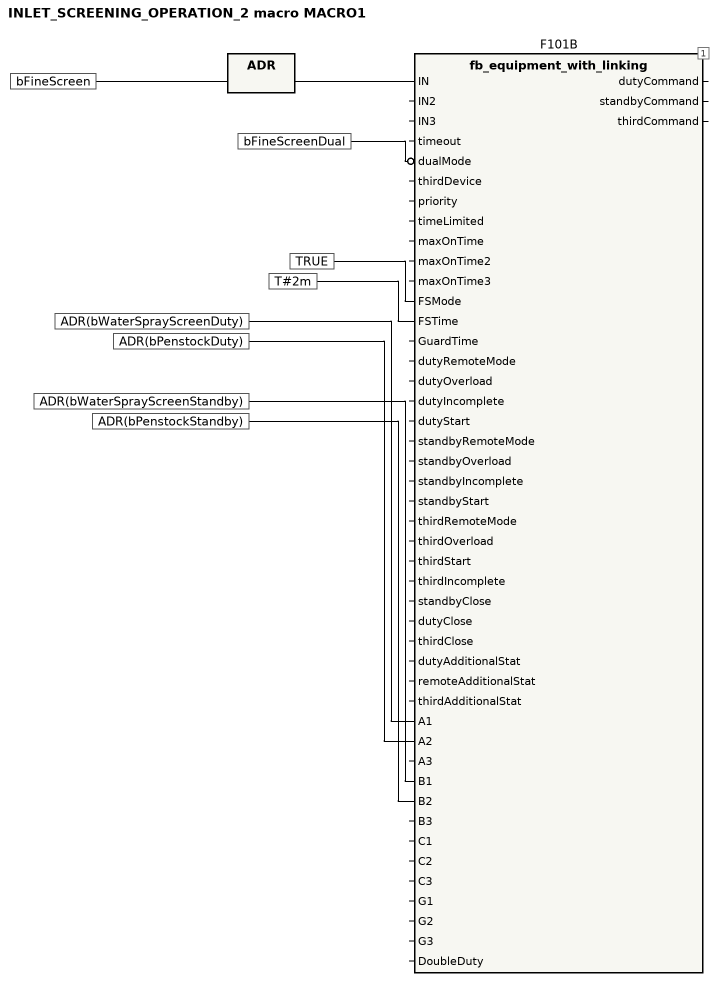
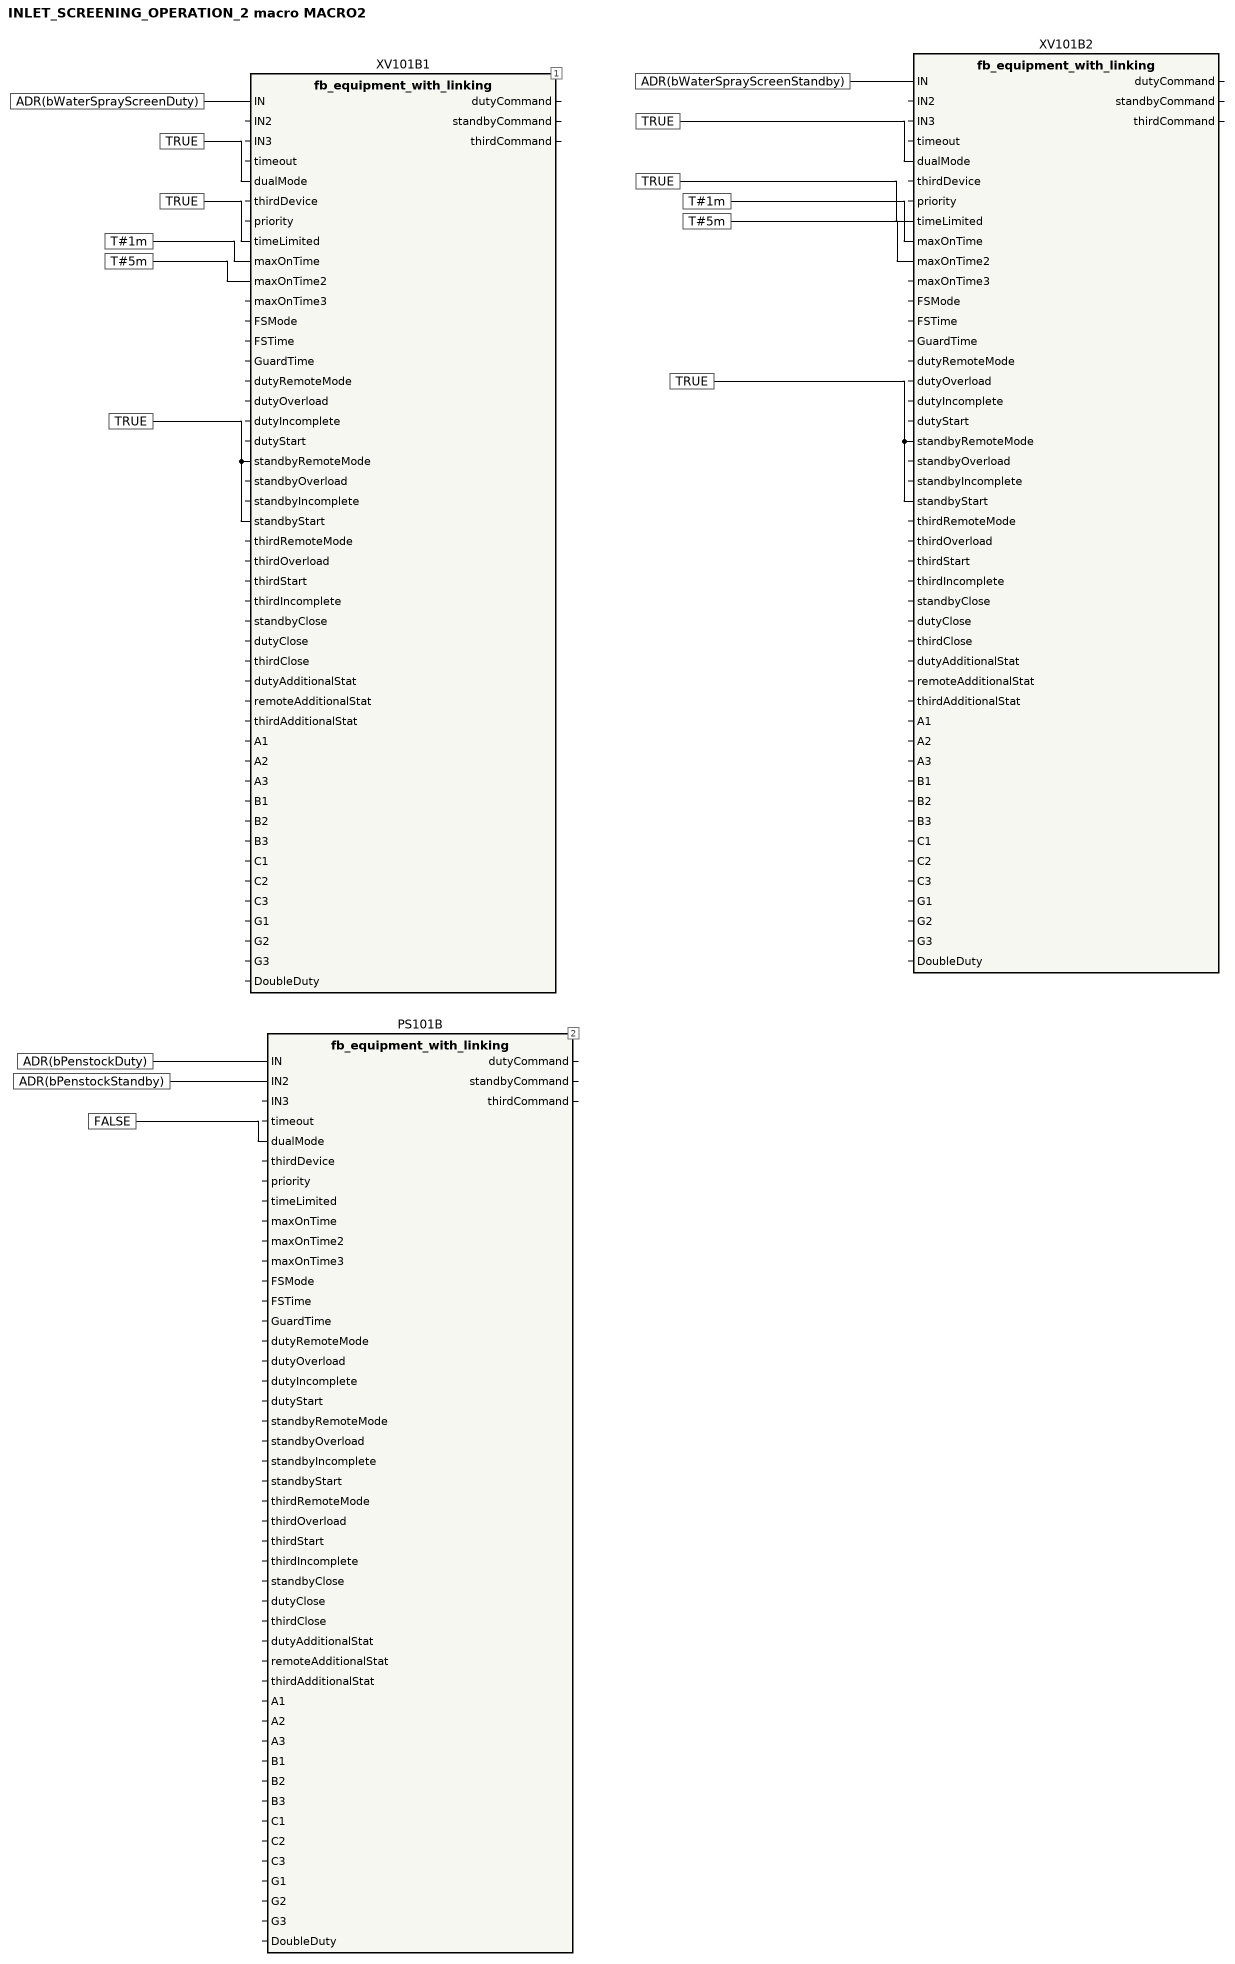
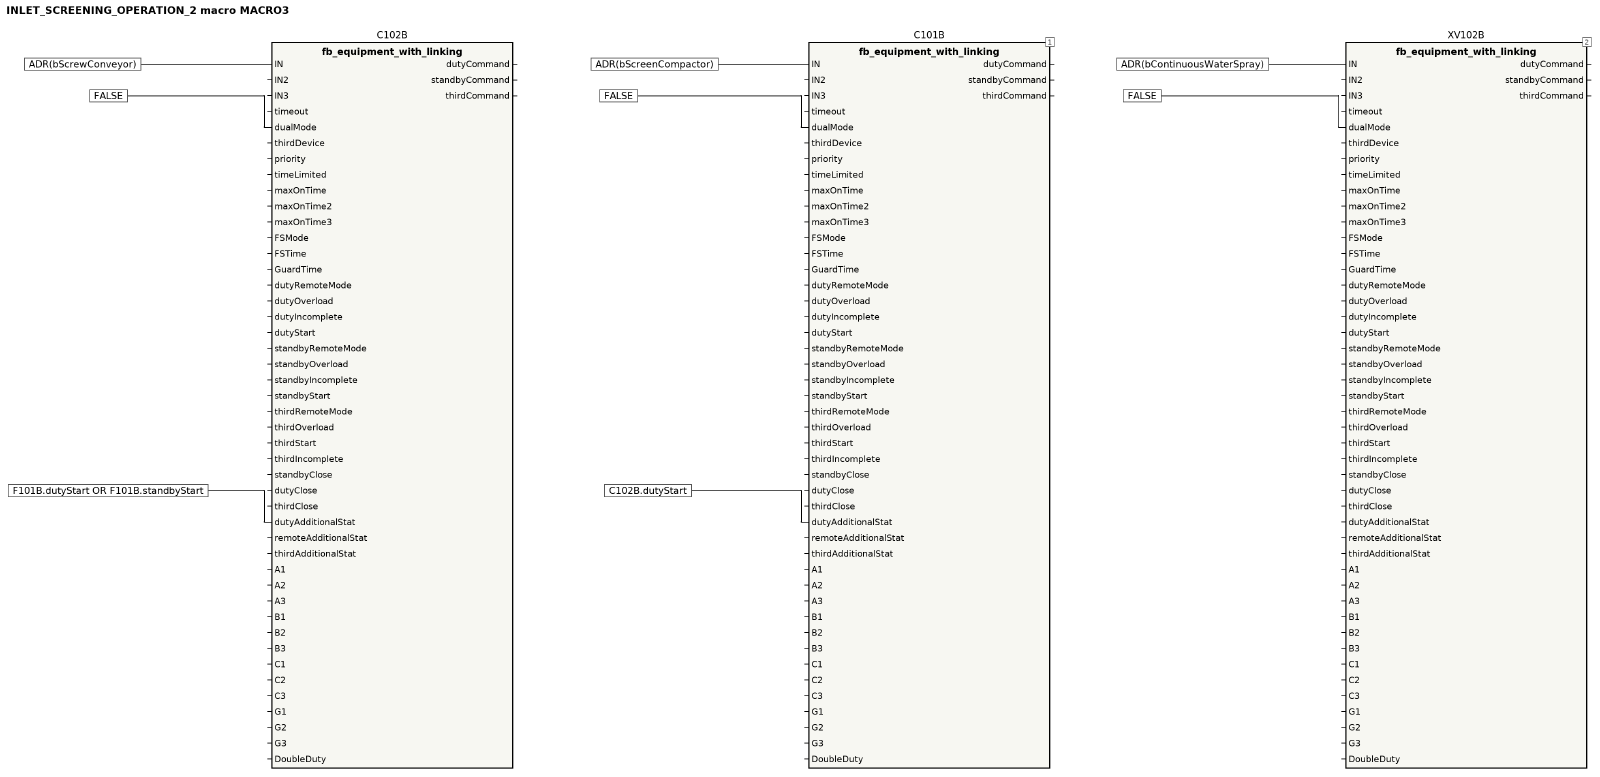
_CFC_ (* Continuous Function Chart, elements in execution order *)
#0 Input()
#1 LSH105B:inBlock()
#2 LSHH105B:inBlock()
#3 MOVE(EN: NOT #1.Q, FALSE)
#4 bFineScreen <= #3
#5 AND(#1.Q, #2.Q)
#6 Timer1:TON(IN: #5, PT: T#2m)
#7 bFineScreenDual <= #6.Q
#8 MOVE(EN: #6.Q, TRUE)
#9 bWarningStreamLineOverflow <= #8
#10 MOVE(EN: #1.Q, TRUE)
#11 bFineScreen <= #10
#12 timerCompactor:TON(IN: #1.Q, PT: T#60s)
#13 OR(#6.Q, #12.Q)
#14 AND(NOT bWaterSprayScreenDuty, NOT bWaterSprayScreenStandby)
#15 StopTimer:TON(IN: #14, PT: T#5m)
#16 MOVE(EN: #15.Q, FALSE)
#17 bScrewConveyor <= #16
#18 bScreenCompactor <= #16
#19 AND(#13, NOT #16.ENO)
#20 MOVE(EN: #19, TRUE)
#21 bScrewConveyor <= #20
#22 bScreenCompactor <= #20
#23 bContinuousWaterSpray <= #20
#24 MACRO MACRO1()
	#25 ADR(bFineScreen)
	#26 F101B:fb_equipment_with_linking(IN: #25, IN2: -, IN3: -, timeout: -, dualMode: NOT bFineScreenDual, thirdDevice: -, priority: -, timeLimited: -, maxOnTime: -, maxOnTime2: -, maxOnTime3: -, FSMode: TRUE, FSTime: T#2m, GuardTime: -, dutyRemoteMode: -, dutyOverload: -, dutyIncomplete: -, dutyStart: -, standbyRemoteMode: -, standbyOverload: -, standbyIncomplete: -, standbyStart: -, thirdRemoteMode: -, thirdOverload: -, thirdStart: -, thirdIncomplete: -, standbyClose: -, dutyClose: -, thirdClose: -, dutyAdditionalStat: -, remoteAdditionalStat: -, thirdAdditionalStat: -, A1: ADR(bWaterSprayScreenDuty), A2: ADR(bPenstockDuty), A3: -, B1: ADR(bWaterSprayScreenStandby), B2: ADR(bPenstockStandby), B3: -, C1: -, C2: -, C3: -, G1: -, G2: -, G3: -, DoubleDuty: -)
END_MACRO
#27 MACRO MACRO2()
	#28 XV101B2:fb_equipment_with_linking(IN: ADR(bWaterSprayScreenStandby), IN2: -, IN3: -, timeout: -, dualMode: TRUE, thirdDevice: -, priority: -, timeLimited: TRUE, maxOnTime: T#1m, maxOnTime2: T#5m, maxOnTime3: -, FSMode: -, FSTime: -, GuardTime: -, dutyRemoteMode: -, dutyOverload: -, dutyIncomplete: -, dutyStart: -, standbyRemoteMode: TRUE, standbyOverload: -, standbyIncomplete: -, standbyStart: TRUE, thirdRemoteMode: -, thirdOverload: -, thirdStart: -, thirdIncomplete: -, standbyClose: -, dutyClose: -, thirdClose: -, dutyAdditionalStat: -, remoteAdditionalStat: -, thirdAdditionalStat: -, A1: -, A2: -, A3: -, B1: -, B2: -, B3: -, C1: -, C2: -, C3: -, G1: -, G2: -, G3: -, DoubleDuty: -)
	#29 XV101B1:fb_equipment_with_linking(IN: ADR(bWaterSprayScreenDuty), IN2: -, IN3: -, timeout: -, dualMode: TRUE, thirdDevice: -, priority: -, timeLimited: TRUE, maxOnTime: T#1m, maxOnTime2: T#5m, maxOnTime3: -, FSMode: -, FSTime: -, GuardTime: -, dutyRemoteMode: -, dutyOverload: -, dutyIncomplete: -, dutyStart: -, standbyRemoteMode: TRUE, standbyOverload: -, standbyIncomplete: -, standbyStart: TRUE, thirdRemoteMode: -, thirdOverload: -, thirdStart: -, thirdIncomplete: -, standbyClose: -, dutyClose: -, thirdClose: -, dutyAdditionalStat: -, remoteAdditionalStat: -, thirdAdditionalStat: -, A1: -, A2: -, A3: -, B1: -, B2: -, B3: -, C1: -, C2: -, C3: -, G1: -, G2: -, G3: -, DoubleDuty: -)
	#30 PS101B:fb_equipment_with_linking(IN: ADR(bPenstockDuty), IN2: ADR(bPenstockStandby), IN3: -, timeout: -, dualMode: FALSE, thirdDevice: -, priority: -, timeLimited: -, maxOnTime: -, maxOnTime2: -, maxOnTime3: -, FSMode: -, FSTime: -, GuardTime: -, dutyRemoteMode: -, dutyOverload: -, dutyIncomplete: -, dutyStart: -, standbyRemoteMode: -, standbyOverload: -, standbyIncomplete: -, standbyStart: -, thirdRemoteMode: -, thirdOverload: -, thirdStart: -, thirdIncomplete: -, standbyClose: -, dutyClose: -, thirdClose: -, dutyAdditionalStat: -, remoteAdditionalStat: -, thirdAdditionalStat: -, A1: -, A2: -, A3: -, B1: -, B2: -, B3: -, C1: -, C2: -, C3: -, G1: -, G2: -, G3: -, DoubleDuty: -)
END_MACRO
#31 MACRO MACRO3()
	#32 C102B:fb_equipment_with_linking(IN: ADR(bScrewConveyor), IN2: -, IN3: -, timeout: -, dualMode: FALSE, thirdDevice: -, priority: -, timeLimited: -, maxOnTime: -, maxOnTime2: -, maxOnTime3: -, FSMode: -, FSTime: -, GuardTime: -, dutyRemoteMode: -, dutyOverload: -, dutyIncomplete: -, dutyStart: -, standbyRemoteMode: -, standbyOverload: -, standbyIncomplete: -, standbyStart: -, thirdRemoteMode: -, thirdOverload: -, thirdStart: -, thirdIncomplete: -, standbyClose: -, dutyClose: -, thirdClose: -, dutyAdditionalStat: F101B.dutyStart OR F101B.standbyStart, remoteAdditionalStat: -, thirdAdditionalStat: -, A1: -, A2: -, A3: -, B1: -, B2: -, B3: -, C1: -, C2: -, C3: -, G1: -, G2: -, G3: -, DoubleDuty: -)
	#33 C101B:fb_equipment_with_linking(IN: ADR(bScreenCompactor), IN2: -, IN3: -, timeout: -, dualMode: FALSE, thirdDevice: -, priority: -, timeLimited: -, maxOnTime: -, maxOnTime2: -, maxOnTime3: -, FSMode: -, FSTime: -, GuardTime: -, dutyRemoteMode: -, dutyOverload: -, dutyIncomplete: -, dutyStart: -, standbyRemoteMode: -, standbyOverload: -, standbyIncomplete: -, standbyStart: -, thirdRemoteMode: -, thirdOverload: -, thirdStart: -, thirdIncomplete: -, standbyClose: -, dutyClose: -, thirdClose: -, dutyAdditionalStat: C102B.dutyStart, remoteAdditionalStat: -, thirdAdditionalStat: -, A1: -, A2: -, A3: -, B1: -, B2: -, B3: -, C1: -, C2: -, C3: -, G1: -, G2: -, G3: -, DoubleDuty: -)
	#34 XV102B:fb_equipment_with_linking(IN: ADR(bContinuousWaterSpray), IN2: -, IN3: -, timeout: -, dualMode: FALSE, thirdDevice: -, priority: -, timeLimited: -, maxOnTime: -, maxOnTime2: -, maxOnTime3: -, FSMode: -, FSTime: -, GuardTime: -, dutyRemoteMode: -, dutyOverload: -, dutyIncomplete: -, dutyStart: -, standbyRemoteMode: -, standbyOverload: -, standbyIncomplete: -, standbyStart: -, thirdRemoteMode: -, thirdOverload: -, thirdStart: -, thirdIncomplete: -, standbyClose: -, dutyClose: -, thirdClose: -, dutyAdditionalStat: -, remoteAdditionalStat: -, thirdAdditionalStat: -, A1: -, A2: -, A3: -, B1: -, B2: -, B3: -, C1: -, C2: -, C3: -, G1: -, G2: -, G3: -, DoubleDuty: -)
END_MACRO
_END_CFC_
(* the same logic as Structured Text *)
Input();
LSH105B();
LSHH105B();
IF NOT LSH105B.Q THEN bFineScreen := FALSE; END_IF;
Timer1(IN := LSH105B.Q AND LSHH105B.Q, PT := T#2m);
bFineScreenDual := Timer1.Q;
IF Timer1.Q THEN bWarningStreamLineOverflow := TRUE; END_IF;
IF LSH105B.Q THEN bFineScreen := TRUE; END_IF;
timerCompactor(IN := LSH105B.Q, PT := T#60s);
StopTimer(IN := NOT bWaterSprayScreenDuty AND NOT bWaterSprayScreenStandby, PT := T#5m);
_en57 := StopTimer.Q;
IF _en57 THEN _t57 := FALSE; END_IF;
IF _en57 THEN bScrewConveyor := _t57; END_IF;
IF _en57 THEN bScreenCompactor := _t57; END_IF;
_en85 := (Timer1.Q OR timerCompactor.Q) AND NOT _en57;
IF _en85 THEN _t85 := TRUE; END_IF;
IF _en85 THEN bScrewConveyor := _t85; END_IF;
IF _en85 THEN bScreenCompactor := _t85; END_IF;
IF _en85 THEN bContinuousWaterSpray := _t85; END_IF;
(* macro MACRO1 *)
F101B(IN := ADR(bFineScreen), dualMode := NOT bFineScreenDual, FSMode := TRUE, FSTime := T#2m, A1 := ADR(bWaterSprayScreenDuty), A2 := ADR(bPenstockDuty), B1 := ADR(bWaterSprayScreenStandby), B2 := ADR(bPenstockStandby));
(* macro MACRO2 *)
XV101B2(IN := ADR(bWaterSprayScreenStandby), dualMode := TRUE, timeLimited := TRUE, maxOnTime := T#1m, maxOnTime2 := T#5m, standbyRemoteMode := TRUE, standbyStart := TRUE);
XV101B1(IN := ADR(bWaterSprayScreenDuty), dualMode := TRUE, timeLimited := TRUE, maxOnTime := T#1m, maxOnTime2 := T#5m, standbyRemoteMode := TRUE, standbyStart := TRUE);
PS101B(IN := ADR(bPenstockDuty), IN2 := ADR(bPenstockStandby), dualMode := FALSE);
(* macro MACRO3 *)
C102B(IN := ADR(bScrewConveyor), dualMode := FALSE, dutyAdditionalStat := F101B.dutyStart OR F101B.standbyStart);
C101B(IN := ADR(bScreenCompactor), dualMode := FALSE, dutyAdditionalStat := C102B.dutyStart);
XV102B(IN := ADR(bContinuousWaterSpray), dualMode := FALSE);
END_PROGRAM
ACTION Input:
LSH105B( );
LSHH105B( );
END_ACTION

(* POU SBR_TRANSFER_2, CFC *)
PROGRAM SBR_TRANSFER_2
VAR
	LSL103B : inBlock;
	LSS103B : inBlock;
	LSH103B : inBlock;
	LSD103B : inBlock;

	bXV205B : BOOL;
 	bXV206B : BOOL;
	bXV207B : BOOL;
	bXV208B : BOOL;
	bSBRTransfer:BOOL;


	bWarningSBRDry: BOOL;
	bCriticalSBRDry: BOOL;
	bCriticalSBRHi: BOOL;
	P102B: fb_equipment_with_linking;
END_VAR
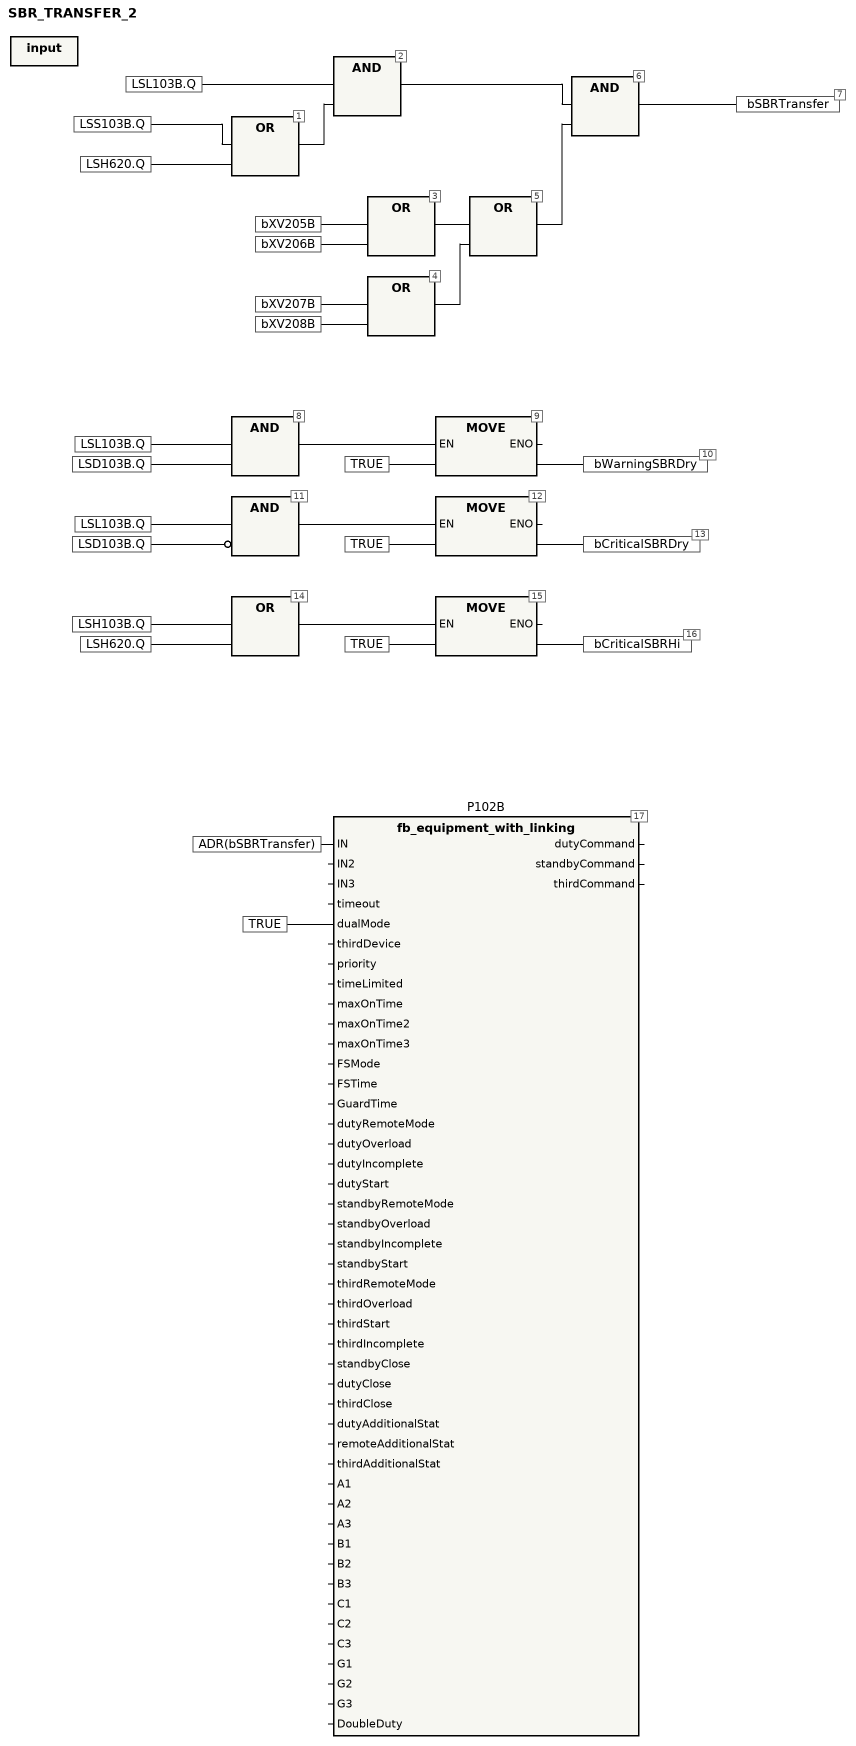
_CFC_ (* Continuous Function Chart, elements in execution order *)
#0 input()
#1 OR(LSS103B.Q, LSH620.Q)
#2 AND(LSL103B.Q, #1)
#3 OR(bXV205B, bXV206B)
#4 OR(bXV207B, bXV208B)
#5 OR(#3, #4)
#6 AND(#2, #5)
#7 bSBRTransfer <= #6
#8 AND(LSL103B.Q, LSD103B.Q)
#9 MOVE(EN: #8, TRUE)
#10 bWarningSBRDry <= #9
#11 AND(LSL103B.Q, NOT LSD103B.Q)
#12 MOVE(EN: #11, TRUE)
#13 bCriticalSBRDry <= #12
#14 OR(LSH103B.Q, LSH620.Q)
#15 MOVE(EN: #14, TRUE)
#16 bCriticalSBRHi <= #15
#17 P102B:fb_equipment_with_linking(IN: ADR(bSBRTransfer), IN2: -, IN3: -, timeout: -, dualMode: TRUE, thirdDevice: -, priority: -, timeLimited: -, maxOnTime: -, maxOnTime2: -, maxOnTime3: -, FSMode: -, FSTime: -, GuardTime: -, dutyRemoteMode: -, dutyOverload: -, dutyIncomplete: -, dutyStart: -, standbyRemoteMode: -, standbyOverload: -, standbyIncomplete: -, standbyStart: -, thirdRemoteMode: -, thirdOverload: -, thirdStart: -, thirdIncomplete: -, standbyClose: -, dutyClose: -, thirdClose: -, dutyAdditionalStat: -, remoteAdditionalStat: -, thirdAdditionalStat: -, A1: -, A2: -, A3: -, B1: -, B2: -, B3: -, C1: -, C2: -, C3: -, G1: -, G2: -, G3: -, DoubleDuty: -)
_END_CFC_
(* the same logic as Structured Text *)
input();
bSBRTransfer := (LSL103B.Q AND (LSS103B.Q OR LSH620.Q)) AND ((bXV205B OR bXV206B) OR (bXV207B OR bXV208B));
IF LSL103B.Q AND LSD103B.Q THEN bWarningSBRDry := TRUE; END_IF;
IF LSL103B.Q AND NOT LSD103B.Q THEN bCriticalSBRDry := TRUE; END_IF;
IF LSH103B.Q OR LSH620.Q THEN bCriticalSBRHi := TRUE; END_IF;
P102B(IN := ADR(bSBRTransfer), dualMode := TRUE);
END_PROGRAM
ACTION Input:
LSD103B( );
LSH103B();
LSH620( );
LSL103B( );
LSS103B( );
END_ACTION

(* POU GRIT_REMOVAL_OPERATION, CFC *)
PROGRAM GRIT_REMOVAL_OPERATION
VAR
	bGritAirBlower: BOOL;
	bGritClasifier: BOOL;
	bSuctionValveOperation: BOOL;
	offGritClassifier: TON;
	B101A: fb_equipment_with_linking;
	bSuctionValveA1: BOOL;
	bSuctionValveA2: BOOL;
	bSuctionValveB1: BOOL;
	bSuctionValveB2: BOOL;
	XV100A: fb_equipment_with_linking;
	XV100B: fb_equipment_with_linking;
	bGritClassifierA: BOOL;
	bGritClassifierB: BOOL;
	C103AandB: fb_equipment_with_linking;
END_VAR
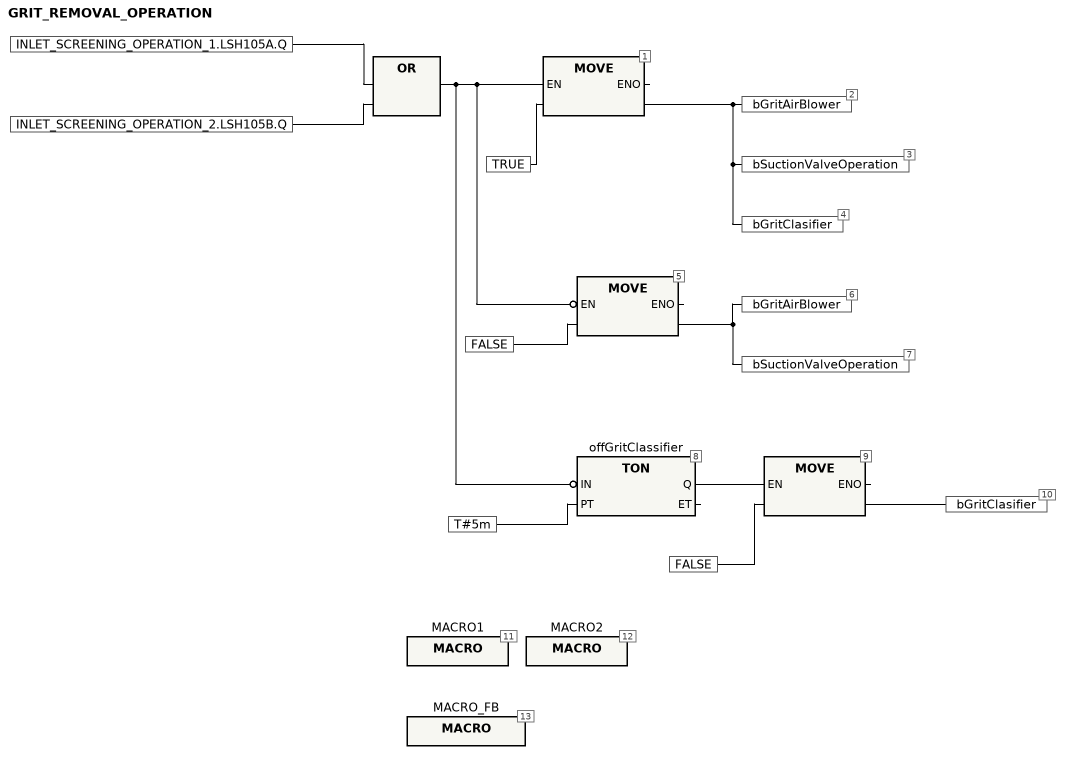
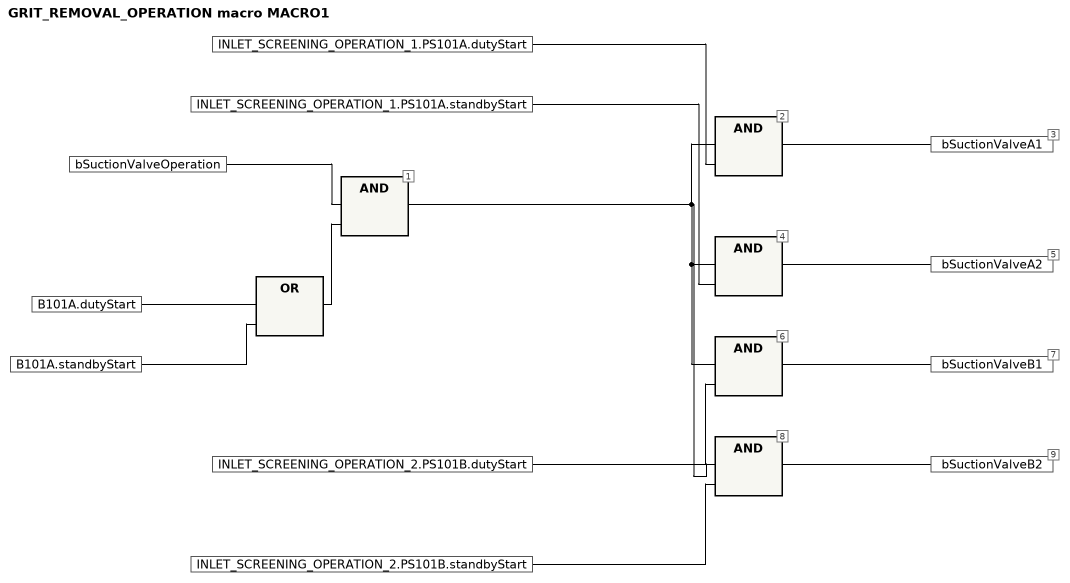
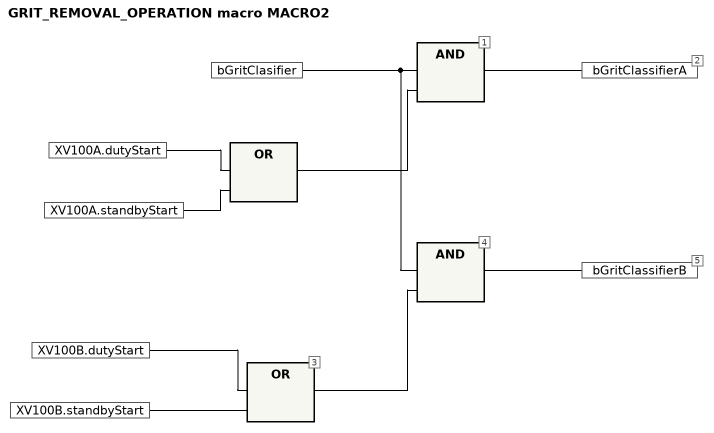
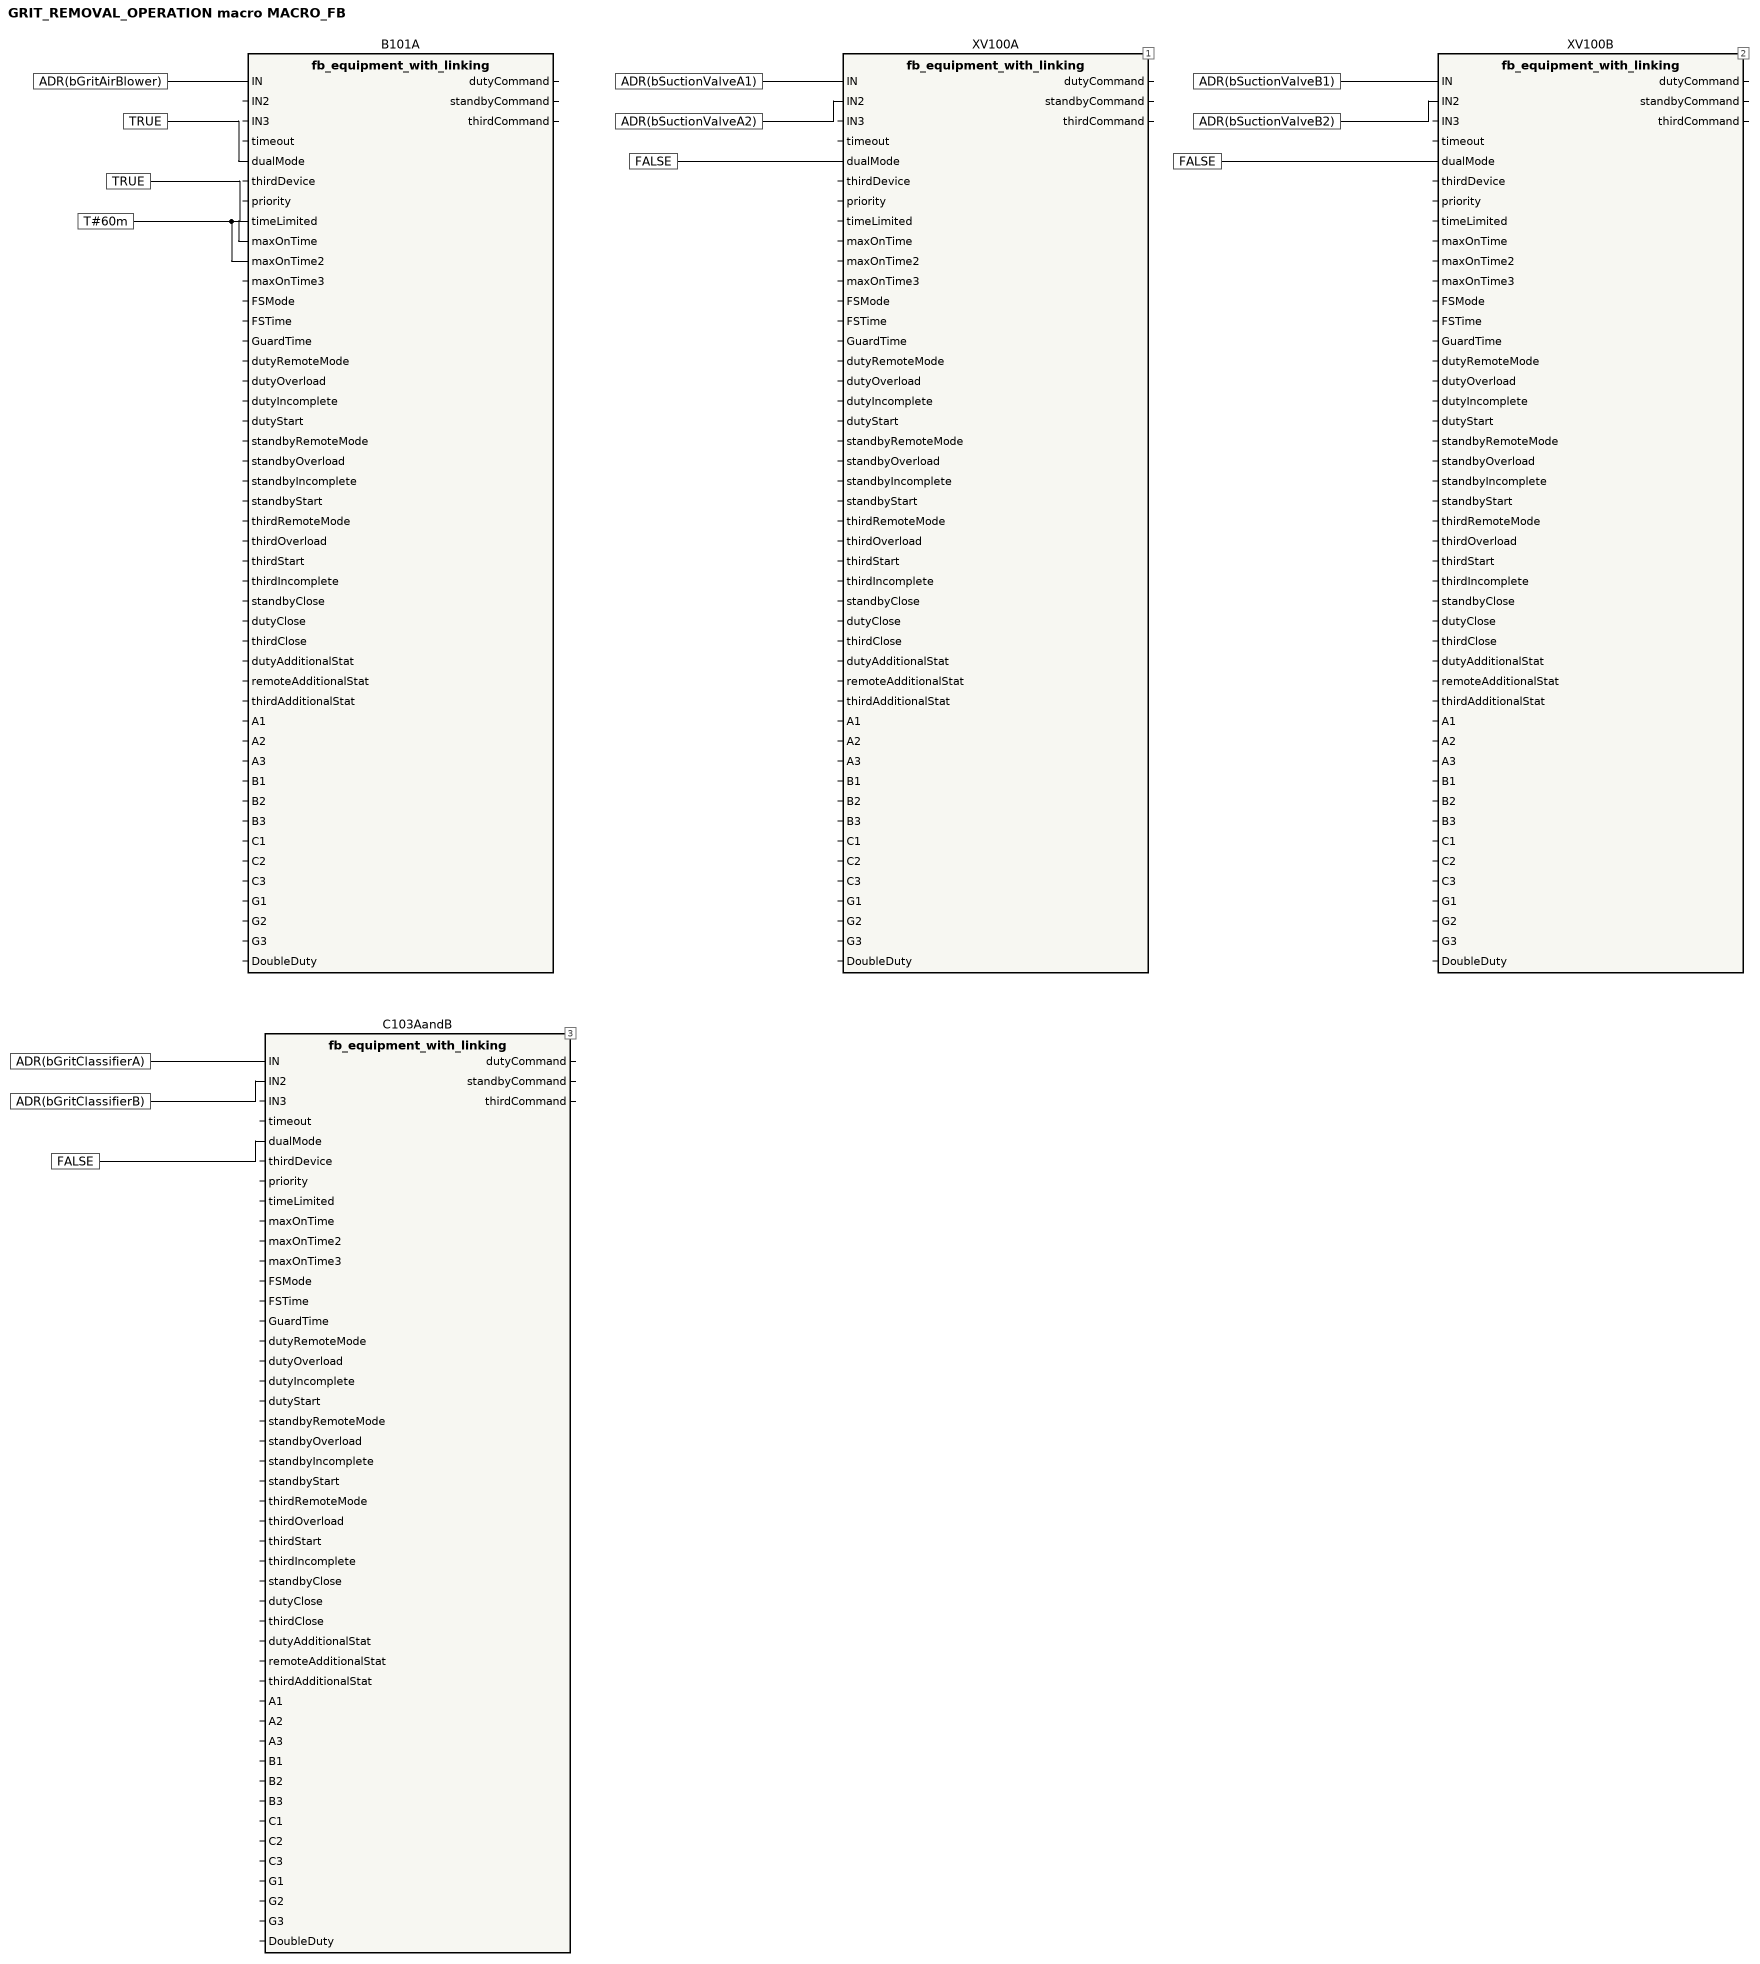
_CFC_ (* Continuous Function Chart, elements in execution order *)
#0 OR(INLET_SCREENING_OPERATION_1.LSH105A.Q, INLET_SCREENING_OPERATION_2.LSH105B.Q)
#1 MOVE(EN: #0, TRUE)
#2 bGritAirBlower <= #1
#3 bSuctionValveOperation <= #1
#4 bGritClasifier <= #1
#5 MOVE(EN: NOT #0, FALSE)
#6 bGritAirBlower <= #5
#7 bSuctionValveOperation <= #5
#8 offGritClassifier:TON(IN: NOT #0, PT: T#5m)
#9 MOVE(EN: #8.Q, FALSE)
#10 bGritClasifier <= #9
#11 MACRO MACRO1()
	#12 OR(B101A.dutyStart, B101A.standbyStart)
	#13 AND(bSuctionValveOperation, #12)
	#14 AND(#13, INLET_SCREENING_OPERATION_1.PS101A.dutyStart)
	#15 bSuctionValveA1 <= #14
	#16 AND(#13, INLET_SCREENING_OPERATION_1.PS101A.standbyStart)
	#17 bSuctionValveA2 <= #16
	#18 AND(#13, INLET_SCREENING_OPERATION_2.PS101B.dutyStart)
	#19 bSuctionValveB1 <= #18
	#20 AND(#13, INLET_SCREENING_OPERATION_2.PS101B.standbyStart)
	#21 bSuctionValveB2 <= #20
END_MACRO
#22 MACRO MACRO2()
	#23 OR(XV100A.dutyStart, XV100A.standbyStart)
	#24 AND(bGritClasifier, #23)
	#25 bGritClassifierA <= #24
	#26 OR(XV100B.dutyStart, XV100B.standbyStart)
	#27 AND(bGritClasifier, #26)
	#28 bGritClassifierB <= #27
END_MACRO
#29 MACRO MACRO_FB()
	#30 B101A:fb_equipment_with_linking(IN: ADR(bGritAirBlower), IN2: -, IN3: -, timeout: -, dualMode: TRUE, thirdDevice: -, priority: -, timeLimited: TRUE, maxOnTime: T#60m, maxOnTime2: T#60m, maxOnTime3: -, FSMode: -, FSTime: -, GuardTime: -, dutyRemoteMode: -, dutyOverload: -, dutyIncomplete: -, dutyStart: -, standbyRemoteMode: -, standbyOverload: -, standbyIncomplete: -, standbyStart: -, thirdRemoteMode: -, thirdOverload: -, thirdStart: -, thirdIncomplete: -, standbyClose: -, dutyClose: -, thirdClose: -, dutyAdditionalStat: -, remoteAdditionalStat: -, thirdAdditionalStat: -, A1: -, A2: -, A3: -, B1: -, B2: -, B3: -, C1: -, C2: -, C3: -, G1: -, G2: -, G3: -, DoubleDuty: -)
	#31 XV100A:fb_equipment_with_linking(IN: ADR(bSuctionValveA1), IN2: ADR(bSuctionValveA2), IN3: -, timeout: -, dualMode: FALSE, thirdDevice: -, priority: -, timeLimited: -, maxOnTime: -, maxOnTime2: -, maxOnTime3: -, FSMode: -, FSTime: -, GuardTime: -, dutyRemoteMode: -, dutyOverload: -, dutyIncomplete: -, dutyStart: -, standbyRemoteMode: -, standbyOverload: -, standbyIncomplete: -, standbyStart: -, thirdRemoteMode: -, thirdOverload: -, thirdStart: -, thirdIncomplete: -, standbyClose: -, dutyClose: -, thirdClose: -, dutyAdditionalStat: -, remoteAdditionalStat: -, thirdAdditionalStat: -, A1: -, A2: -, A3: -, B1: -, B2: -, B3: -, C1: -, C2: -, C3: -, G1: -, G2: -, G3: -, DoubleDuty: -)
	#32 XV100B:fb_equipment_with_linking(IN: ADR(bSuctionValveB1), IN2: ADR(bSuctionValveB2), IN3: -, timeout: -, dualMode: FALSE, thirdDevice: -, priority: -, timeLimited: -, maxOnTime: -, maxOnTime2: -, maxOnTime3: -, FSMode: -, FSTime: -, GuardTime: -, dutyRemoteMode: -, dutyOverload: -, dutyIncomplete: -, dutyStart: -, standbyRemoteMode: -, standbyOverload: -, standbyIncomplete: -, standbyStart: -, thirdRemoteMode: -, thirdOverload: -, thirdStart: -, thirdIncomplete: -, standbyClose: -, dutyClose: -, thirdClose: -, dutyAdditionalStat: -, remoteAdditionalStat: -, thirdAdditionalStat: -, A1: -, A2: -, A3: -, B1: -, B2: -, B3: -, C1: -, C2: -, C3: -, G1: -, G2: -, G3: -, DoubleDuty: -)
	#33 C103AandB:fb_equipment_with_linking(IN: ADR(bGritClassifierA), IN2: ADR(bGritClassifierB), IN3: -, timeout: -, dualMode: FALSE, thirdDevice: -, priority: -, timeLimited: -, maxOnTime: -, maxOnTime2: -, maxOnTime3: -, FSMode: -, FSTime: -, GuardTime: -, dutyRemoteMode: -, dutyOverload: -, dutyIncomplete: -, dutyStart: -, standbyRemoteMode: -, standbyOverload: -, standbyIncomplete: -, standbyStart: -, thirdRemoteMode: -, thirdOverload: -, thirdStart: -, thirdIncomplete: -, standbyClose: -, dutyClose: -, thirdClose: -, dutyAdditionalStat: -, remoteAdditionalStat: -, thirdAdditionalStat: -, A1: -, A2: -, A3: -, B1: -, B2: -, B3: -, C1: -, C2: -, C3: -, G1: -, G2: -, G3: -, DoubleDuty: -)
END_MACRO
_END_CFC_
END_PROGRAM

(* POU REUSE_WATER_SYSTEM, CFC *)
PROGRAM REUSE_WATER_SYSTEM
VAR
	bVacumPrimingOperation: BOOL;
	LSH405 : inBlock;
	LSL308A : inBlock;
	LSH308A : inBlock;
	bSolenoidValve: BOOL;
	bVacumPumDuty: BOOL;
	WaitToFill: TON;
	FSL101:inBlock;
	bWarning_PrimingNoWater: BOOL;
	bTriggerNegative: BOOL;
	bOverrideON: BOOL;
	bOverrideOFF: BOOL;
	bTriggerPositive: BOOL;
	TOverrideON: TON;
	TOverrideOFF: TON;
	bJokeyPump: BOOL;
	PSL411 AT%I* : INT;
	rWaterPressureSensor:REAL;
	bPumpSequence: BOOL;
	Lower_3_5_timer: TON;
	bLeadPumpAB: BOOL;
	bLeadPumpCD: BOOL;
	bWarningWaterPressureHigh: BOOL;
	PSL412 AT%I*: BOOL;
	bJokeyPumpInternalOff: BOOL;
	P403: fb_equipment_with_linking;
	P402: fb_equipment_with_linking;
	P401AB: fb_equipment_with_linking;
	P401CD: fb_equipment_with_linking;

	XV102: fb_equipment_with_linking;
END_VAR
VAR (* helpers for the ST form of the networks *)
	_t23 : BOOL;
	_t1 : BOOL;
	_t10 : BOOL;
	_t4 : BOOL;
	_t109 : BOOL;
	_t44 : BOOL;
	_en56 : BOOL;
	_en89 : BOOL;
	_t102 : BOOL;
	_t101 : BOOL;
	_t49 : BOOL;
	_t56 : BOOL;
	_t62 : BOOL;
	_en65 : BOOL;
	_t65 : BOOL;
	_t68 : BOOL;
	_t73 : BOOL;
	_t77 : BOOL;
	_en78 : BOOL;
	_t78 : BOOL;
	_t89 : BOOL;
	_t88 : BOOL;
	_t97 : BOOL;
END_VAR
